// TIA Portal V19 export
FUNCTION "SUB_OUTPUT" : Void   // FC5, LAD
{ S7_Optimized_Access := 'TRUE' }
// stored: SetENOAutomatically false
   VAR_TEMP   // added for the SCL form of the ladder/FBD networks
      _w1 : Bool;
   END_VAR
BEGIN

REGION Network 2: "CENTRIFUGAL_PUMP-1"
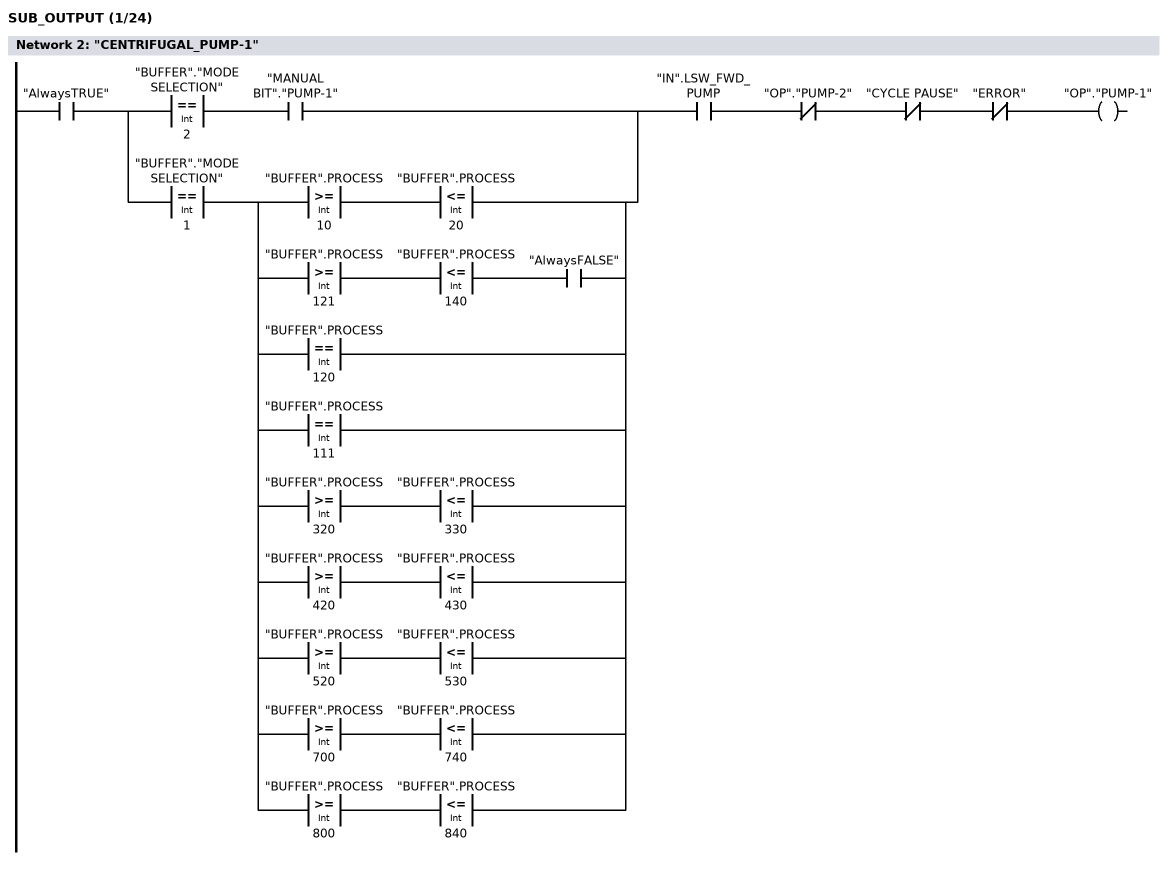
   RUNG wire#powerrail
      Contact( "AlwaysTRUE" )
      wire#w1
      { S7_Templates := "SrcType := Int" } EQ_Contact(in1 := "BUFFER"."MODE SELECTION", in2 := 2)
      Contact( "MANUAL BIT"."PUMP-1" )
      wire#w2
      Contact( "IN".LSW_FWD_PUMP )
      I_Contact( "OP"."PUMP-2" )
      I_Contact( "CYCLE PAUSE" )
      I_Contact( "ERROR" )
      Coil( "OP"."PUMP-1" )
   END_RUNG
   RUNG wire#w1
      { S7_Templates := "SrcType := Int" } EQ_Contact(in1 := "BUFFER"."MODE SELECTION", in2 := 1)
      wire#w3
      { S7_Templates := "SrcType := Int" } GE_Contact(in1 := "BUFFER".PROCESS, in2 := 10)
      { S7_Templates := "SrcType := Int" } LE_Contact(in1 := "BUFFER".PROCESS, in2 := 20)
   END_RUNG wire#w2
   RUNG wire#w3
      { S7_Templates := "SrcType := Int" } GE_Contact(in1 := "BUFFER".PROCESS, in2 := 121)
      { S7_Templates := "SrcType := Int" } LE_Contact(in1 := "BUFFER".PROCESS, in2 := 140)
      Contact( "AlwaysFALSE" )
   END_RUNG wire#w2
   RUNG wire#w3
      { S7_Templates := "SrcType := Int" } EQ_Contact(in1 := "BUFFER".PROCESS, in2 := 120)
   END_RUNG wire#w2
   RUNG wire#w3
      { S7_Templates := "SrcType := Int" } EQ_Contact(in1 := "BUFFER".PROCESS, in2 := 111)
   END_RUNG wire#w2
   RUNG wire#w3
      { S7_Templates := "SrcType := Int" } GE_Contact(in1 := "BUFFER".PROCESS, in2 := 320)
      { S7_Templates := "SrcType := Int" } LE_Contact(in1 := "BUFFER".PROCESS, in2 := 330)
   END_RUNG wire#w2
   RUNG wire#w3
      { S7_Templates := "SrcType := Int" } GE_Contact(in1 := "BUFFER".PROCESS, in2 := 420)
      { S7_Templates := "SrcType := Int" } LE_Contact(in1 := "BUFFER".PROCESS, in2 := 430)
   END_RUNG wire#w2
   RUNG wire#w3
      { S7_Templates := "SrcType := Int" } GE_Contact(in1 := "BUFFER".PROCESS, in2 := 520)
      { S7_Templates := "SrcType := Int" } LE_Contact(in1 := "BUFFER".PROCESS, in2 := 530)
   END_RUNG wire#w2
   RUNG wire#w3
      { S7_Templates := "SrcType := Int" } GE_Contact(in1 := "BUFFER".PROCESS, in2 := 700)
      { S7_Templates := "SrcType := Int" } LE_Contact(in1 := "BUFFER".PROCESS, in2 := 740)
   END_RUNG wire#w2
   RUNG wire#w3
      { S7_Templates := "SrcType := Int" } GE_Contact(in1 := "BUFFER".PROCESS, in2 := 800)
      { S7_Templates := "SrcType := Int" } LE_Contact(in1 := "BUFFER".PROCESS, in2 := 840)
   END_RUNG wire#w2
   // the same network as SCL:
   "OP"."PUMP-1" := "AlwaysTRUE" AND ((("BUFFER"."MODE SELECTION" = 2) AND "MANUAL BIT"."PUMP-1") OR (("BUFFER"."MODE SELECTION" = 1) AND ((("BUFFER".PROCESS >= 10) AND ("BUFFER".PROCESS <= 20)) OR (("BUFFER".PROCESS >= 121) AND ("BUFFER".PROCESS <= 140) AND "AlwaysFALSE") OR ("BUFFER".PROCESS = 120) OR ("BUFFER".PROCESS = 111) OR (("BUFFER".PROCESS >= 320) AND ("BUFFER".PROCESS <= 330)) OR (("BUFFER".PROCESS >= 420) AND ("BUFFER".PROCESS <= 430)) OR (("BUFFER".PROCESS >= 520) AND ("BUFFER".PROCESS <= 530)) OR (("BUFFER".PROCESS >= 700) AND ("BUFFER".PROCESS <= 740)) OR (("BUFFER".PROCESS >= 800) AND ("BUFFER".PROCESS <= 840))))) AND "IN".LSW_FWD_PUMP AND NOT "OP"."PUMP-2" AND NOT "CYCLE PAUSE" AND NOT "ERROR";
END_REGION

REGION Network 3: "CENTRIFUGAL_PUMP-2"
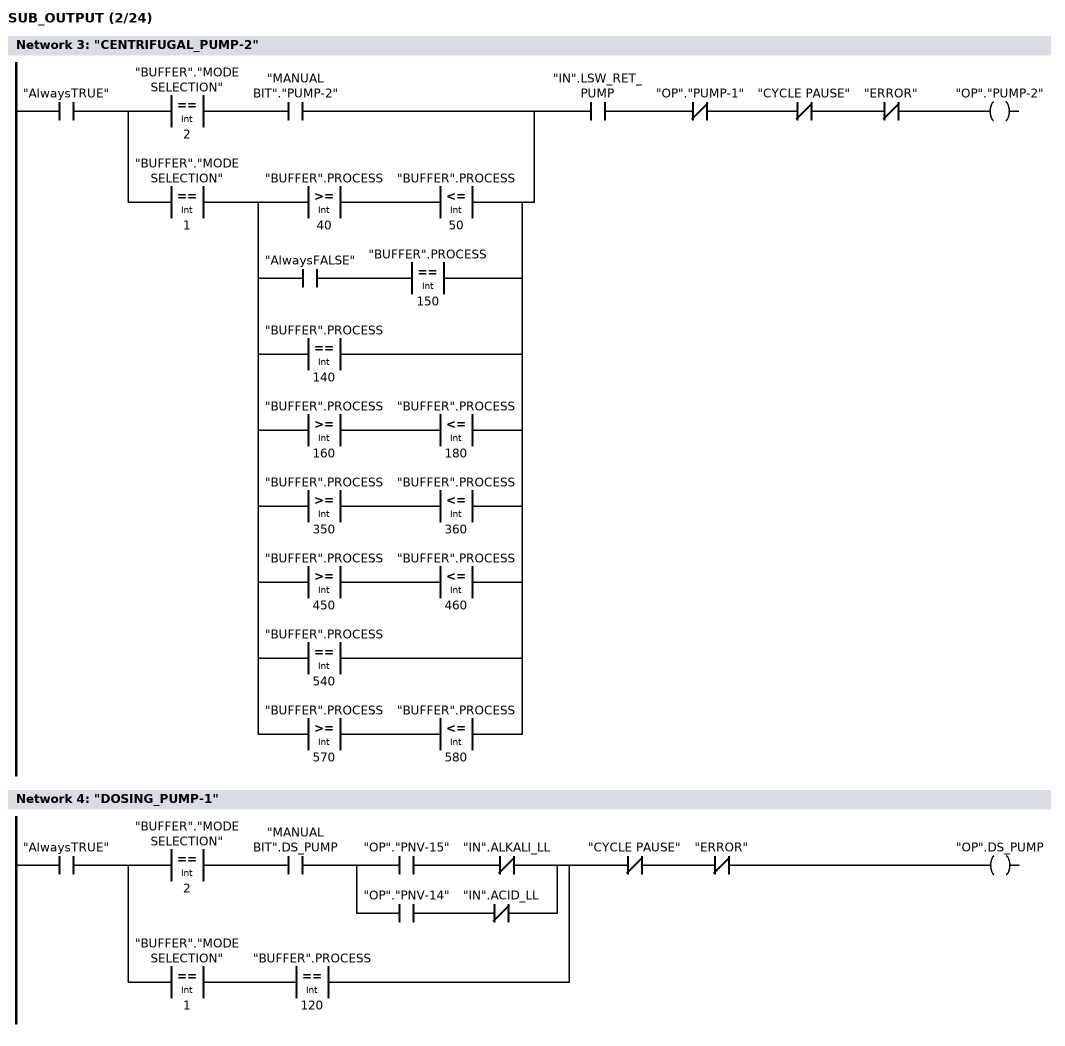
   RUNG wire#powerrail
      Contact( "AlwaysTRUE" )
      wire#w1
      { S7_Templates := "SrcType := Int" } EQ_Contact(in1 := "BUFFER"."MODE SELECTION", in2 := 2)
      Contact( "MANUAL BIT"."PUMP-2" )
      wire#w2
      Contact( "IN".LSW_RET_PUMP )
      I_Contact( "OP"."PUMP-1" )
      I_Contact( "CYCLE PAUSE" )
      I_Contact( "ERROR" )
      Coil( "OP"."PUMP-2" )
   END_RUNG
   RUNG wire#w1
      { S7_Templates := "SrcType := Int" } EQ_Contact(in1 := "BUFFER"."MODE SELECTION", in2 := 1)
      wire#w3
      { S7_Templates := "SrcType := Int" } GE_Contact(in1 := "BUFFER".PROCESS, in2 := 40)
      { S7_Templates := "SrcType := Int" } LE_Contact(in1 := "BUFFER".PROCESS, in2 := 50)
   END_RUNG wire#w2
   RUNG wire#w3
      Contact( "AlwaysFALSE" )
      { S7_Templates := "SrcType := Int" } EQ_Contact(in1 := "BUFFER".PROCESS, in2 := 150)
   END_RUNG wire#w2
   RUNG wire#w3
      { S7_Templates := "SrcType := Int" } EQ_Contact(in1 := "BUFFER".PROCESS, in2 := 140)
   END_RUNG wire#w2
   RUNG wire#w3
      { S7_Templates := "SrcType := Int" } GE_Contact(in1 := "BUFFER".PROCESS, in2 := 160)
      { S7_Templates := "SrcType := Int" } LE_Contact(in1 := "BUFFER".PROCESS, in2 := 180)
   END_RUNG wire#w2
   RUNG wire#w3
      { S7_Templates := "SrcType := Int" } GE_Contact(in1 := "BUFFER".PROCESS, in2 := 350)
      { S7_Templates := "SrcType := Int" } LE_Contact(in1 := "BUFFER".PROCESS, in2 := 360)
   END_RUNG wire#w2
   RUNG wire#w3
      { S7_Templates := "SrcType := Int" } GE_Contact(in1 := "BUFFER".PROCESS, in2 := 450)
      { S7_Templates := "SrcType := Int" } LE_Contact(in1 := "BUFFER".PROCESS, in2 := 460)
   END_RUNG wire#w2
   RUNG wire#w3
      { S7_Templates := "SrcType := Int" } EQ_Contact(in1 := "BUFFER".PROCESS, in2 := 540)
   END_RUNG wire#w2
   RUNG wire#w3
      { S7_Templates := "SrcType := Int" } GE_Contact(in1 := "BUFFER".PROCESS, in2 := 570)
      { S7_Templates := "SrcType := Int" } LE_Contact(in1 := "BUFFER".PROCESS, in2 := 580)
   END_RUNG wire#w2
   // the same network as SCL:
   "OP"."PUMP-2" := "AlwaysTRUE" AND ((("BUFFER"."MODE SELECTION" = 2) AND "MANUAL BIT"."PUMP-2") OR (("BUFFER"."MODE SELECTION" = 1) AND ((("BUFFER".PROCESS >= 40) AND ("BUFFER".PROCESS <= 50)) OR ("AlwaysFALSE" AND ("BUFFER".PROCESS = 150)) OR ("BUFFER".PROCESS = 140) OR (("BUFFER".PROCESS >= 160) AND ("BUFFER".PROCESS <= 180)) OR (("BUFFER".PROCESS >= 350) AND ("BUFFER".PROCESS <= 360)) OR (("BUFFER".PROCESS >= 450) AND ("BUFFER".PROCESS <= 460)) OR ("BUFFER".PROCESS = 540) OR (("BUFFER".PROCESS >= 570) AND ("BUFFER".PROCESS <= 580))))) AND "IN".LSW_RET_PUMP AND NOT "OP"."PUMP-1" AND NOT "CYCLE PAUSE" AND NOT "ERROR";
END_REGION

REGION Network 4: "DOSING_PUMP-1"
   RUNG wire#powerrail
      Contact( "AlwaysTRUE" )
      wire#w1
      { S7_Templates := "SrcType := Int" } EQ_Contact(in1 := "BUFFER"."MODE SELECTION", in2 := 2)
      Contact( "MANUAL BIT".DS_PUMP )
      wire#w2
      Contact( "OP"."PNV-15" )
      I_Contact( "IN".ALKALI_LL )
      wire#w3
      I_Contact( "CYCLE PAUSE" )
      I_Contact( "ERROR" )
      Coil( "OP".DS_PUMP )
   END_RUNG
   RUNG wire#w2
      Contact( "OP"."PNV-14" )
      I_Contact( "IN".ACID_LL )
   END_RUNG wire#w3
   RUNG wire#w1
      { S7_Templates := "SrcType := Int" } EQ_Contact(in1 := "BUFFER"."MODE SELECTION", in2 := 1)
      { S7_Templates := "SrcType := Int" } EQ_Contact(in1 := "BUFFER".PROCESS, in2 := 120)
   END_RUNG wire#w3
   // the same network as SCL:
   "OP".DS_PUMP := "AlwaysTRUE" AND ((("BUFFER"."MODE SELECTION" = 2) AND "MANUAL BIT".DS_PUMP AND (("OP"."PNV-15" AND NOT "IN".ALKALI_LL) OR ("OP"."PNV-14" AND NOT "IN".ACID_LL))) OR (("BUFFER"."MODE SELECTION" = 1) AND ("BUFFER".PROCESS = 120))) AND NOT "CYCLE PAUSE" AND NOT "ERROR";
END_REGION

REGION Network 5: "PBV-125 PURIFIED WATER VESSEL OUTLET VALVE"
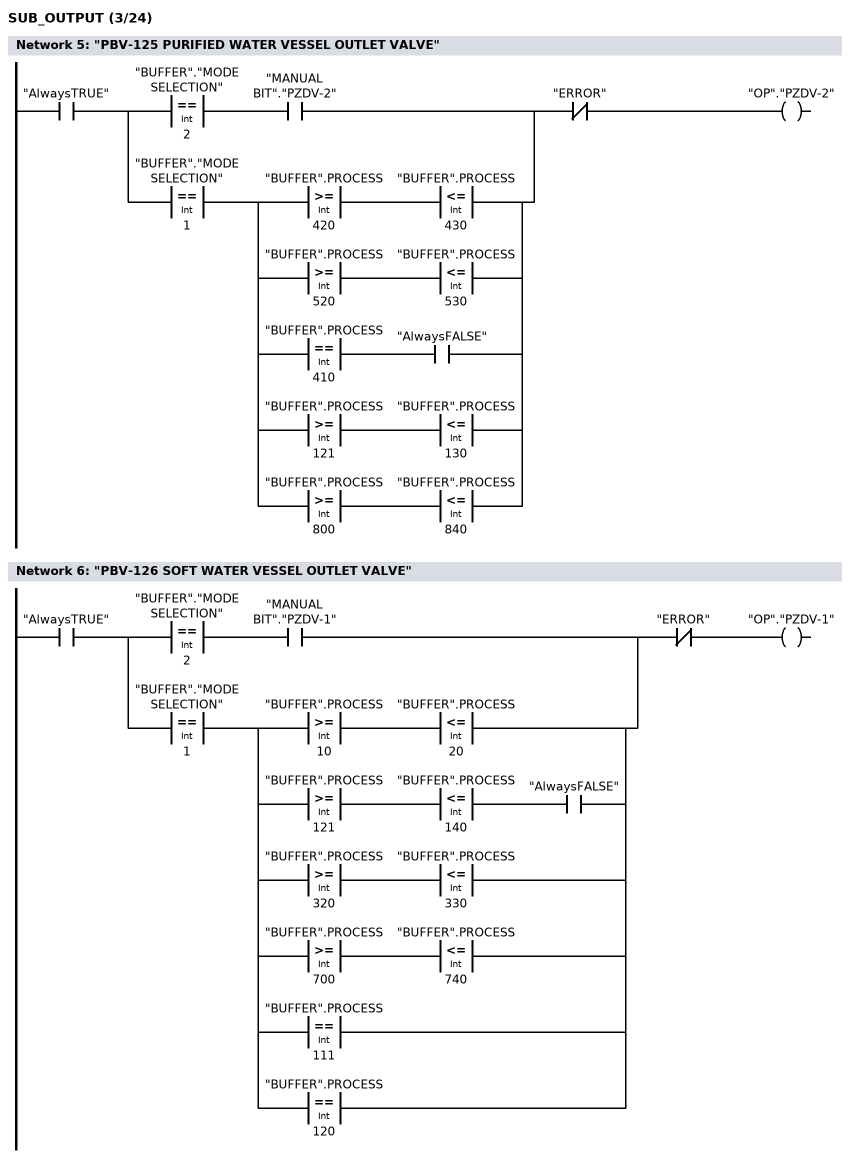
   RUNG wire#powerrail
      Contact( "AlwaysTRUE" )
      wire#w1
      { S7_Templates := "SrcType := Int" } EQ_Contact(in1 := "BUFFER"."MODE SELECTION", in2 := 2)
      Contact( "MANUAL BIT"."PZDV-2" )
      wire#w2
      I_Contact( "ERROR" )
      Coil( "OP"."PZDV-2" )
   END_RUNG
   RUNG wire#w1
      { S7_Templates := "SrcType := Int" } EQ_Contact(in1 := "BUFFER"."MODE SELECTION", in2 := 1)
      wire#w3
      { S7_Templates := "SrcType := Int" } GE_Contact(in1 := "BUFFER".PROCESS, in2 := 420)
      { S7_Templates := "SrcType := Int" } LE_Contact(in1 := "BUFFER".PROCESS, in2 := 430)
   END_RUNG wire#w2
   RUNG wire#w3
      { S7_Templates := "SrcType := Int" } GE_Contact(in1 := "BUFFER".PROCESS, in2 := 520)
      { S7_Templates := "SrcType := Int" } LE_Contact(in1 := "BUFFER".PROCESS, in2 := 530)
   END_RUNG wire#w2
   RUNG wire#w3
      { S7_Templates := "SrcType := Int" } EQ_Contact(in1 := "BUFFER".PROCESS, in2 := 410)
      Contact( "AlwaysFALSE" )
   END_RUNG wire#w2
   RUNG wire#w3
      { S7_Templates := "SrcType := Int" } GE_Contact(in1 := "BUFFER".PROCESS, in2 := 121)
      { S7_Templates := "SrcType := Int" } LE_Contact(in1 := "BUFFER".PROCESS, in2 := 130)
   END_RUNG wire#w2
   RUNG wire#w3
      { S7_Templates := "SrcType := Int" } GE_Contact(in1 := "BUFFER".PROCESS, in2 := 800)
      { S7_Templates := "SrcType := Int" } LE_Contact(in1 := "BUFFER".PROCESS, in2 := 840)
   END_RUNG wire#w2
   // the same network as SCL:
   "OP"."PZDV-2" := "AlwaysTRUE" AND ((("BUFFER"."MODE SELECTION" = 2) AND "MANUAL BIT"."PZDV-2") OR (("BUFFER"."MODE SELECTION" = 1) AND ((("BUFFER".PROCESS >= 420) AND ("BUFFER".PROCESS <= 430)) OR (("BUFFER".PROCESS >= 520) AND ("BUFFER".PROCESS <= 530)) OR (("BUFFER".PROCESS = 410) AND "AlwaysFALSE") OR (("BUFFER".PROCESS >= 121) AND ("BUFFER".PROCESS <= 130)) OR (("BUFFER".PROCESS >= 800) AND ("BUFFER".PROCESS <= 840))))) AND NOT "ERROR";
END_REGION

REGION Network 6: "PBV-126 SOFT WATER VESSEL OUTLET VALVE"
   RUNG wire#powerrail
      Contact( "AlwaysTRUE" )
      wire#w1
      { S7_Templates := "SrcType := Int" } EQ_Contact(in1 := "BUFFER"."MODE SELECTION", in2 := 2)
      Contact( "MANUAL BIT"."PZDV-1" )
      wire#w2
      I_Contact( "ERROR" )
      Coil( "OP"."PZDV-1" )
   END_RUNG
   RUNG wire#w1
      { S7_Templates := "SrcType := Int" } EQ_Contact(in1 := "BUFFER"."MODE SELECTION", in2 := 1)
      wire#w3
      { S7_Templates := "SrcType := Int" } GE_Contact(in1 := "BUFFER".PROCESS, in2 := 10)
      { S7_Templates := "SrcType := Int" } LE_Contact(in1 := "BUFFER".PROCESS, in2 := 20)
   END_RUNG wire#w2
   RUNG wire#w3
      { S7_Templates := "SrcType := Int" } GE_Contact(in1 := "BUFFER".PROCESS, in2 := 121)
      { S7_Templates := "SrcType := Int" } LE_Contact(in1 := "BUFFER".PROCESS, in2 := 140)
      Contact( "AlwaysFALSE" )
   END_RUNG wire#w2
   RUNG wire#w3
      { S7_Templates := "SrcType := Int" } GE_Contact(in1 := "BUFFER".PROCESS, in2 := 320)
      { S7_Templates := "SrcType := Int" } LE_Contact(in1 := "BUFFER".PROCESS, in2 := 330)
   END_RUNG wire#w2
   RUNG wire#w3
      { S7_Templates := "SrcType := Int" } GE_Contact(in1 := "BUFFER".PROCESS, in2 := 700)
      { S7_Templates := "SrcType := Int" } LE_Contact(in1 := "BUFFER".PROCESS, in2 := 740)
   END_RUNG wire#w2
   RUNG wire#w3
      { S7_Templates := "SrcType := Int" } EQ_Contact(in1 := "BUFFER".PROCESS, in2 := 111)
   END_RUNG wire#w2
   RUNG wire#w3
      { S7_Templates := "SrcType := Int" } EQ_Contact(in1 := "BUFFER".PROCESS, in2 := 120)
   END_RUNG wire#w2
   // the same network as SCL:
   "OP"."PZDV-1" := "AlwaysTRUE" AND ((("BUFFER"."MODE SELECTION" = 2) AND "MANUAL BIT"."PZDV-1") OR (("BUFFER"."MODE SELECTION" = 1) AND ((("BUFFER".PROCESS >= 10) AND ("BUFFER".PROCESS <= 20)) OR (("BUFFER".PROCESS >= 121) AND ("BUFFER".PROCESS <= 140) AND "AlwaysFALSE") OR (("BUFFER".PROCESS >= 320) AND ("BUFFER".PROCESS <= 330)) OR (("BUFFER".PROCESS >= 700) AND ("BUFFER".PROCESS <= 740)) OR ("BUFFER".PROCESS = 111) OR ("BUFFER".PROCESS = 120)))) AND NOT "ERROR";
END_REGION

REGION Network 7: "PBV-127 PW INLET LINE"
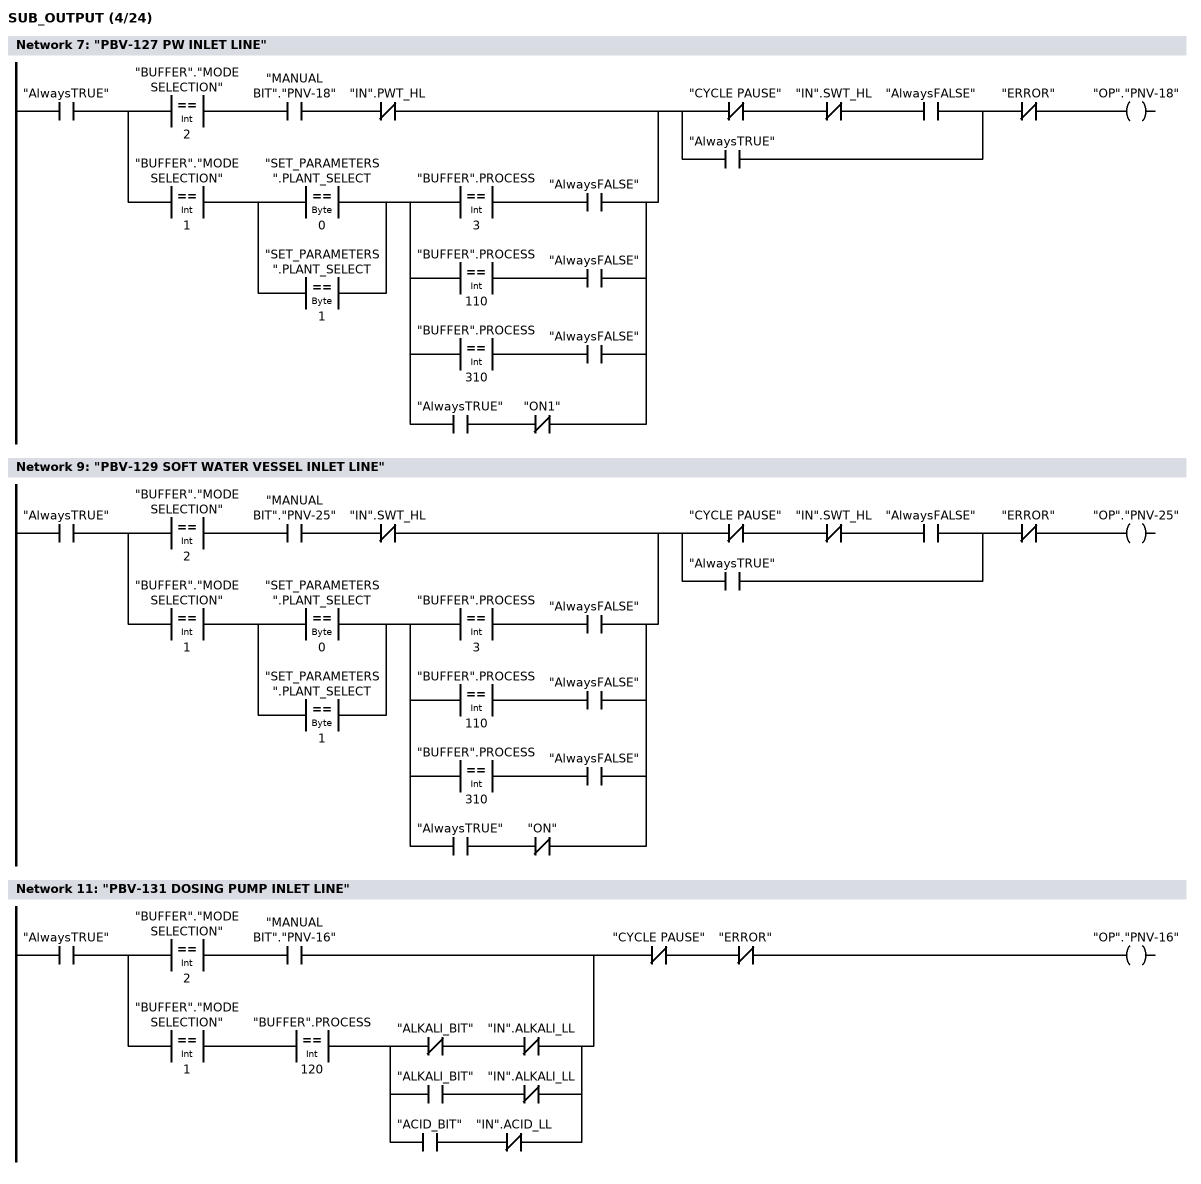
   RUNG wire#powerrail
      Contact( "AlwaysTRUE" )
      wire#w1
      { S7_Templates := "SrcType := Int" } EQ_Contact(in1 := "BUFFER"."MODE SELECTION", in2 := 2)
      Contact( "MANUAL BIT"."PNV-18" )
      I_Contact( "IN".PWT_HL )
      wire#w2
      I_Contact( "CYCLE PAUSE" )
      I_Contact( "IN".SWT_HL )
      Contact( "AlwaysFALSE" )
      wire#w5
      I_Contact( "ERROR" )
      Coil( "OP"."PNV-18" )
   END_RUNG
   RUNG wire#w1
      { S7_Templates := "SrcType := Int" } EQ_Contact(in1 := "BUFFER"."MODE SELECTION", in2 := 1)
      wire#w3
      { S7_Templates := "SrcType := Byte" } EQ_Contact(in1 := "SET_PARAMETERS".PLANT_SELECT, in2 := 0)
      wire#w4
      { S7_Templates := "SrcType := Int" } EQ_Contact(in1 := "BUFFER".PROCESS, in2 := 3)
      Contact( "AlwaysFALSE" )
   END_RUNG wire#w2
   RUNG wire#w3
      { S7_Templates := "SrcType := Byte" } EQ_Contact(in1 := "SET_PARAMETERS".PLANT_SELECT, in2 := 1)
   END_RUNG wire#w4
   RUNG wire#w4
      { S7_Templates := "SrcType := Int" } EQ_Contact(in1 := "BUFFER".PROCESS, in2 := 110)
      Contact( "AlwaysFALSE" )
   END_RUNG wire#w2
   RUNG wire#w4
      { S7_Templates := "SrcType := Int" } EQ_Contact(in1 := "BUFFER".PROCESS, in2 := 310)
      Contact( "AlwaysFALSE" )
   END_RUNG wire#w2
   RUNG wire#w4
      Contact( "AlwaysTRUE" )
      I_Contact( "ON1" )
   END_RUNG wire#w2
   RUNG wire#w2
      Contact( "AlwaysTRUE" )
   END_RUNG wire#w5
   // the same network as SCL:
   "OP"."PNV-18" := "AlwaysTRUE" AND ((("BUFFER"."MODE SELECTION" = 2) AND "MANUAL BIT"."PNV-18" AND NOT "IN".PWT_HL) OR (("BUFFER"."MODE SELECTION" = 1) AND (("SET_PARAMETERS".PLANT_SELECT = 0) OR ("SET_PARAMETERS".PLANT_SELECT = 1)) AND ((("BUFFER".PROCESS = 3) AND "AlwaysFALSE") OR (("BUFFER".PROCESS = 110) AND "AlwaysFALSE") OR (("BUFFER".PROCESS = 310) AND "AlwaysFALSE") OR ("AlwaysTRUE" AND NOT "ON1")))) AND ((NOT "CYCLE PAUSE" AND NOT "IN".SWT_HL AND "AlwaysFALSE") OR "AlwaysTRUE") AND NOT "ERROR";
END_REGION

REGION Network 8: "PBV-128 PURIFIED WATER VESSEL–SPRAY BALL INLET LINE"//////////////////NA
END_REGION

REGION Network 9: "PBV-129 SOFT WATER VESSEL INLET LINE"
   RUNG wire#powerrail
      Contact( "AlwaysTRUE" )
      wire#w1
      { S7_Templates := "SrcType := Int" } EQ_Contact(in1 := "BUFFER"."MODE SELECTION", in2 := 2)
      Contact( "MANUAL BIT"."PNV-25" )
      I_Contact( "IN".SWT_HL )
      wire#w2
      I_Contact( "CYCLE PAUSE" )
      I_Contact( "IN".SWT_HL )
      Contact( "AlwaysFALSE" )
      wire#w5
      I_Contact( "ERROR" )
      Coil( "OP"."PNV-25" )
   END_RUNG
   RUNG wire#w1
      { S7_Templates := "SrcType := Int" } EQ_Contact(in1 := "BUFFER"."MODE SELECTION", in2 := 1)
      wire#w3
      { S7_Templates := "SrcType := Byte" } EQ_Contact(in1 := "SET_PARAMETERS".PLANT_SELECT, in2 := 0)
      wire#w4
      { S7_Templates := "SrcType := Int" } EQ_Contact(in1 := "BUFFER".PROCESS, in2 := 3)
      Contact( "AlwaysFALSE" )
   END_RUNG wire#w2
   RUNG wire#w3
      { S7_Templates := "SrcType := Byte" } EQ_Contact(in1 := "SET_PARAMETERS".PLANT_SELECT, in2 := 1)
   END_RUNG wire#w4
   RUNG wire#w4
      { S7_Templates := "SrcType := Int" } EQ_Contact(in1 := "BUFFER".PROCESS, in2 := 110)
      Contact( "AlwaysFALSE" )
   END_RUNG wire#w2
   RUNG wire#w4
      { S7_Templates := "SrcType := Int" } EQ_Contact(in1 := "BUFFER".PROCESS, in2 := 310)
      Contact( "AlwaysFALSE" )
   END_RUNG wire#w2
   RUNG wire#w4
      Contact( "AlwaysTRUE" )
      I_Contact( "ON" )
   END_RUNG wire#w2
   RUNG wire#w2
      Contact( "AlwaysTRUE" )
   END_RUNG wire#w5
   // the same network as SCL:
   "OP"."PNV-25" := "AlwaysTRUE" AND ((("BUFFER"."MODE SELECTION" = 2) AND "MANUAL BIT"."PNV-25" AND NOT "IN".SWT_HL) OR (("BUFFER"."MODE SELECTION" = 1) AND (("SET_PARAMETERS".PLANT_SELECT = 0) OR ("SET_PARAMETERS".PLANT_SELECT = 1)) AND ((("BUFFER".PROCESS = 3) AND "AlwaysFALSE") OR (("BUFFER".PROCESS = 110) AND "AlwaysFALSE") OR (("BUFFER".PROCESS = 310) AND "AlwaysFALSE") OR ("AlwaysTRUE" AND NOT "ON")))) AND ((NOT "CYCLE PAUSE" AND NOT "IN".SWT_HL AND "AlwaysFALSE") OR "AlwaysTRUE") AND NOT "ERROR";
END_REGION

REGION Network 10: "PBV-130 SOFT WATER VESSEL–SPRAY BALL INLET LINE" /////////////////NA
END_REGION

REGION Network 11: "PBV-131 DOSING PUMP INLET LINE"
   RUNG wire#powerrail
      Contact( "AlwaysTRUE" )
      wire#w1
      { S7_Templates := "SrcType := Int" } EQ_Contact(in1 := "BUFFER"."MODE SELECTION", in2 := 2)
      Contact( "MANUAL BIT"."PNV-16" )
      wire#w2
      I_Contact( "CYCLE PAUSE" )
      I_Contact( "ERROR" )
      Coil( "OP"."PNV-16" )
   END_RUNG
   RUNG wire#w1
      { S7_Templates := "SrcType := Int" } EQ_Contact(in1 := "BUFFER"."MODE SELECTION", in2 := 1)
      { S7_Templates := "SrcType := Int" } EQ_Contact(in1 := "BUFFER".PROCESS, in2 := 120)
      wire#w3
      I_Contact( "ALKALI_BIT" )
      I_Contact( "IN".ALKALI_LL )
   END_RUNG wire#w2
   RUNG wire#w3
      Contact( "ALKALI_BIT" )
      I_Contact( "IN".ALKALI_LL )
   END_RUNG wire#w2
   RUNG wire#w3
      Contact( "ACID_BIT" )
      I_Contact( "IN".ACID_LL )
   END_RUNG wire#w2
   // the same network as SCL:
   "OP"."PNV-16" := "AlwaysTRUE" AND ((("BUFFER"."MODE SELECTION" = 2) AND "MANUAL BIT"."PNV-16") OR (("BUFFER"."MODE SELECTION" = 1) AND ("BUFFER".PROCESS = 120) AND ((NOT "ALKALI_BIT" AND NOT "IN".ALKALI_LL) OR ("ALKALI_BIT" AND NOT "IN".ALKALI_LL) OR ("ACID_BIT" AND NOT "IN".ACID_LL)))) AND NOT "CYCLE PAUSE" AND NOT "ERROR";
END_REGION

REGION Network 12: "PBV-132 PURIFIED WATER VESSEL OUTLET LINE" /////////////////NA
END_REGION

REGION Network 13: "PBV-133 SOFT WATER VESSEL OUTLET LINE" /////////////////NA
END_REGION

REGION Network 14: "PBV-134 FORWARD PUMP INLET LINE" /////////////////NA
END_REGION

REGION Network 15: "PBV-135 REVERSE PUMP CASING DRAIN"
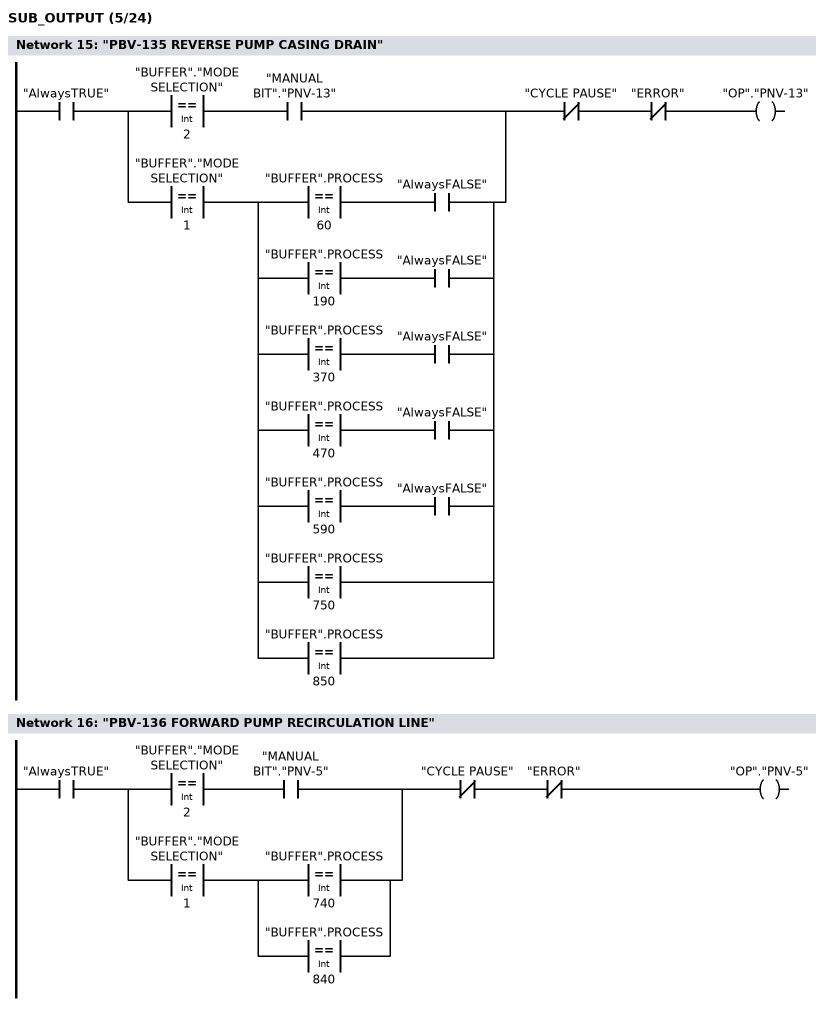
   RUNG wire#powerrail
      Contact( "AlwaysTRUE" )
      wire#w1
      { S7_Templates := "SrcType := Int" } EQ_Contact(in1 := "BUFFER"."MODE SELECTION", in2 := 2)
      Contact( "MANUAL BIT"."PNV-13" )
      wire#w2
      I_Contact( "CYCLE PAUSE" )
      I_Contact( "ERROR" )
      Coil( "OP"."PNV-13" )
   END_RUNG
   RUNG wire#w1
      { S7_Templates := "SrcType := Int" } EQ_Contact(in1 := "BUFFER"."MODE SELECTION", in2 := 1)
      wire#w3
      { S7_Templates := "SrcType := Int" } EQ_Contact(in1 := "BUFFER".PROCESS, in2 := 60)
      Contact( "AlwaysFALSE" )
   END_RUNG wire#w2
   RUNG wire#w3
      { S7_Templates := "SrcType := Int" } EQ_Contact(in1 := "BUFFER".PROCESS, in2 := 190)
      Contact( "AlwaysFALSE" )
   END_RUNG wire#w2
   RUNG wire#w3
      { S7_Templates := "SrcType := Int" } EQ_Contact(in1 := "BUFFER".PROCESS, in2 := 370)
      Contact( "AlwaysFALSE" )
   END_RUNG wire#w2
   RUNG wire#w3
      { S7_Templates := "SrcType := Int" } EQ_Contact(in1 := "BUFFER".PROCESS, in2 := 470)
      Contact( "AlwaysFALSE" )
   END_RUNG wire#w2
   RUNG wire#w3
      { S7_Templates := "SrcType := Int" } EQ_Contact(in1 := "BUFFER".PROCESS, in2 := 590)
      Contact( "AlwaysFALSE" )
   END_RUNG wire#w2
   RUNG wire#w3
      { S7_Templates := "SrcType := Int" } EQ_Contact(in1 := "BUFFER".PROCESS, in2 := 750)
   END_RUNG wire#w2
   RUNG wire#w3
      { S7_Templates := "SrcType := Int" } EQ_Contact(in1 := "BUFFER".PROCESS, in2 := 850)
   END_RUNG wire#w2
   // the same network as SCL:
   "OP"."PNV-13" := "AlwaysTRUE" AND ((("BUFFER"."MODE SELECTION" = 2) AND "MANUAL BIT"."PNV-13") OR (("BUFFER"."MODE SELECTION" = 1) AND ((("BUFFER".PROCESS = 60) AND "AlwaysFALSE") OR (("BUFFER".PROCESS = 190) AND "AlwaysFALSE") OR (("BUFFER".PROCESS = 370) AND "AlwaysFALSE") OR (("BUFFER".PROCESS = 470) AND "AlwaysFALSE") OR (("BUFFER".PROCESS = 590) AND "AlwaysFALSE") OR ("BUFFER".PROCESS = 750) OR ("BUFFER".PROCESS = 850)))) AND NOT "CYCLE PAUSE" AND NOT "ERROR";
END_REGION

REGION Network 16: "PBV-136 FORWARD PUMP RECIRCULATION LINE"
   RUNG wire#powerrail
      Contact( "AlwaysTRUE" )
      wire#w1
      { S7_Templates := "SrcType := Int" } EQ_Contact(in1 := "BUFFER"."MODE SELECTION", in2 := 2)
      Contact( "MANUAL BIT"."PNV-5" )
      wire#w2
      I_Contact( "CYCLE PAUSE" )
      I_Contact( "ERROR" )
      Coil( "OP"."PNV-5" )
   END_RUNG
   RUNG wire#w1
      { S7_Templates := "SrcType := Int" } EQ_Contact(in1 := "BUFFER"."MODE SELECTION", in2 := 1)
      wire#w3
      { S7_Templates := "SrcType := Int" } EQ_Contact(in1 := "BUFFER".PROCESS, in2 := 740)
   END_RUNG wire#w2
   RUNG wire#w3
      { S7_Templates := "SrcType := Int" } EQ_Contact(in1 := "BUFFER".PROCESS, in2 := 840)
   END_RUNG wire#w2
   // the same network as SCL:
   "OP"."PNV-5" := "AlwaysTRUE" AND ((("BUFFER"."MODE SELECTION" = 2) AND "MANUAL BIT"."PNV-5") OR (("BUFFER"."MODE SELECTION" = 1) AND (("BUFFER".PROCESS = 740) OR ("BUFFER".PROCESS = 840)))) AND NOT "CYCLE PAUSE" AND NOT "ERROR";
END_REGION

REGION Network 17: "PBV-137 FORWARD PUMP TO HEAT EXCHANGER LINE"
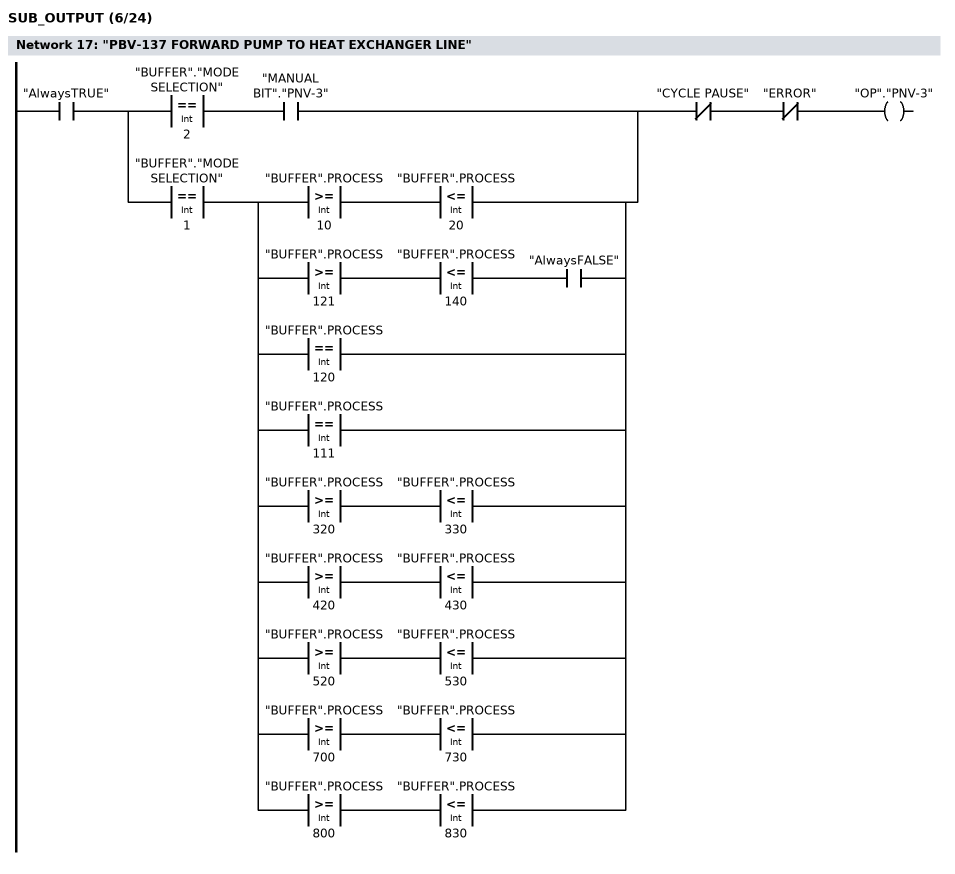
   RUNG wire#powerrail
      Contact( "AlwaysTRUE" )
      wire#w1
      { S7_Templates := "SrcType := Int" } EQ_Contact(in1 := "BUFFER"."MODE SELECTION", in2 := 2)
      Contact( "MANUAL BIT"."PNV-3" )
      wire#w2
      I_Contact( "CYCLE PAUSE" )
      I_Contact( "ERROR" )
      Coil( "OP"."PNV-3" )
   END_RUNG
   RUNG wire#w1
      { S7_Templates := "SrcType := Int" } EQ_Contact(in1 := "BUFFER"."MODE SELECTION", in2 := 1)
      wire#w3
      { S7_Templates := "SrcType := Int" } GE_Contact(in1 := "BUFFER".PROCESS, in2 := 10)
      { S7_Templates := "SrcType := Int" } LE_Contact(in1 := "BUFFER".PROCESS, in2 := 20)
   END_RUNG wire#w2
   RUNG wire#w3
      { S7_Templates := "SrcType := Int" } GE_Contact(in1 := "BUFFER".PROCESS, in2 := 121)
      { S7_Templates := "SrcType := Int" } LE_Contact(in1 := "BUFFER".PROCESS, in2 := 140)
      Contact( "AlwaysFALSE" )
   END_RUNG wire#w2
   RUNG wire#w3
      { S7_Templates := "SrcType := Int" } EQ_Contact(in1 := "BUFFER".PROCESS, in2 := 120)
   END_RUNG wire#w2
   RUNG wire#w3
      { S7_Templates := "SrcType := Int" } EQ_Contact(in1 := "BUFFER".PROCESS, in2 := 111)
   END_RUNG wire#w2
   RUNG wire#w3
      { S7_Templates := "SrcType := Int" } GE_Contact(in1 := "BUFFER".PROCESS, in2 := 320)
      { S7_Templates := "SrcType := Int" } LE_Contact(in1 := "BUFFER".PROCESS, in2 := 330)
   END_RUNG wire#w2
   RUNG wire#w3
      { S7_Templates := "SrcType := Int" } GE_Contact(in1 := "BUFFER".PROCESS, in2 := 420)
      { S7_Templates := "SrcType := Int" } LE_Contact(in1 := "BUFFER".PROCESS, in2 := 430)
   END_RUNG wire#w2
   RUNG wire#w3
      { S7_Templates := "SrcType := Int" } GE_Contact(in1 := "BUFFER".PROCESS, in2 := 520)
      { S7_Templates := "SrcType := Int" } LE_Contact(in1 := "BUFFER".PROCESS, in2 := 530)
   END_RUNG wire#w2
   RUNG wire#w3
      { S7_Templates := "SrcType := Int" } GE_Contact(in1 := "BUFFER".PROCESS, in2 := 700)
      { S7_Templates := "SrcType := Int" } LE_Contact(in1 := "BUFFER".PROCESS, in2 := 730)
   END_RUNG wire#w2
   RUNG wire#w3
      { S7_Templates := "SrcType := Int" } GE_Contact(in1 := "BUFFER".PROCESS, in2 := 800)
      { S7_Templates := "SrcType := Int" } LE_Contact(in1 := "BUFFER".PROCESS, in2 := 830)
   END_RUNG wire#w2
   // the same network as SCL:
   "OP"."PNV-3" := "AlwaysTRUE" AND ((("BUFFER"."MODE SELECTION" = 2) AND "MANUAL BIT"."PNV-3") OR (("BUFFER"."MODE SELECTION" = 1) AND ((("BUFFER".PROCESS >= 10) AND ("BUFFER".PROCESS <= 20)) OR (("BUFFER".PROCESS >= 121) AND ("BUFFER".PROCESS <= 140) AND "AlwaysFALSE") OR ("BUFFER".PROCESS = 120) OR ("BUFFER".PROCESS = 111) OR (("BUFFER".PROCESS >= 320) AND ("BUFFER".PROCESS <= 330)) OR (("BUFFER".PROCESS >= 420) AND ("BUFFER".PROCESS <= 430)) OR (("BUFFER".PROCESS >= 520) AND ("BUFFER".PROCESS <= 530)) OR (("BUFFER".PROCESS >= 700) AND ("BUFFER".PROCESS <= 730)) OR (("BUFFER".PROCESS >= 800) AND ("BUFFER".PROCESS <= 830))))) AND NOT "CYCLE PAUSE" AND NOT "ERROR";
END_REGION

REGION Network 18: "PBV-138 PURIFIED WATER DRAIN LINE" /////////////////NA
END_REGION

REGION Network 19: "PAV-139 HEAT EXCHANGER BYPASS DRAIN"
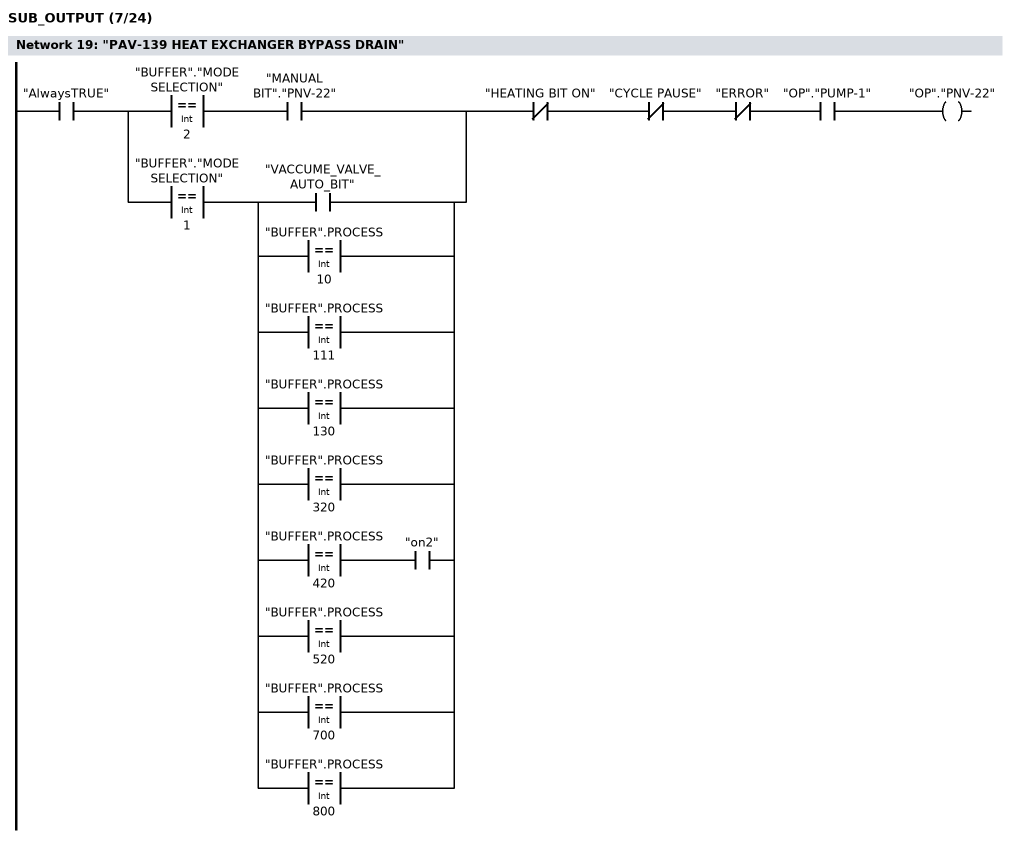
   RUNG wire#powerrail
      Contact( "AlwaysTRUE" )
      wire#w1
      { S7_Templates := "SrcType := Int" } EQ_Contact(in1 := "BUFFER"."MODE SELECTION", in2 := 2)
      Contact( "MANUAL BIT"."PNV-22" )
      wire#w2
      I_Contact( "HEATING BIT ON" )
      I_Contact( "CYCLE PAUSE" )
      I_Contact( "ERROR" )
      Contact( "OP"."PUMP-1" )
      Coil( "OP"."PNV-22" )
   END_RUNG
   RUNG wire#w1
      { S7_Templates := "SrcType := Int" } EQ_Contact(in1 := "BUFFER"."MODE SELECTION", in2 := 1)
      wire#w3
      Contact( "VACCUME_VALVE_AUTO_BIT" )
   END_RUNG wire#w2
   RUNG wire#w3
      { S7_Templates := "SrcType := Int" } EQ_Contact(in1 := "BUFFER".PROCESS, in2 := 10)
   END_RUNG wire#w2
   RUNG wire#w3
      { S7_Templates := "SrcType := Int" } EQ_Contact(in1 := "BUFFER".PROCESS, in2 := 111)
   END_RUNG wire#w2
   RUNG wire#w3
      { S7_Templates := "SrcType := Int" } EQ_Contact(in1 := "BUFFER".PROCESS, in2 := 130)
   END_RUNG wire#w2
   RUNG wire#w3
      { S7_Templates := "SrcType := Int" } EQ_Contact(in1 := "BUFFER".PROCESS, in2 := 320)
   END_RUNG wire#w2
   RUNG wire#w3
      { S7_Templates := "SrcType := Int" } EQ_Contact(in1 := "BUFFER".PROCESS, in2 := 420)
      Contact( "on2" )
   END_RUNG wire#w2
   RUNG wire#w3
      { S7_Templates := "SrcType := Int" } EQ_Contact(in1 := "BUFFER".PROCESS, in2 := 520)
   END_RUNG wire#w2
   RUNG wire#w3
      { S7_Templates := "SrcType := Int" } EQ_Contact(in1 := "BUFFER".PROCESS, in2 := 700)
   END_RUNG wire#w2
   RUNG wire#w3
      { S7_Templates := "SrcType := Int" } EQ_Contact(in1 := "BUFFER".PROCESS, in2 := 800)
   END_RUNG wire#w2
   // the same network as SCL:
   "OP"."PNV-22" := "AlwaysTRUE" AND ((("BUFFER"."MODE SELECTION" = 2) AND "MANUAL BIT"."PNV-22") OR (("BUFFER"."MODE SELECTION" = 1) AND ("VACCUME_VALVE_AUTO_BIT" OR ("BUFFER".PROCESS = 10) OR ("BUFFER".PROCESS = 111) OR ("BUFFER".PROCESS = 130) OR ("BUFFER".PROCESS = 320) OR (("BUFFER".PROCESS = 420) AND "on2") OR ("BUFFER".PROCESS = 520) OR ("BUFFER".PROCESS = 700) OR ("BUFFER".PROCESS = 800)))) AND NOT "HEATING BIT ON" AND NOT "CYCLE PAUSE" AND NOT "ERROR" AND "OP"."PUMP-1";
END_REGION

REGION Network 20: "PBV-140 HEAT EXCHANGER INLET LINE"
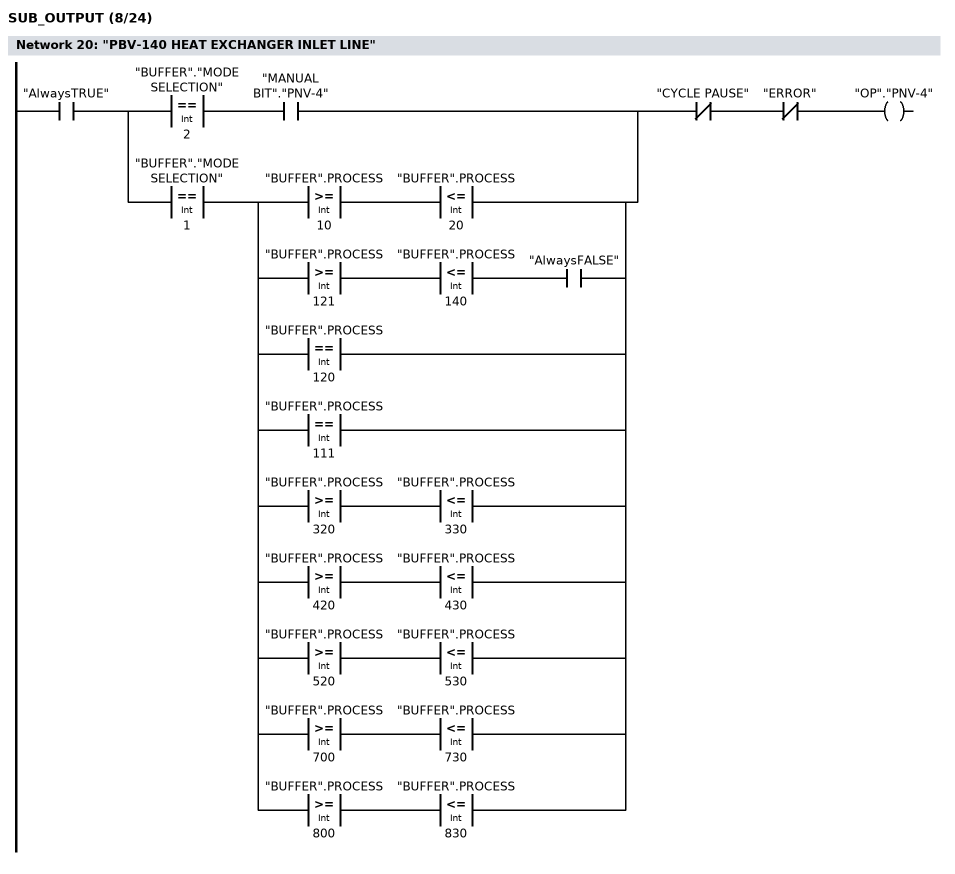
   RUNG wire#powerrail
      Contact( "AlwaysTRUE" )
      wire#w1
      { S7_Templates := "SrcType := Int" } EQ_Contact(in1 := "BUFFER"."MODE SELECTION", in2 := 2)
      Contact( "MANUAL BIT"."PNV-4" )
      wire#w2
      I_Contact( "CYCLE PAUSE" )
      I_Contact( "ERROR" )
      Coil( "OP"."PNV-4" )
   END_RUNG
   RUNG wire#w1
      { S7_Templates := "SrcType := Int" } EQ_Contact(in1 := "BUFFER"."MODE SELECTION", in2 := 1)
      wire#w3
      { S7_Templates := "SrcType := Int" } GE_Contact(in1 := "BUFFER".PROCESS, in2 := 10)
      { S7_Templates := "SrcType := Int" } LE_Contact(in1 := "BUFFER".PROCESS, in2 := 20)
   END_RUNG wire#w2
   RUNG wire#w3
      { S7_Templates := "SrcType := Int" } GE_Contact(in1 := "BUFFER".PROCESS, in2 := 121)
      { S7_Templates := "SrcType := Int" } LE_Contact(in1 := "BUFFER".PROCESS, in2 := 140)
      Contact( "AlwaysFALSE" )
   END_RUNG wire#w2
   RUNG wire#w3
      { S7_Templates := "SrcType := Int" } EQ_Contact(in1 := "BUFFER".PROCESS, in2 := 120)
   END_RUNG wire#w2
   RUNG wire#w3
      { S7_Templates := "SrcType := Int" } EQ_Contact(in1 := "BUFFER".PROCESS, in2 := 111)
   END_RUNG wire#w2
   RUNG wire#w3
      { S7_Templates := "SrcType := Int" } GE_Contact(in1 := "BUFFER".PROCESS, in2 := 320)
      { S7_Templates := "SrcType := Int" } LE_Contact(in1 := "BUFFER".PROCESS, in2 := 330)
   END_RUNG wire#w2
   RUNG wire#w3
      { S7_Templates := "SrcType := Int" } GE_Contact(in1 := "BUFFER".PROCESS, in2 := 420)
      { S7_Templates := "SrcType := Int" } LE_Contact(in1 := "BUFFER".PROCESS, in2 := 430)
   END_RUNG wire#w2
   RUNG wire#w3
      { S7_Templates := "SrcType := Int" } GE_Contact(in1 := "BUFFER".PROCESS, in2 := 520)
      { S7_Templates := "SrcType := Int" } LE_Contact(in1 := "BUFFER".PROCESS, in2 := 530)
   END_RUNG wire#w2
   RUNG wire#w3
      { S7_Templates := "SrcType := Int" } GE_Contact(in1 := "BUFFER".PROCESS, in2 := 700)
      { S7_Templates := "SrcType := Int" } LE_Contact(in1 := "BUFFER".PROCESS, in2 := 730)
   END_RUNG wire#w2
   RUNG wire#w3
      { S7_Templates := "SrcType := Int" } GE_Contact(in1 := "BUFFER".PROCESS, in2 := 800)
      { S7_Templates := "SrcType := Int" } LE_Contact(in1 := "BUFFER".PROCESS, in2 := 830)
   END_RUNG wire#w2
   // the same network as SCL:
   "OP"."PNV-4" := "AlwaysTRUE" AND ((("BUFFER"."MODE SELECTION" = 2) AND "MANUAL BIT"."PNV-4") OR (("BUFFER"."MODE SELECTION" = 1) AND ((("BUFFER".PROCESS >= 10) AND ("BUFFER".PROCESS <= 20)) OR (("BUFFER".PROCESS >= 121) AND ("BUFFER".PROCESS <= 140) AND "AlwaysFALSE") OR ("BUFFER".PROCESS = 120) OR ("BUFFER".PROCESS = 111) OR (("BUFFER".PROCESS >= 320) AND ("BUFFER".PROCESS <= 330)) OR (("BUFFER".PROCESS >= 420) AND ("BUFFER".PROCESS <= 430)) OR (("BUFFER".PROCESS >= 520) AND ("BUFFER".PROCESS <= 530)) OR (("BUFFER".PROCESS >= 700) AND ("BUFFER".PROCESS <= 730)) OR (("BUFFER".PROCESS >= 800) AND ("BUFFER".PROCESS <= 830))))) AND NOT "CYCLE PAUSE" AND NOT "ERROR";
END_REGION

REGION Network 21: "PNEUMATIC_VALVE-1" (PBFV-1) MFG1- SUGAR
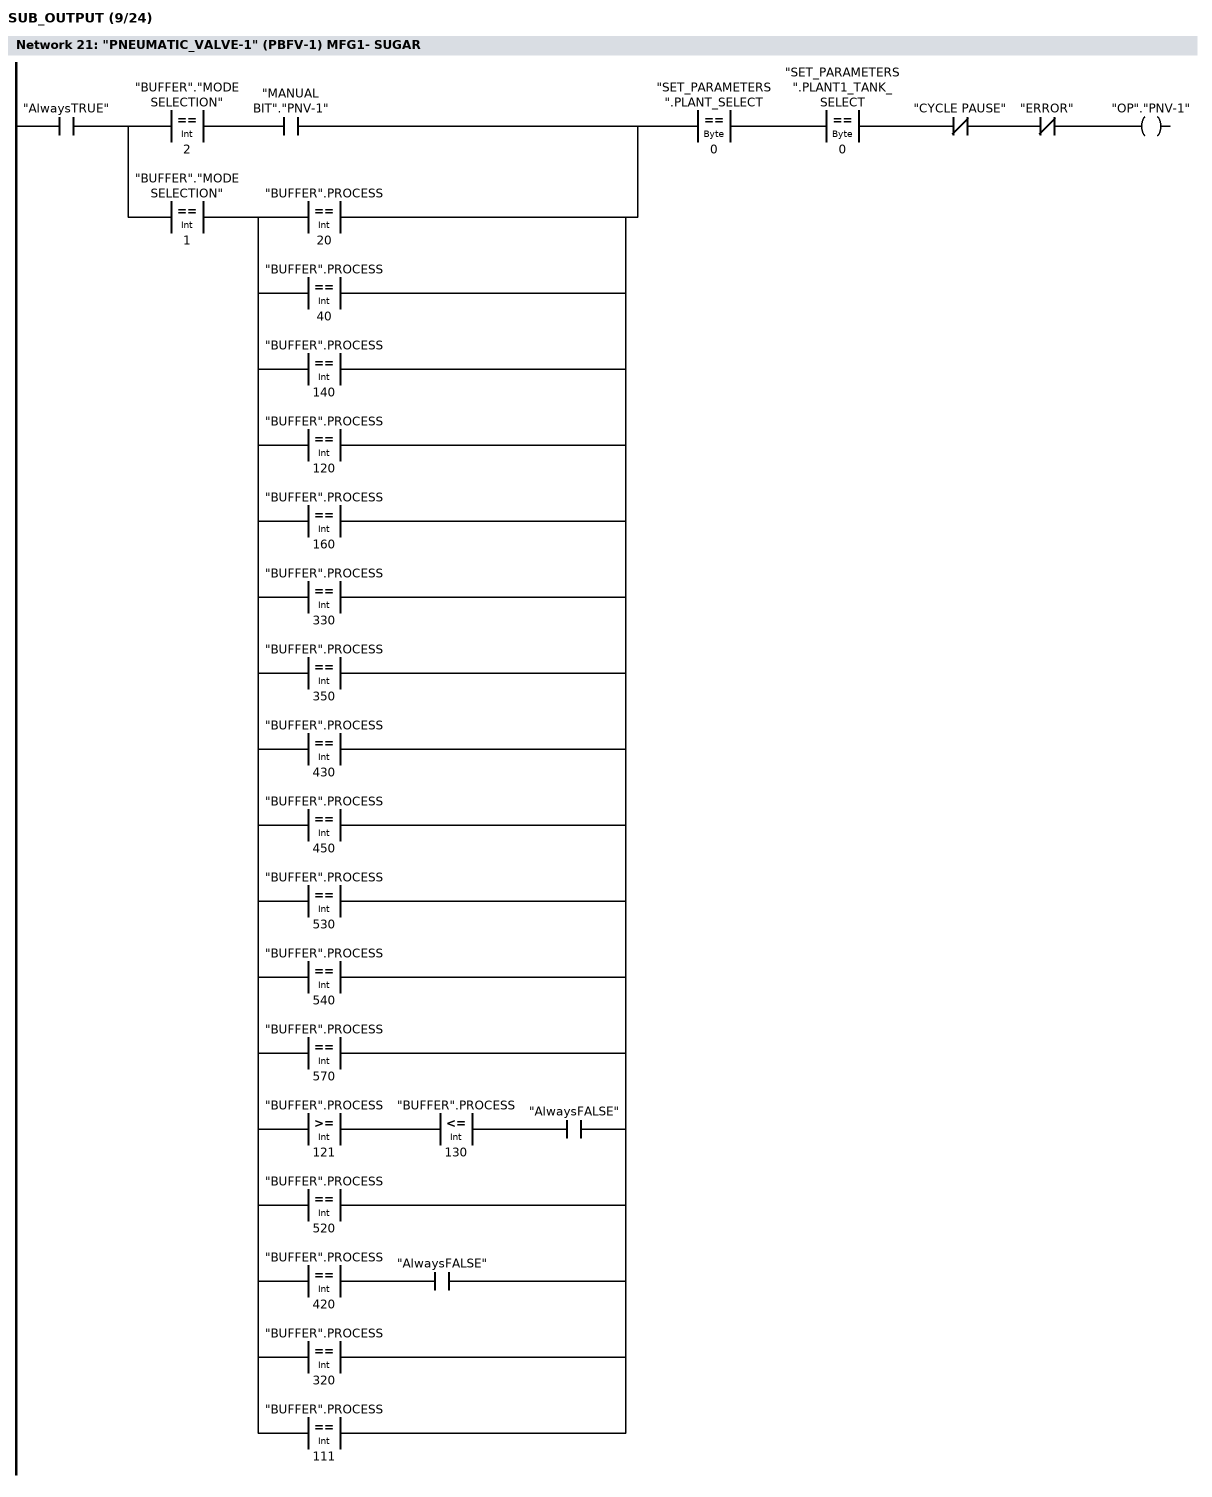
   RUNG wire#powerrail
      Contact( "AlwaysTRUE" )
      wire#w1
      { S7_Templates := "SrcType := Int" } EQ_Contact(in1 := "BUFFER"."MODE SELECTION", in2 := 2)
      Contact( "MANUAL BIT"."PNV-1" )
      wire#w2
      { S7_Templates := "SrcType := Byte" } EQ_Contact(in1 := "SET_PARAMETERS".PLANT_SELECT, in2 := 0)
      { S7_Templates := "SrcType := Byte" } EQ_Contact(in1 := "SET_PARAMETERS".PLANT1_TANK_SELECT, in2 := 0)
      I_Contact( "CYCLE PAUSE" )
      I_Contact( "ERROR" )
      Coil( "OP"."PNV-1" )
   END_RUNG
   RUNG wire#w1
      { S7_Templates := "SrcType := Int" } EQ_Contact(in1 := "BUFFER"."MODE SELECTION", in2 := 1)
      wire#w3
      { S7_Templates := "SrcType := Int" } EQ_Contact(in1 := "BUFFER".PROCESS, in2 := 20)
   END_RUNG wire#w2
   RUNG wire#w3
      { S7_Templates := "SrcType := Int" } EQ_Contact(in1 := "BUFFER".PROCESS, in2 := 40)
   END_RUNG wire#w2
   RUNG wire#w3
      { S7_Templates := "SrcType := Int" } EQ_Contact(in1 := "BUFFER".PROCESS, in2 := 140)
   END_RUNG wire#w2
   RUNG wire#w3
      { S7_Templates := "SrcType := Int" } EQ_Contact(in1 := "BUFFER".PROCESS, in2 := 120)
   END_RUNG wire#w2
   RUNG wire#w3
      { S7_Templates := "SrcType := Int" } EQ_Contact(in1 := "BUFFER".PROCESS, in2 := 160)
   END_RUNG wire#w2
   RUNG wire#w3
      { S7_Templates := "SrcType := Int" } EQ_Contact(in1 := "BUFFER".PROCESS, in2 := 330)
   END_RUNG wire#w2
   RUNG wire#w3
      { S7_Templates := "SrcType := Int" } EQ_Contact(in1 := "BUFFER".PROCESS, in2 := 350)
   END_RUNG wire#w2
   RUNG wire#w3
      { S7_Templates := "SrcType := Int" } EQ_Contact(in1 := "BUFFER".PROCESS, in2 := 430)
   END_RUNG wire#w2
   RUNG wire#w3
      { S7_Templates := "SrcType := Int" } EQ_Contact(in1 := "BUFFER".PROCESS, in2 := 450)
   END_RUNG wire#w2
   RUNG wire#w3
      { S7_Templates := "SrcType := Int" } EQ_Contact(in1 := "BUFFER".PROCESS, in2 := 530)
   END_RUNG wire#w2
   RUNG wire#w3
      { S7_Templates := "SrcType := Int" } EQ_Contact(in1 := "BUFFER".PROCESS, in2 := 540)
   END_RUNG wire#w2
   RUNG wire#w3
      { S7_Templates := "SrcType := Int" } EQ_Contact(in1 := "BUFFER".PROCESS, in2 := 570)
   END_RUNG wire#w2
   RUNG wire#w3
      { S7_Templates := "SrcType := Int" } GE_Contact(in1 := "BUFFER".PROCESS, in2 := 121)
      { S7_Templates := "SrcType := Int" } LE_Contact(in1 := "BUFFER".PROCESS, in2 := 130)
      Contact( "AlwaysFALSE" )
   END_RUNG wire#w2
   RUNG wire#w3
      { S7_Templates := "SrcType := Int" } EQ_Contact(in1 := "BUFFER".PROCESS, in2 := 520)
   END_RUNG wire#w2
   RUNG wire#w3
      { S7_Templates := "SrcType := Int" } EQ_Contact(in1 := "BUFFER".PROCESS, in2 := 420)
      Contact( "AlwaysFALSE" )
   END_RUNG wire#w2
   RUNG wire#w3
      { S7_Templates := "SrcType := Int" } EQ_Contact(in1 := "BUFFER".PROCESS, in2 := 320)
   END_RUNG wire#w2
   RUNG wire#w3
      { S7_Templates := "SrcType := Int" } EQ_Contact(in1 := "BUFFER".PROCESS, in2 := 111)
   END_RUNG wire#w2
   // the same network as SCL:
   "OP"."PNV-1" := "AlwaysTRUE" AND ((("BUFFER"."MODE SELECTION" = 2) AND "MANUAL BIT"."PNV-1") OR (("BUFFER"."MODE SELECTION" = 1) AND (("BUFFER".PROCESS = 20) OR ("BUFFER".PROCESS = 40) OR ("BUFFER".PROCESS = 140) OR ("BUFFER".PROCESS = 120) OR ("BUFFER".PROCESS = 160) OR ("BUFFER".PROCESS = 330) OR ("BUFFER".PROCESS = 350) OR ("BUFFER".PROCESS = 430) OR ("BUFFER".PROCESS = 450) OR ("BUFFER".PROCESS = 530) OR ("BUFFER".PROCESS = 540) OR ("BUFFER".PROCESS = 570) OR (("BUFFER".PROCESS >= 121) AND ("BUFFER".PROCESS <= 130) AND "AlwaysFALSE") OR ("BUFFER".PROCESS = 520) OR (("BUFFER".PROCESS = 420) AND "AlwaysFALSE") OR ("BUFFER".PROCESS = 320) OR ("BUFFER".PROCESS = 111)))) AND ("SET_PARAMETERS".PLANT_SELECT = 0) AND ("SET_PARAMETERS".PLANT1_TANK_SELECT = 0) AND NOT "CYCLE PAUSE" AND NOT "ERROR";
END_REGION

REGION Network 22: "PNEUMATIC_VALVE-2" (PBFV-2) MFG1- MFG
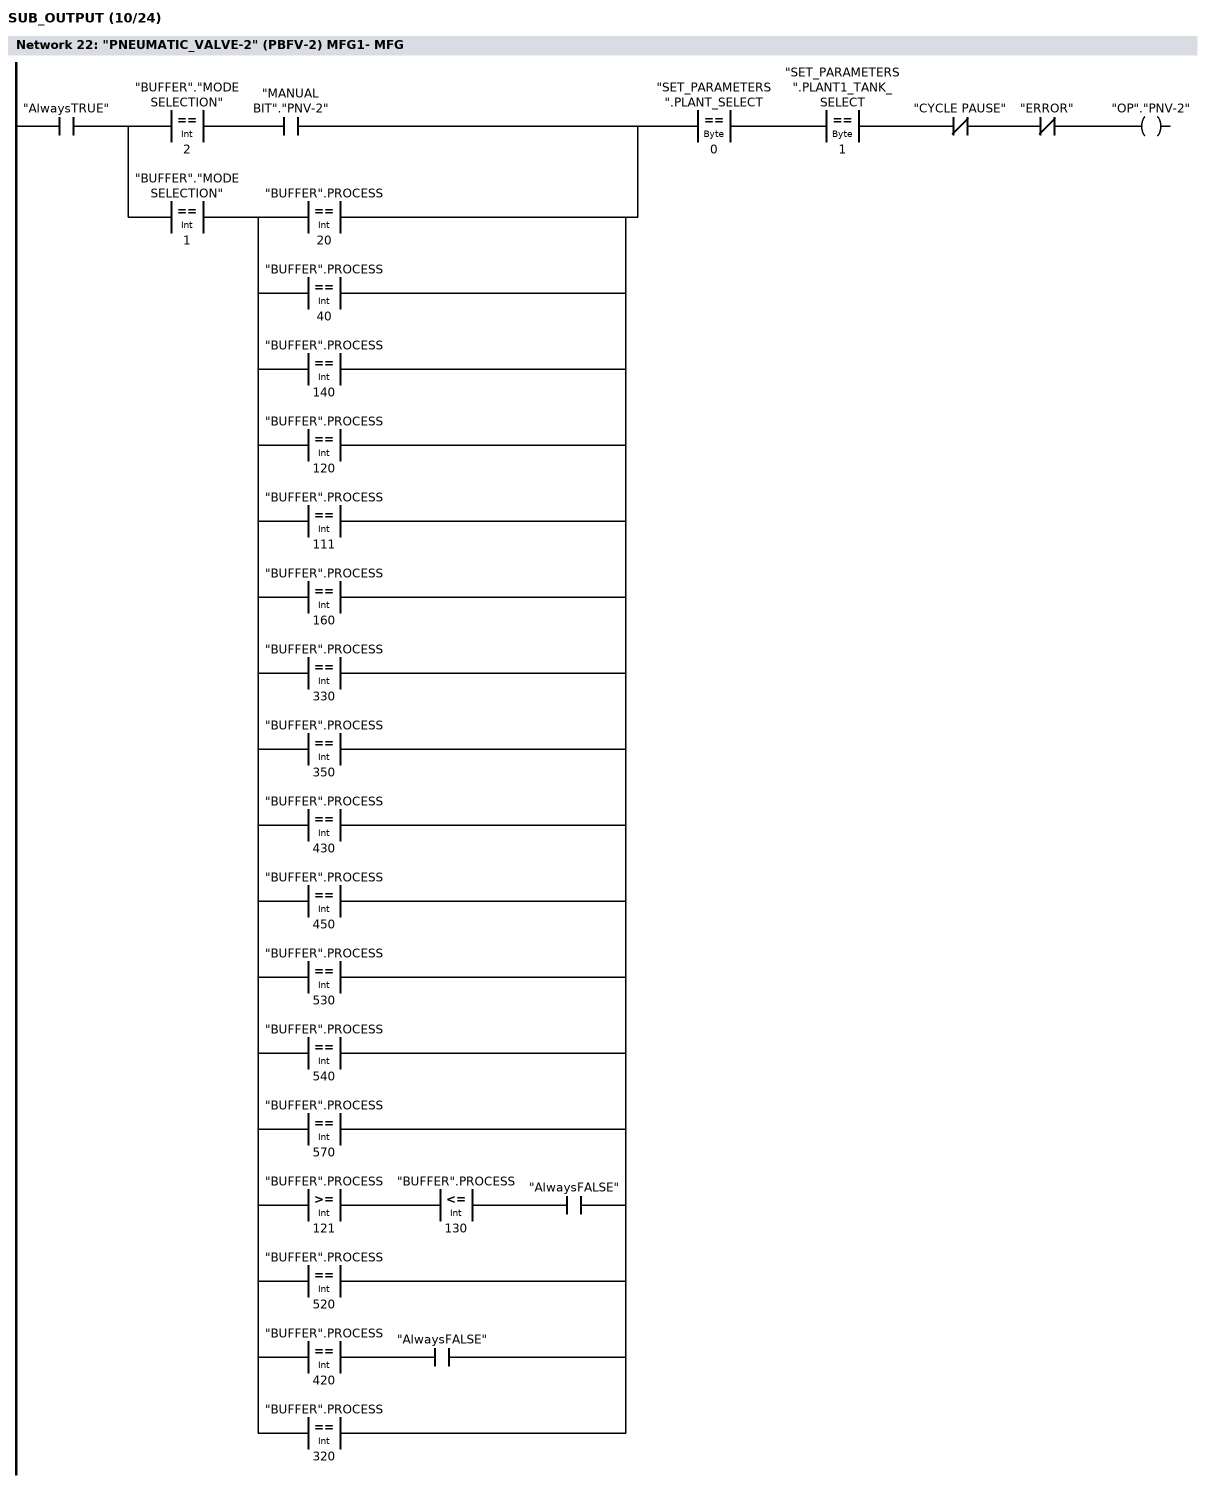
   RUNG wire#powerrail
      Contact( "AlwaysTRUE" )
      wire#w1
      { S7_Templates := "SrcType := Int" } EQ_Contact(in1 := "BUFFER"."MODE SELECTION", in2 := 2)
      Contact( "MANUAL BIT"."PNV-2" )
      wire#w2
      { S7_Templates := "SrcType := Byte" } EQ_Contact(in1 := "SET_PARAMETERS".PLANT_SELECT, in2 := 0)
      { S7_Templates := "SrcType := Byte" } EQ_Contact(in1 := "SET_PARAMETERS".PLANT1_TANK_SELECT, in2 := 1)
      I_Contact( "CYCLE PAUSE" )
      I_Contact( "ERROR" )
      Coil( "OP"."PNV-2" )
   END_RUNG
   RUNG wire#w1
      { S7_Templates := "SrcType := Int" } EQ_Contact(in1 := "BUFFER"."MODE SELECTION", in2 := 1)
      wire#w3
      { S7_Templates := "SrcType := Int" } EQ_Contact(in1 := "BUFFER".PROCESS, in2 := 20)
   END_RUNG wire#w2
   RUNG wire#w3
      { S7_Templates := "SrcType := Int" } EQ_Contact(in1 := "BUFFER".PROCESS, in2 := 40)
   END_RUNG wire#w2
   RUNG wire#w3
      { S7_Templates := "SrcType := Int" } EQ_Contact(in1 := "BUFFER".PROCESS, in2 := 140)
   END_RUNG wire#w2
   RUNG wire#w3
      { S7_Templates := "SrcType := Int" } EQ_Contact(in1 := "BUFFER".PROCESS, in2 := 120)
   END_RUNG wire#w2
   RUNG wire#w3
      { S7_Templates := "SrcType := Int" } EQ_Contact(in1 := "BUFFER".PROCESS, in2 := 111)
   END_RUNG wire#w2
   RUNG wire#w3
      { S7_Templates := "SrcType := Int" } EQ_Contact(in1 := "BUFFER".PROCESS, in2 := 160)
   END_RUNG wire#w2
   RUNG wire#w3
      { S7_Templates := "SrcType := Int" } EQ_Contact(in1 := "BUFFER".PROCESS, in2 := 330)
   END_RUNG wire#w2
   RUNG wire#w3
      { S7_Templates := "SrcType := Int" } EQ_Contact(in1 := "BUFFER".PROCESS, in2 := 350)
   END_RUNG wire#w2
   RUNG wire#w3
      { S7_Templates := "SrcType := Int" } EQ_Contact(in1 := "BUFFER".PROCESS, in2 := 430)
   END_RUNG wire#w2
   RUNG wire#w3
      { S7_Templates := "SrcType := Int" } EQ_Contact(in1 := "BUFFER".PROCESS, in2 := 450)
   END_RUNG wire#w2
   RUNG wire#w3
      { S7_Templates := "SrcType := Int" } EQ_Contact(in1 := "BUFFER".PROCESS, in2 := 530)
   END_RUNG wire#w2
   RUNG wire#w3
      { S7_Templates := "SrcType := Int" } EQ_Contact(in1 := "BUFFER".PROCESS, in2 := 540)
   END_RUNG wire#w2
   RUNG wire#w3
      { S7_Templates := "SrcType := Int" } EQ_Contact(in1 := "BUFFER".PROCESS, in2 := 570)
   END_RUNG wire#w2
   RUNG wire#w3
      { S7_Templates := "SrcType := Int" } GE_Contact(in1 := "BUFFER".PROCESS, in2 := 121)
      { S7_Templates := "SrcType := Int" } LE_Contact(in1 := "BUFFER".PROCESS, in2 := 130)
      Contact( "AlwaysFALSE" )
   END_RUNG wire#w2
   RUNG wire#w3
      { S7_Templates := "SrcType := Int" } EQ_Contact(in1 := "BUFFER".PROCESS, in2 := 520)
   END_RUNG wire#w2
   RUNG wire#w3
      { S7_Templates := "SrcType := Int" } EQ_Contact(in1 := "BUFFER".PROCESS, in2 := 420)
      Contact( "AlwaysFALSE" )
   END_RUNG wire#w2
   RUNG wire#w3
      { S7_Templates := "SrcType := Int" } EQ_Contact(in1 := "BUFFER".PROCESS, in2 := 320)
   END_RUNG wire#w2
   // the same network as SCL:
   "OP"."PNV-2" := "AlwaysTRUE" AND ((("BUFFER"."MODE SELECTION" = 2) AND "MANUAL BIT"."PNV-2") OR (("BUFFER"."MODE SELECTION" = 1) AND (("BUFFER".PROCESS = 20) OR ("BUFFER".PROCESS = 40) OR ("BUFFER".PROCESS = 140) OR ("BUFFER".PROCESS = 120) OR ("BUFFER".PROCESS = 111) OR ("BUFFER".PROCESS = 160) OR ("BUFFER".PROCESS = 330) OR ("BUFFER".PROCESS = 350) OR ("BUFFER".PROCESS = 430) OR ("BUFFER".PROCESS = 450) OR ("BUFFER".PROCESS = 530) OR ("BUFFER".PROCESS = 540) OR ("BUFFER".PROCESS = 570) OR (("BUFFER".PROCESS >= 121) AND ("BUFFER".PROCESS <= 130) AND "AlwaysFALSE") OR ("BUFFER".PROCESS = 520) OR (("BUFFER".PROCESS = 420) AND "AlwaysFALSE") OR ("BUFFER".PROCESS = 320)))) AND ("SET_PARAMETERS".PLANT_SELECT = 0) AND ("SET_PARAMETERS".PLANT1_TANK_SELECT = 1) AND NOT "CYCLE PAUSE" AND NOT "ERROR";
END_REGION

REGION Network 23: "PNEUMATIC_VALVE-6" (PBFV-6)
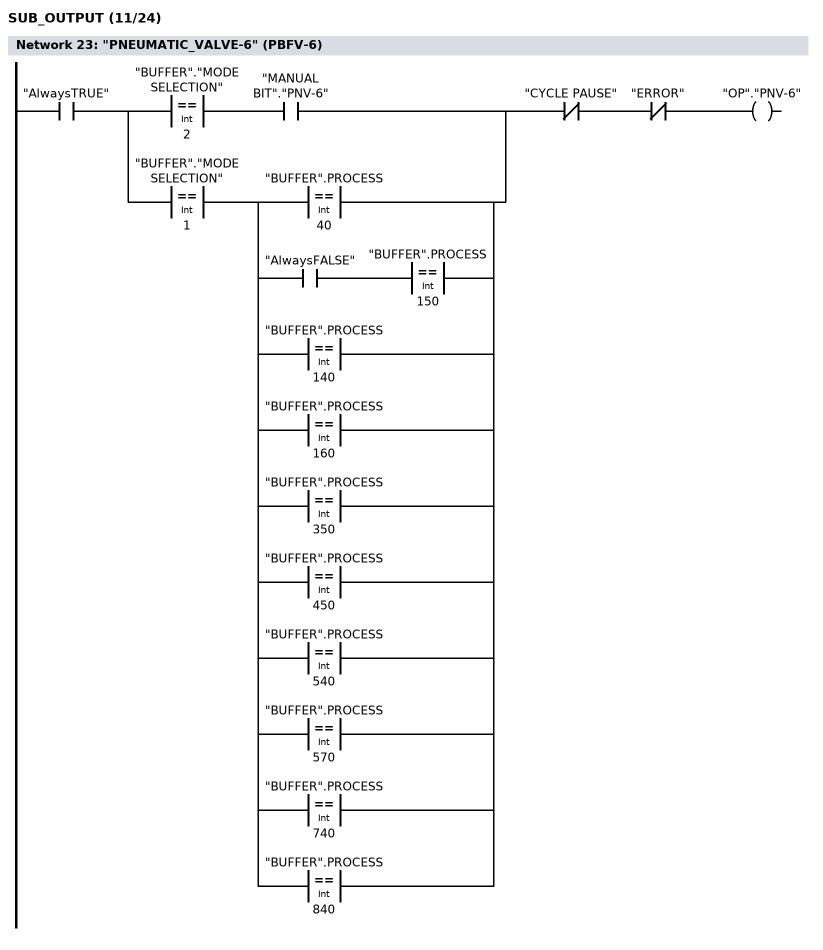
   RUNG wire#powerrail
      Contact( "AlwaysTRUE" )
      wire#w1
      { S7_Templates := "SrcType := Int" } EQ_Contact(in1 := "BUFFER"."MODE SELECTION", in2 := 2)
      Contact( "MANUAL BIT"."PNV-6" )
      wire#w2
      I_Contact( "CYCLE PAUSE" )
      I_Contact( "ERROR" )
      Coil( "OP"."PNV-6" )
   END_RUNG
   RUNG wire#w1
      { S7_Templates := "SrcType := Int" } EQ_Contact(in1 := "BUFFER"."MODE SELECTION", in2 := 1)
      wire#w3
      { S7_Templates := "SrcType := Int" } EQ_Contact(in1 := "BUFFER".PROCESS, in2 := 40)
   END_RUNG wire#w2
   RUNG wire#w3
      Contact( "AlwaysFALSE" )
      { S7_Templates := "SrcType := Int" } EQ_Contact(in1 := "BUFFER".PROCESS, in2 := 150)
   END_RUNG wire#w2
   RUNG wire#w3
      { S7_Templates := "SrcType := Int" } EQ_Contact(in1 := "BUFFER".PROCESS, in2 := 140)
   END_RUNG wire#w2
   RUNG wire#w3
      { S7_Templates := "SrcType := Int" } EQ_Contact(in1 := "BUFFER".PROCESS, in2 := 160)
   END_RUNG wire#w2
   RUNG wire#w3
      { S7_Templates := "SrcType := Int" } EQ_Contact(in1 := "BUFFER".PROCESS, in2 := 350)
   END_RUNG wire#w2
   RUNG wire#w3
      { S7_Templates := "SrcType := Int" } EQ_Contact(in1 := "BUFFER".PROCESS, in2 := 450)
   END_RUNG wire#w2
   RUNG wire#w3
      { S7_Templates := "SrcType := Int" } EQ_Contact(in1 := "BUFFER".PROCESS, in2 := 540)
   END_RUNG wire#w2
   RUNG wire#w3
      { S7_Templates := "SrcType := Int" } EQ_Contact(in1 := "BUFFER".PROCESS, in2 := 570)
   END_RUNG wire#w2
   RUNG wire#w3
      { S7_Templates := "SrcType := Int" } EQ_Contact(in1 := "BUFFER".PROCESS, in2 := 740)
   END_RUNG wire#w2
   RUNG wire#w3
      { S7_Templates := "SrcType := Int" } EQ_Contact(in1 := "BUFFER".PROCESS, in2 := 840)
   END_RUNG wire#w2
   // the same network as SCL:
   "OP"."PNV-6" := "AlwaysTRUE" AND ((("BUFFER"."MODE SELECTION" = 2) AND "MANUAL BIT"."PNV-6") OR (("BUFFER"."MODE SELECTION" = 1) AND (("BUFFER".PROCESS = 40) OR ("AlwaysFALSE" AND ("BUFFER".PROCESS = 150)) OR ("BUFFER".PROCESS = 140) OR ("BUFFER".PROCESS = 160) OR ("BUFFER".PROCESS = 350) OR ("BUFFER".PROCESS = 450) OR ("BUFFER".PROCESS = 540) OR ("BUFFER".PROCESS = 570) OR ("BUFFER".PROCESS = 740) OR ("BUFFER".PROCESS = 840)))) AND NOT "CYCLE PAUSE" AND NOT "ERROR";
END_REGION

REGION Network 24: "PNEUMATIC_VALVE-7" (PBFV-7) SWT RECIRCULATION
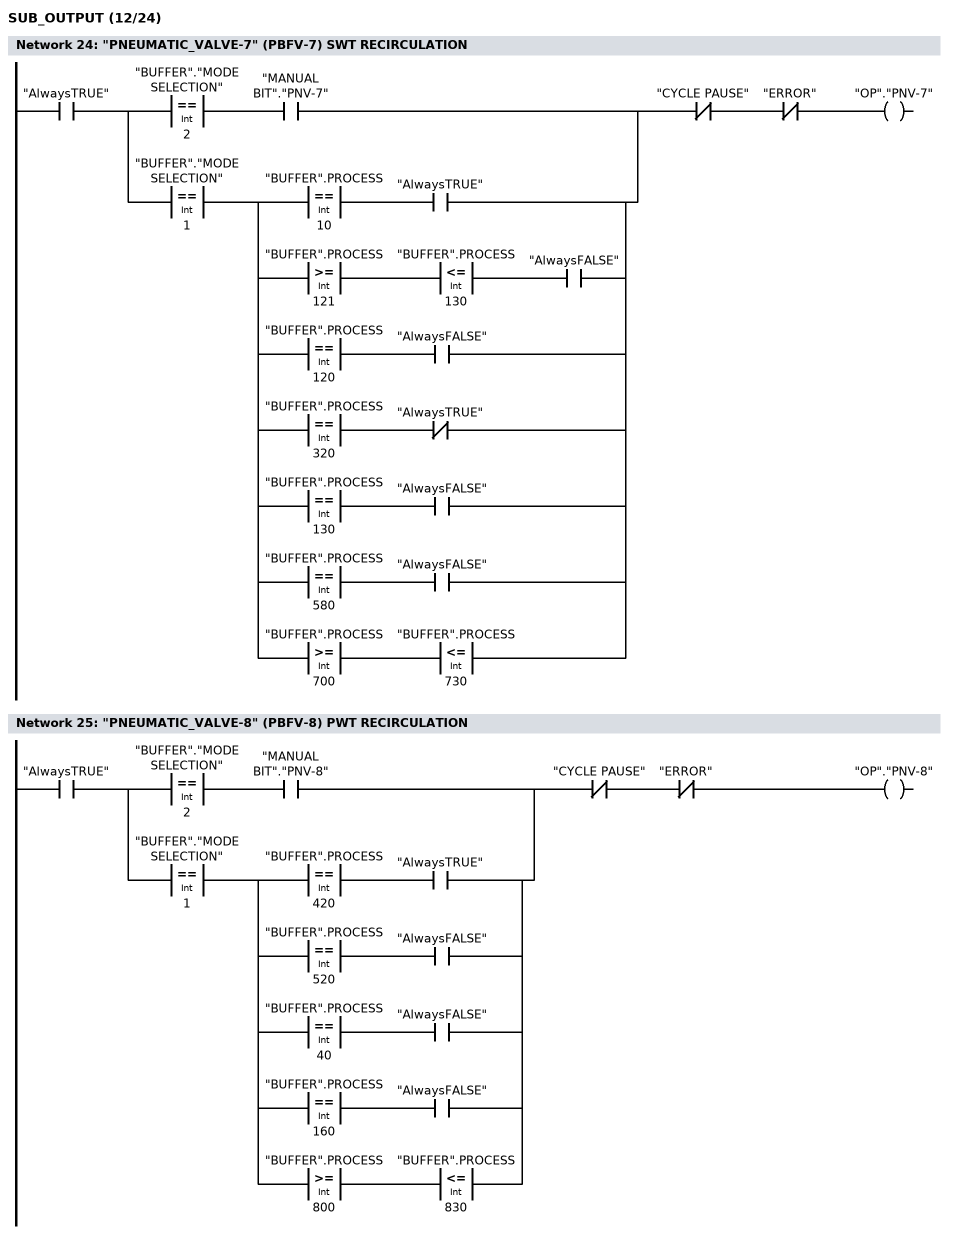
   RUNG wire#powerrail
      Contact( "AlwaysTRUE" )
      wire#w1
      { S7_Templates := "SrcType := Int" } EQ_Contact(in1 := "BUFFER"."MODE SELECTION", in2 := 2)
      Contact( "MANUAL BIT"."PNV-7" )
      wire#w2
      I_Contact( "CYCLE PAUSE" )
      I_Contact( "ERROR" )
      Coil( "OP"."PNV-7" )
   END_RUNG
   RUNG wire#w1
      { S7_Templates := "SrcType := Int" } EQ_Contact(in1 := "BUFFER"."MODE SELECTION", in2 := 1)
      wire#w3
      { S7_Templates := "SrcType := Int" } EQ_Contact(in1 := "BUFFER".PROCESS, in2 := 10)
      Contact( "AlwaysTRUE" )
   END_RUNG wire#w2
   RUNG wire#w3
      { S7_Templates := "SrcType := Int" } GE_Contact(in1 := "BUFFER".PROCESS, in2 := 121)
      { S7_Templates := "SrcType := Int" } LE_Contact(in1 := "BUFFER".PROCESS, in2 := 130)
      Contact( "AlwaysFALSE" )
   END_RUNG wire#w2
   RUNG wire#w3
      { S7_Templates := "SrcType := Int" } EQ_Contact(in1 := "BUFFER".PROCESS, in2 := 120)
      Contact( "AlwaysFALSE" )
   END_RUNG wire#w2
   RUNG wire#w3
      { S7_Templates := "SrcType := Int" } EQ_Contact(in1 := "BUFFER".PROCESS, in2 := 320)
      I_Contact( "AlwaysTRUE" )
   END_RUNG wire#w2
   RUNG wire#w3
      { S7_Templates := "SrcType := Int" } EQ_Contact(in1 := "BUFFER".PROCESS, in2 := 130)
      Contact( "AlwaysFALSE" )
   END_RUNG wire#w2
   RUNG wire#w3
      { S7_Templates := "SrcType := Int" } EQ_Contact(in1 := "BUFFER".PROCESS, in2 := 580)
      Contact( "AlwaysFALSE" )
   END_RUNG wire#w2
   RUNG wire#w3
      { S7_Templates := "SrcType := Int" } GE_Contact(in1 := "BUFFER".PROCESS, in2 := 700)
      { S7_Templates := "SrcType := Int" } LE_Contact(in1 := "BUFFER".PROCESS, in2 := 730)
   END_RUNG wire#w2
   // the same network as SCL:
   "OP"."PNV-7" := "AlwaysTRUE" AND ((("BUFFER"."MODE SELECTION" = 2) AND "MANUAL BIT"."PNV-7") OR (("BUFFER"."MODE SELECTION" = 1) AND ((("BUFFER".PROCESS = 10) AND "AlwaysTRUE") OR (("BUFFER".PROCESS >= 121) AND ("BUFFER".PROCESS <= 130) AND "AlwaysFALSE") OR (("BUFFER".PROCESS = 120) AND "AlwaysFALSE") OR (("BUFFER".PROCESS = 320) AND NOT "AlwaysTRUE") OR (("BUFFER".PROCESS = 130) AND "AlwaysFALSE") OR (("BUFFER".PROCESS = 580) AND "AlwaysFALSE") OR (("BUFFER".PROCESS >= 700) AND ("BUFFER".PROCESS <= 730))))) AND NOT "CYCLE PAUSE" AND NOT "ERROR";
END_REGION

REGION Network 25: "PNEUMATIC_VALVE-8" (PBFV-8) PWT RECIRCULATION
   RUNG wire#powerrail
      Contact( "AlwaysTRUE" )
      wire#w1
      { S7_Templates := "SrcType := Int" } EQ_Contact(in1 := "BUFFER"."MODE SELECTION", in2 := 2)
      Contact( "MANUAL BIT"."PNV-8" )
      wire#w2
      I_Contact( "CYCLE PAUSE" )
      I_Contact( "ERROR" )
      Coil( "OP"."PNV-8" )
   END_RUNG
   RUNG wire#w1
      { S7_Templates := "SrcType := Int" } EQ_Contact(in1 := "BUFFER"."MODE SELECTION", in2 := 1)
      wire#w3
      { S7_Templates := "SrcType := Int" } EQ_Contact(in1 := "BUFFER".PROCESS, in2 := 420)
      Contact( "AlwaysTRUE" )
   END_RUNG wire#w2
   RUNG wire#w3
      { S7_Templates := "SrcType := Int" } EQ_Contact(in1 := "BUFFER".PROCESS, in2 := 520)
      Contact( "AlwaysFALSE" )
   END_RUNG wire#w2
   RUNG wire#w3
      { S7_Templates := "SrcType := Int" } EQ_Contact(in1 := "BUFFER".PROCESS, in2 := 40)
      Contact( "AlwaysFALSE" )
   END_RUNG wire#w2
   RUNG wire#w3
      { S7_Templates := "SrcType := Int" } EQ_Contact(in1 := "BUFFER".PROCESS, in2 := 160)
      Contact( "AlwaysFALSE" )
   END_RUNG wire#w2
   RUNG wire#w3
      { S7_Templates := "SrcType := Int" } GE_Contact(in1 := "BUFFER".PROCESS, in2 := 800)
      { S7_Templates := "SrcType := Int" } LE_Contact(in1 := "BUFFER".PROCESS, in2 := 830)
   END_RUNG wire#w2
   // the same network as SCL:
   "OP"."PNV-8" := "AlwaysTRUE" AND ((("BUFFER"."MODE SELECTION" = 2) AND "MANUAL BIT"."PNV-8") OR (("BUFFER"."MODE SELECTION" = 1) AND ((("BUFFER".PROCESS = 420) AND "AlwaysTRUE") OR (("BUFFER".PROCESS = 520) AND "AlwaysFALSE") OR (("BUFFER".PROCESS = 40) AND "AlwaysFALSE") OR (("BUFFER".PROCESS = 160) AND "AlwaysFALSE") OR (("BUFFER".PROCESS >= 800) AND ("BUFFER".PROCESS <= 830))))) AND NOT "CYCLE PAUSE" AND NOT "ERROR";
END_REGION

REGION Network 26: "PNEUMATIC_VALVE-9" (PBFV-9) MFG-1 - STORAGE1
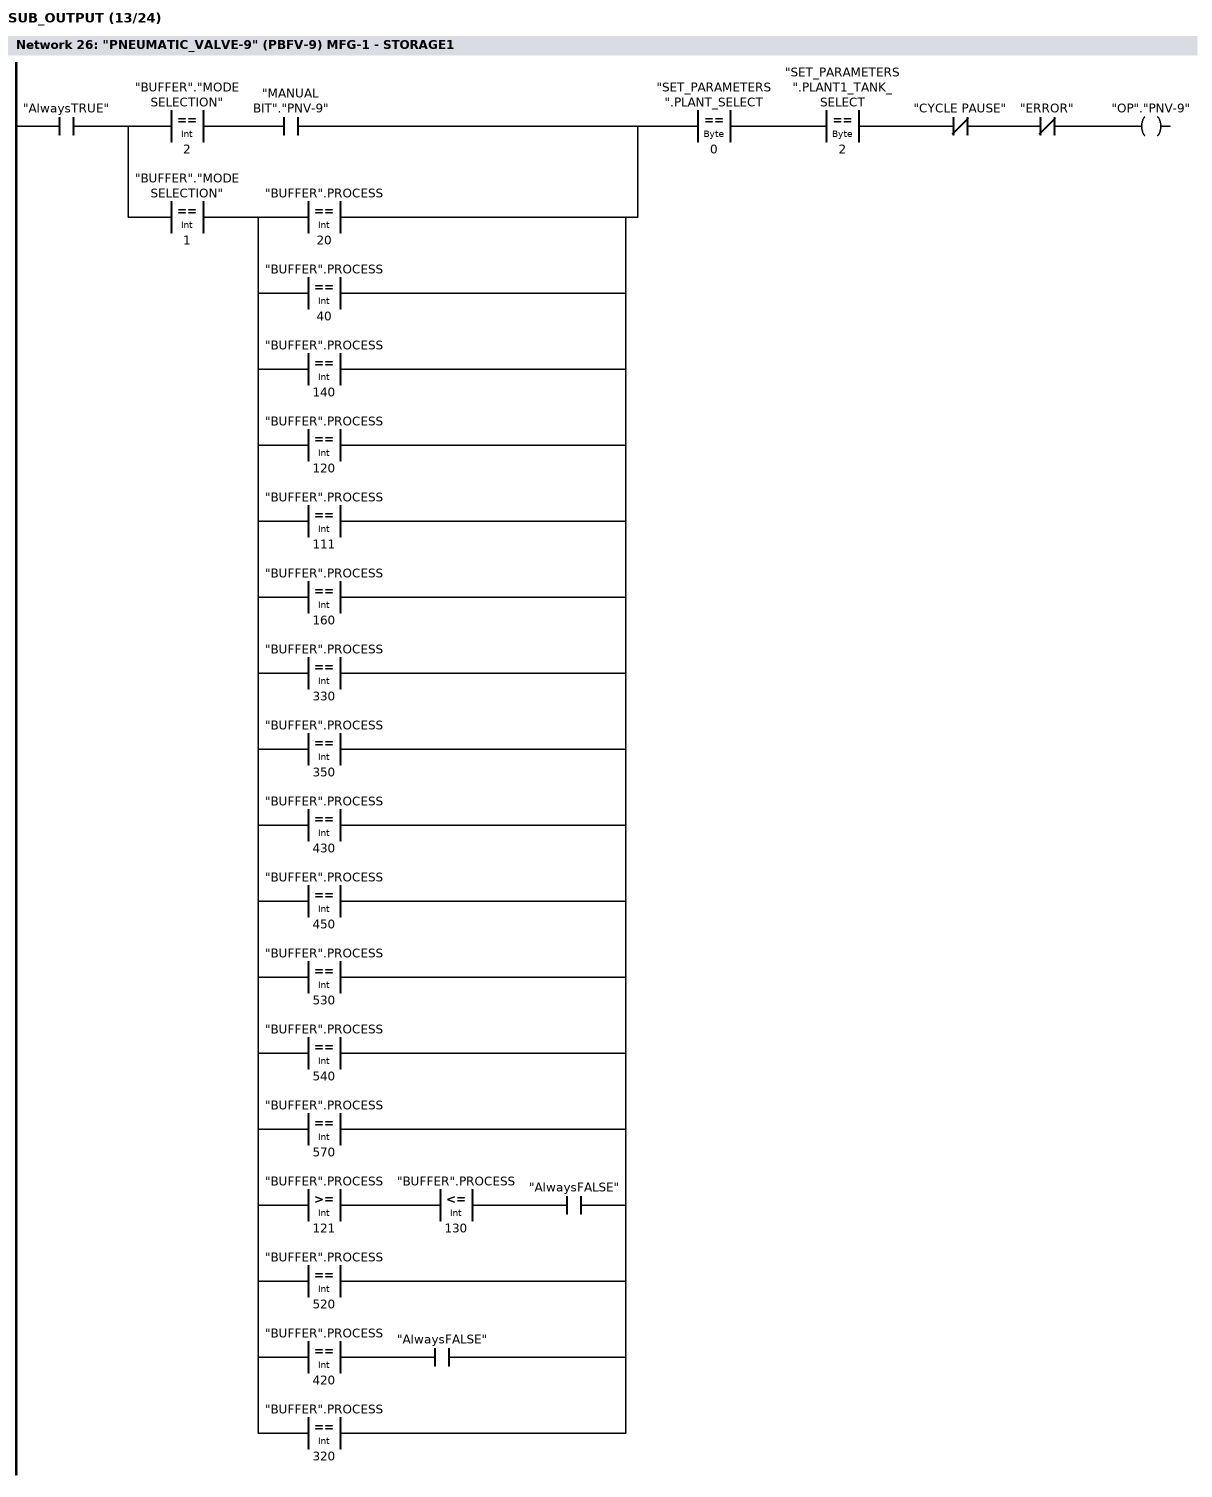
   RUNG wire#powerrail
      Contact( "AlwaysTRUE" )
      wire#w1
      { S7_Templates := "SrcType := Int" } EQ_Contact(in1 := "BUFFER"."MODE SELECTION", in2 := 2)
      Contact( "MANUAL BIT"."PNV-9" )
      wire#w2
      { S7_Templates := "SrcType := Byte" } EQ_Contact(in1 := "SET_PARAMETERS".PLANT_SELECT, in2 := 0)
      { S7_Templates := "SrcType := Byte" } EQ_Contact(in1 := "SET_PARAMETERS".PLANT1_TANK_SELECT, in2 := 2)
      I_Contact( "CYCLE PAUSE" )
      I_Contact( "ERROR" )
      Coil( "OP"."PNV-9" )
   END_RUNG
   RUNG wire#w1
      { S7_Templates := "SrcType := Int" } EQ_Contact(in1 := "BUFFER"."MODE SELECTION", in2 := 1)
      wire#w3
      { S7_Templates := "SrcType := Int" } EQ_Contact(in1 := "BUFFER".PROCESS, in2 := 20)
   END_RUNG wire#w2
   RUNG wire#w3
      { S7_Templates := "SrcType := Int" } EQ_Contact(in1 := "BUFFER".PROCESS, in2 := 40)
   END_RUNG wire#w2
   RUNG wire#w3
      { S7_Templates := "SrcType := Int" } EQ_Contact(in1 := "BUFFER".PROCESS, in2 := 140)
   END_RUNG wire#w2
   RUNG wire#w3
      { S7_Templates := "SrcType := Int" } EQ_Contact(in1 := "BUFFER".PROCESS, in2 := 120)
   END_RUNG wire#w2
   RUNG wire#w3
      { S7_Templates := "SrcType := Int" } EQ_Contact(in1 := "BUFFER".PROCESS, in2 := 111)
   END_RUNG wire#w2
   RUNG wire#w3
      { S7_Templates := "SrcType := Int" } EQ_Contact(in1 := "BUFFER".PROCESS, in2 := 160)
   END_RUNG wire#w2
   RUNG wire#w3
      { S7_Templates := "SrcType := Int" } EQ_Contact(in1 := "BUFFER".PROCESS, in2 := 330)
   END_RUNG wire#w2
   RUNG wire#w3
      { S7_Templates := "SrcType := Int" } EQ_Contact(in1 := "BUFFER".PROCESS, in2 := 350)
   END_RUNG wire#w2
   RUNG wire#w3
      { S7_Templates := "SrcType := Int" } EQ_Contact(in1 := "BUFFER".PROCESS, in2 := 430)
   END_RUNG wire#w2
   RUNG wire#w3
      { S7_Templates := "SrcType := Int" } EQ_Contact(in1 := "BUFFER".PROCESS, in2 := 450)
   END_RUNG wire#w2
   RUNG wire#w3
      { S7_Templates := "SrcType := Int" } EQ_Contact(in1 := "BUFFER".PROCESS, in2 := 530)
   END_RUNG wire#w2
   RUNG wire#w3
      { S7_Templates := "SrcType := Int" } EQ_Contact(in1 := "BUFFER".PROCESS, in2 := 540)
   END_RUNG wire#w2
   RUNG wire#w3
      { S7_Templates := "SrcType := Int" } EQ_Contact(in1 := "BUFFER".PROCESS, in2 := 570)
   END_RUNG wire#w2
   RUNG wire#w3
      { S7_Templates := "SrcType := Int" } GE_Contact(in1 := "BUFFER".PROCESS, in2 := 121)
      { S7_Templates := "SrcType := Int" } LE_Contact(in1 := "BUFFER".PROCESS, in2 := 130)
      Contact( "AlwaysFALSE" )
   END_RUNG wire#w2
   RUNG wire#w3
      { S7_Templates := "SrcType := Int" } EQ_Contact(in1 := "BUFFER".PROCESS, in2 := 520)
   END_RUNG wire#w2
   RUNG wire#w3
      { S7_Templates := "SrcType := Int" } EQ_Contact(in1 := "BUFFER".PROCESS, in2 := 420)
      Contact( "AlwaysFALSE" )
   END_RUNG wire#w2
   RUNG wire#w3
      { S7_Templates := "SrcType := Int" } EQ_Contact(in1 := "BUFFER".PROCESS, in2 := 320)
   END_RUNG wire#w2
   // the same network as SCL:
   "OP"."PNV-9" := "AlwaysTRUE" AND ((("BUFFER"."MODE SELECTION" = 2) AND "MANUAL BIT"."PNV-9") OR (("BUFFER"."MODE SELECTION" = 1) AND (("BUFFER".PROCESS = 20) OR ("BUFFER".PROCESS = 40) OR ("BUFFER".PROCESS = 140) OR ("BUFFER".PROCESS = 120) OR ("BUFFER".PROCESS = 111) OR ("BUFFER".PROCESS = 160) OR ("BUFFER".PROCESS = 330) OR ("BUFFER".PROCESS = 350) OR ("BUFFER".PROCESS = 430) OR ("BUFFER".PROCESS = 450) OR ("BUFFER".PROCESS = 530) OR ("BUFFER".PROCESS = 540) OR ("BUFFER".PROCESS = 570) OR (("BUFFER".PROCESS >= 121) AND ("BUFFER".PROCESS <= 130) AND "AlwaysFALSE") OR ("BUFFER".PROCESS = 520) OR (("BUFFER".PROCESS = 420) AND "AlwaysFALSE") OR ("BUFFER".PROCESS = 320)))) AND ("SET_PARAMETERS".PLANT_SELECT = 0) AND ("SET_PARAMETERS".PLANT1_TANK_SELECT = 2) AND NOT "CYCLE PAUSE" AND NOT "ERROR";
END_REGION

REGION Network 27: "PNEUMATIC_VALVE-10" (PBFV-10) MFG1- STORAGE2
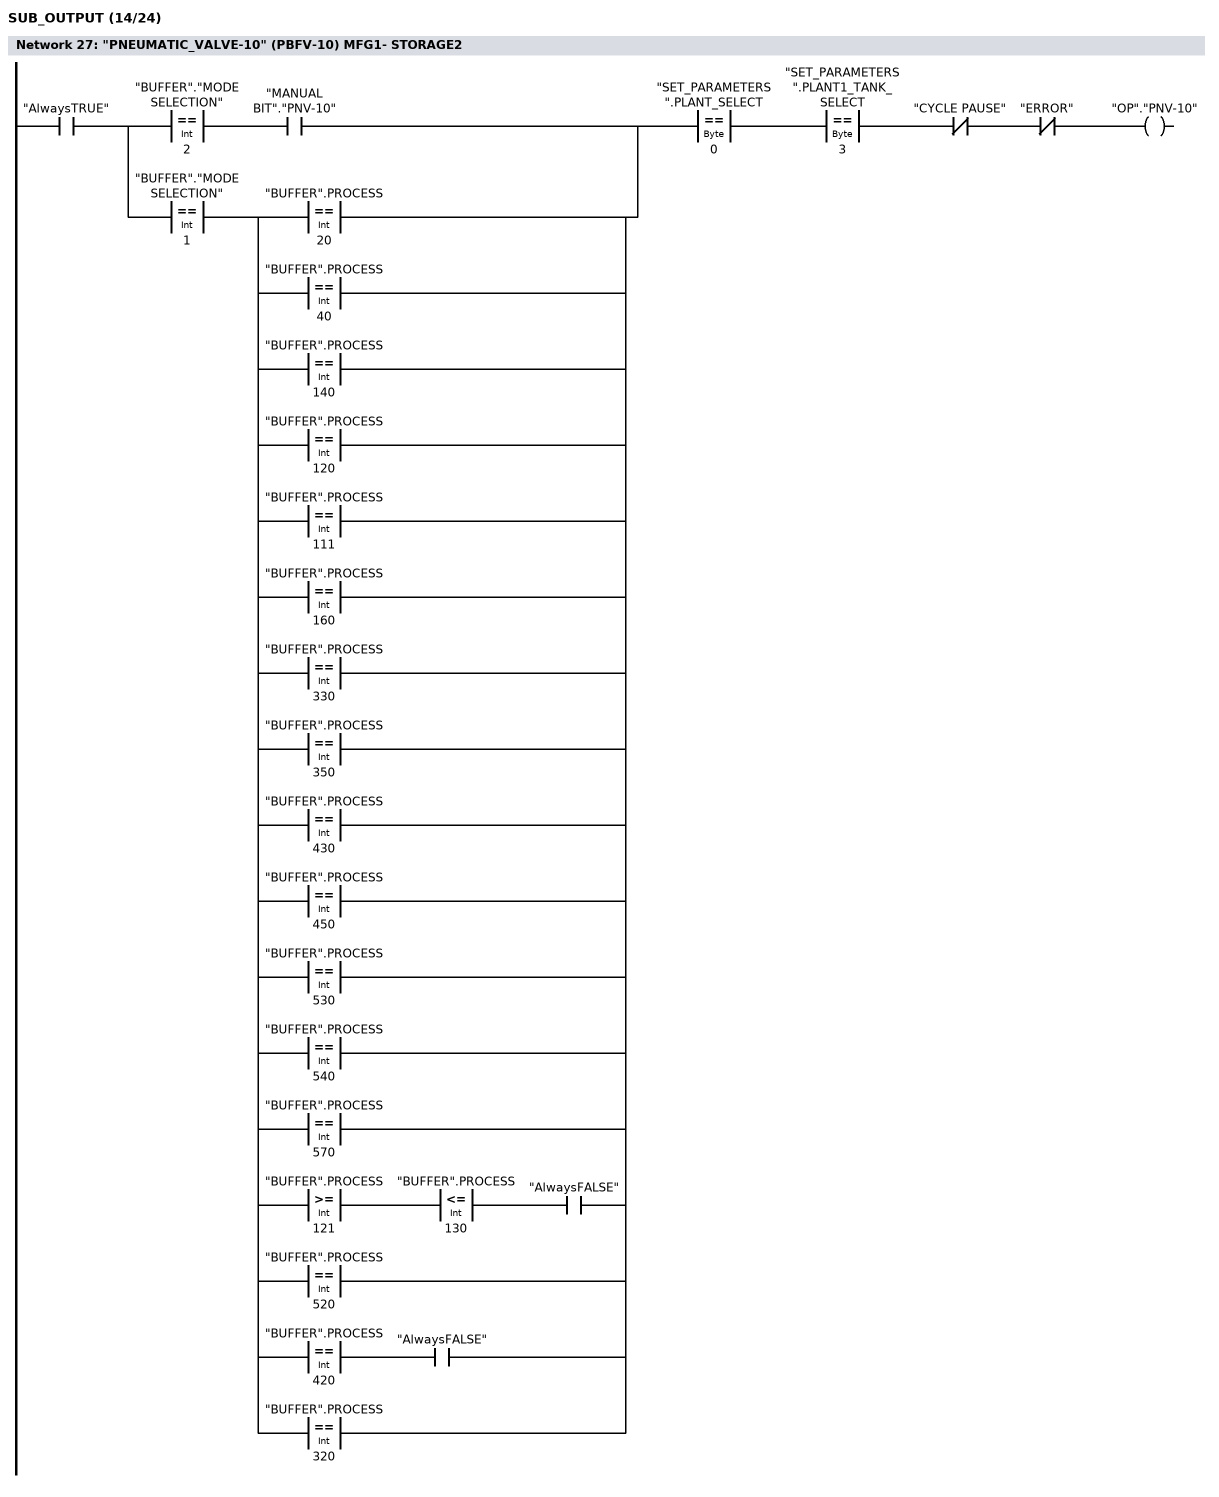
   RUNG wire#powerrail
      Contact( "AlwaysTRUE" )
      wire#w1
      { S7_Templates := "SrcType := Int" } EQ_Contact(in1 := "BUFFER"."MODE SELECTION", in2 := 2)
      Contact( "MANUAL BIT"."PNV-10" )
      wire#w2
      { S7_Templates := "SrcType := Byte" } EQ_Contact(in1 := "SET_PARAMETERS".PLANT_SELECT, in2 := 0)
      { S7_Templates := "SrcType := Byte" } EQ_Contact(in1 := "SET_PARAMETERS".PLANT1_TANK_SELECT, in2 := 3)
      I_Contact( "CYCLE PAUSE" )
      I_Contact( "ERROR" )
      Coil( "OP"."PNV-10" )
   END_RUNG
   RUNG wire#w1
      { S7_Templates := "SrcType := Int" } EQ_Contact(in1 := "BUFFER"."MODE SELECTION", in2 := 1)
      wire#w3
      { S7_Templates := "SrcType := Int" } EQ_Contact(in1 := "BUFFER".PROCESS, in2 := 20)
   END_RUNG wire#w2
   RUNG wire#w3
      { S7_Templates := "SrcType := Int" } EQ_Contact(in1 := "BUFFER".PROCESS, in2 := 40)
   END_RUNG wire#w2
   RUNG wire#w3
      { S7_Templates := "SrcType := Int" } EQ_Contact(in1 := "BUFFER".PROCESS, in2 := 140)
   END_RUNG wire#w2
   RUNG wire#w3
      { S7_Templates := "SrcType := Int" } EQ_Contact(in1 := "BUFFER".PROCESS, in2 := 120)
   END_RUNG wire#w2
   RUNG wire#w3
      { S7_Templates := "SrcType := Int" } EQ_Contact(in1 := "BUFFER".PROCESS, in2 := 111)
   END_RUNG wire#w2
   RUNG wire#w3
      { S7_Templates := "SrcType := Int" } EQ_Contact(in1 := "BUFFER".PROCESS, in2 := 160)
   END_RUNG wire#w2
   RUNG wire#w3
      { S7_Templates := "SrcType := Int" } EQ_Contact(in1 := "BUFFER".PROCESS, in2 := 330)
   END_RUNG wire#w2
   RUNG wire#w3
      { S7_Templates := "SrcType := Int" } EQ_Contact(in1 := "BUFFER".PROCESS, in2 := 350)
   END_RUNG wire#w2
   RUNG wire#w3
      { S7_Templates := "SrcType := Int" } EQ_Contact(in1 := "BUFFER".PROCESS, in2 := 430)
   END_RUNG wire#w2
   RUNG wire#w3
      { S7_Templates := "SrcType := Int" } EQ_Contact(in1 := "BUFFER".PROCESS, in2 := 450)
   END_RUNG wire#w2
   RUNG wire#w3
      { S7_Templates := "SrcType := Int" } EQ_Contact(in1 := "BUFFER".PROCESS, in2 := 530)
   END_RUNG wire#w2
   RUNG wire#w3
      { S7_Templates := "SrcType := Int" } EQ_Contact(in1 := "BUFFER".PROCESS, in2 := 540)
   END_RUNG wire#w2
   RUNG wire#w3
      { S7_Templates := "SrcType := Int" } EQ_Contact(in1 := "BUFFER".PROCESS, in2 := 570)
   END_RUNG wire#w2
   RUNG wire#w3
      { S7_Templates := "SrcType := Int" } GE_Contact(in1 := "BUFFER".PROCESS, in2 := 121)
      { S7_Templates := "SrcType := Int" } LE_Contact(in1 := "BUFFER".PROCESS, in2 := 130)
      Contact( "AlwaysFALSE" )
   END_RUNG wire#w2
   RUNG wire#w3
      { S7_Templates := "SrcType := Int" } EQ_Contact(in1 := "BUFFER".PROCESS, in2 := 520)
   END_RUNG wire#w2
   RUNG wire#w3
      { S7_Templates := "SrcType := Int" } EQ_Contact(in1 := "BUFFER".PROCESS, in2 := 420)
      Contact( "AlwaysFALSE" )
   END_RUNG wire#w2
   RUNG wire#w3
      { S7_Templates := "SrcType := Int" } EQ_Contact(in1 := "BUFFER".PROCESS, in2 := 320)
   END_RUNG wire#w2
   // the same network as SCL:
   "OP"."PNV-10" := "AlwaysTRUE" AND ((("BUFFER"."MODE SELECTION" = 2) AND "MANUAL BIT"."PNV-10") OR (("BUFFER"."MODE SELECTION" = 1) AND (("BUFFER".PROCESS = 20) OR ("BUFFER".PROCESS = 40) OR ("BUFFER".PROCESS = 140) OR ("BUFFER".PROCESS = 120) OR ("BUFFER".PROCESS = 111) OR ("BUFFER".PROCESS = 160) OR ("BUFFER".PROCESS = 330) OR ("BUFFER".PROCESS = 350) OR ("BUFFER".PROCESS = 430) OR ("BUFFER".PROCESS = 450) OR ("BUFFER".PROCESS = 530) OR ("BUFFER".PROCESS = 540) OR ("BUFFER".PROCESS = 570) OR (("BUFFER".PROCESS >= 121) AND ("BUFFER".PROCESS <= 130) AND "AlwaysFALSE") OR ("BUFFER".PROCESS = 520) OR (("BUFFER".PROCESS = 420) AND "AlwaysFALSE") OR ("BUFFER".PROCESS = 320)))) AND ("SET_PARAMETERS".PLANT_SELECT = 0) AND ("SET_PARAMETERS".PLANT1_TANK_SELECT = 3) AND NOT "CYCLE PAUSE" AND NOT "ERROR";
END_REGION

REGION Network 28: "PNEUMATIC_VALVE-11" (PBFV-11)
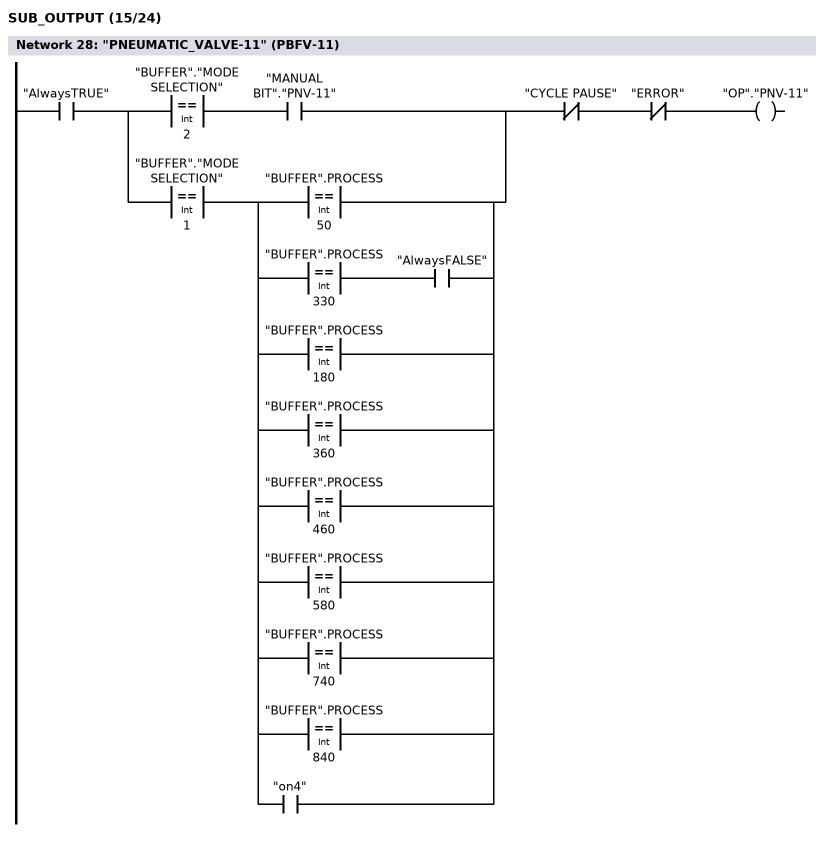
   RUNG wire#powerrail
      Contact( "AlwaysTRUE" )
      wire#w1
      { S7_Templates := "SrcType := Int" } EQ_Contact(in1 := "BUFFER"."MODE SELECTION", in2 := 2)
      Contact( "MANUAL BIT"."PNV-11" )
      wire#w2
      I_Contact( "CYCLE PAUSE" )
      I_Contact( "ERROR" )
      Coil( "OP"."PNV-11" )
   END_RUNG
   RUNG wire#w1
      { S7_Templates := "SrcType := Int" } EQ_Contact(in1 := "BUFFER"."MODE SELECTION", in2 := 1)
      wire#w3
      { S7_Templates := "SrcType := Int" } EQ_Contact(in1 := "BUFFER".PROCESS, in2 := 50)
   END_RUNG wire#w2
   RUNG wire#w3
      { S7_Templates := "SrcType := Int" } EQ_Contact(in1 := "BUFFER".PROCESS, in2 := 330)
      Contact( "AlwaysFALSE" )
   END_RUNG wire#w2
   RUNG wire#w3
      { S7_Templates := "SrcType := Int" } EQ_Contact(in1 := "BUFFER".PROCESS, in2 := 180)
   END_RUNG wire#w2
   RUNG wire#w3
      { S7_Templates := "SrcType := Int" } EQ_Contact(in1 := "BUFFER".PROCESS, in2 := 360)
   END_RUNG wire#w2
   RUNG wire#w3
      { S7_Templates := "SrcType := Int" } EQ_Contact(in1 := "BUFFER".PROCESS, in2 := 460)
   END_RUNG wire#w2
   RUNG wire#w3
      { S7_Templates := "SrcType := Int" } EQ_Contact(in1 := "BUFFER".PROCESS, in2 := 580)
   END_RUNG wire#w2
   RUNG wire#w3
      { S7_Templates := "SrcType := Int" } EQ_Contact(in1 := "BUFFER".PROCESS, in2 := 740)
   END_RUNG wire#w2
   RUNG wire#w3
      { S7_Templates := "SrcType := Int" } EQ_Contact(in1 := "BUFFER".PROCESS, in2 := 840)
   END_RUNG wire#w2
   RUNG wire#w3
      Contact( "on4" )
   END_RUNG wire#w2
   // the same network as SCL:
   "OP"."PNV-11" := "AlwaysTRUE" AND ((("BUFFER"."MODE SELECTION" = 2) AND "MANUAL BIT"."PNV-11") OR (("BUFFER"."MODE SELECTION" = 1) AND (("BUFFER".PROCESS = 50) OR (("BUFFER".PROCESS = 330) AND "AlwaysFALSE") OR ("BUFFER".PROCESS = 180) OR ("BUFFER".PROCESS = 360) OR ("BUFFER".PROCESS = 460) OR ("BUFFER".PROCESS = 580) OR ("BUFFER".PROCESS = 740) OR ("BUFFER".PROCESS = 840) OR "on4"))) AND NOT "CYCLE PAUSE" AND NOT "ERROR";
END_REGION

REGION Network 29: (PBFV-12)
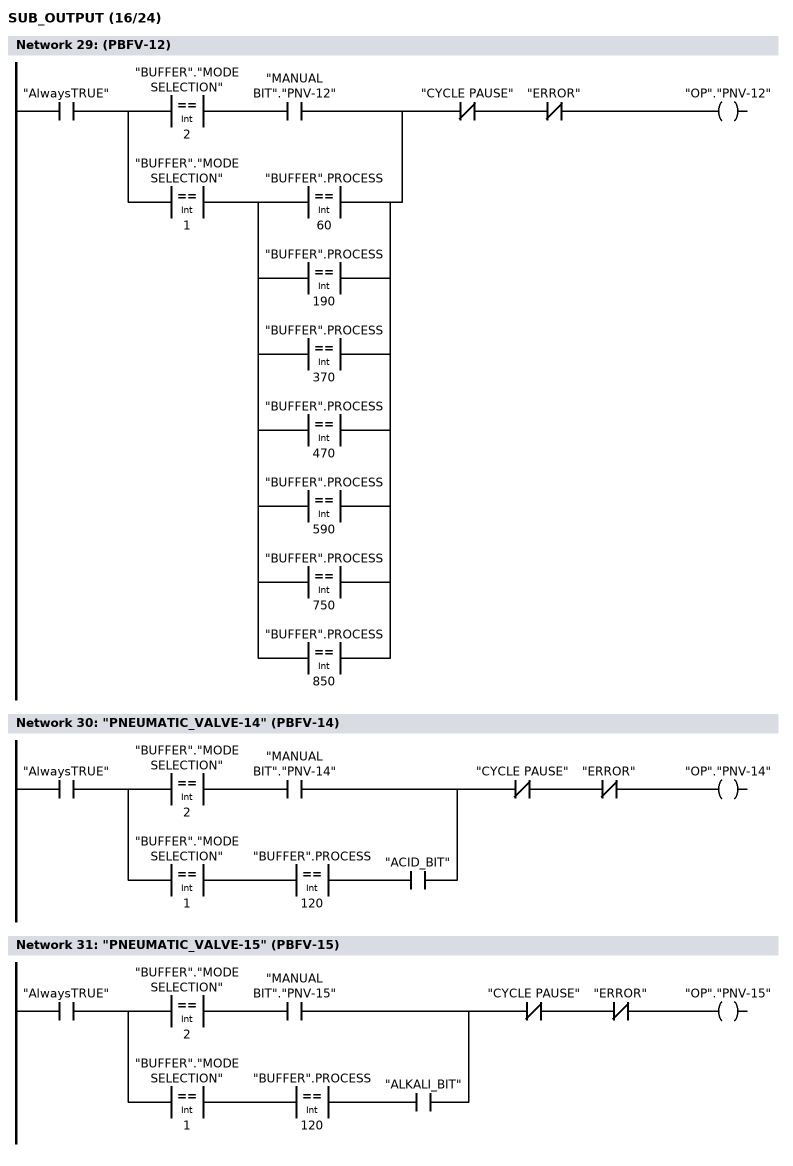
   RUNG wire#powerrail
      Contact( "AlwaysTRUE" )
      wire#w1
      { S7_Templates := "SrcType := Int" } EQ_Contact(in1 := "BUFFER"."MODE SELECTION", in2 := 2)
      Contact( "MANUAL BIT"."PNV-12" )
      wire#w2
      I_Contact( "CYCLE PAUSE" )
      I_Contact( "ERROR" )
      Coil( "OP"."PNV-12" )
   END_RUNG
   RUNG wire#w1
      { S7_Templates := "SrcType := Int" } EQ_Contact(in1 := "BUFFER"."MODE SELECTION", in2 := 1)
      wire#w3
      { S7_Templates := "SrcType := Int" } EQ_Contact(in1 := "BUFFER".PROCESS, in2 := 60)
   END_RUNG wire#w2
   RUNG wire#w3
      { S7_Templates := "SrcType := Int" } EQ_Contact(in1 := "BUFFER".PROCESS, in2 := 190)
   END_RUNG wire#w2
   RUNG wire#w3
      { S7_Templates := "SrcType := Int" } EQ_Contact(in1 := "BUFFER".PROCESS, in2 := 370)
   END_RUNG wire#w2
   RUNG wire#w3
      { S7_Templates := "SrcType := Int" } EQ_Contact(in1 := "BUFFER".PROCESS, in2 := 470)
   END_RUNG wire#w2
   RUNG wire#w3
      { S7_Templates := "SrcType := Int" } EQ_Contact(in1 := "BUFFER".PROCESS, in2 := 590)
   END_RUNG wire#w2
   RUNG wire#w3
      { S7_Templates := "SrcType := Int" } EQ_Contact(in1 := "BUFFER".PROCESS, in2 := 750)
   END_RUNG wire#w2
   RUNG wire#w3
      { S7_Templates := "SrcType := Int" } EQ_Contact(in1 := "BUFFER".PROCESS, in2 := 850)
   END_RUNG wire#w2
   // the same network as SCL:
   "OP"."PNV-12" := "AlwaysTRUE" AND ((("BUFFER"."MODE SELECTION" = 2) AND "MANUAL BIT"."PNV-12") OR (("BUFFER"."MODE SELECTION" = 1) AND (("BUFFER".PROCESS = 60) OR ("BUFFER".PROCESS = 190) OR ("BUFFER".PROCESS = 370) OR ("BUFFER".PROCESS = 470) OR ("BUFFER".PROCESS = 590) OR ("BUFFER".PROCESS = 750) OR ("BUFFER".PROCESS = 850)))) AND NOT "CYCLE PAUSE" AND NOT "ERROR";
END_REGION

REGION Network 30: "PNEUMATIC_VALVE-14" (PBFV-14)
   RUNG wire#powerrail
      Contact( "AlwaysTRUE" )
      wire#w1
      { S7_Templates := "SrcType := Int" } EQ_Contact(in1 := "BUFFER"."MODE SELECTION", in2 := 2)
      Contact( "MANUAL BIT"."PNV-14" )
      wire#w2
      I_Contact( "CYCLE PAUSE" )
      I_Contact( "ERROR" )
      Coil( "OP"."PNV-14" )
   END_RUNG
   RUNG wire#w1
      { S7_Templates := "SrcType := Int" } EQ_Contact(in1 := "BUFFER"."MODE SELECTION", in2 := 1)
      { S7_Templates := "SrcType := Int" } EQ_Contact(in1 := "BUFFER".PROCESS, in2 := 120)
      Contact( "ACID_BIT" )
   END_RUNG wire#w2
   // the same network as SCL:
   "OP"."PNV-14" := "AlwaysTRUE" AND ((("BUFFER"."MODE SELECTION" = 2) AND "MANUAL BIT"."PNV-14") OR (("BUFFER"."MODE SELECTION" = 1) AND ("BUFFER".PROCESS = 120) AND "ACID_BIT")) AND NOT "CYCLE PAUSE" AND NOT "ERROR";
END_REGION

REGION Network 31: "PNEUMATIC_VALVE-15" (PBFV-15)
   RUNG wire#powerrail
      Contact( "AlwaysTRUE" )
      wire#w1
      { S7_Templates := "SrcType := Int" } EQ_Contact(in1 := "BUFFER"."MODE SELECTION", in2 := 2)
      Contact( "MANUAL BIT"."PNV-15" )
      wire#w2
      I_Contact( "CYCLE PAUSE" )
      I_Contact( "ERROR" )
      Coil( "OP"."PNV-15" )
   END_RUNG
   RUNG wire#w1
      { S7_Templates := "SrcType := Int" } EQ_Contact(in1 := "BUFFER"."MODE SELECTION", in2 := 1)
      { S7_Templates := "SrcType := Int" } EQ_Contact(in1 := "BUFFER".PROCESS, in2 := 120)
      Contact( "ALKALI_BIT" )
   END_RUNG wire#w2
   // the same network as SCL:
   "OP"."PNV-15" := "AlwaysTRUE" AND ((("BUFFER"."MODE SELECTION" = 2) AND "MANUAL BIT"."PNV-15") OR (("BUFFER"."MODE SELECTION" = 1) AND ("BUFFER".PROCESS = 120) AND "ALKALI_BIT")) AND NOT "CYCLE PAUSE" AND NOT "ERROR";
END_REGION

REGION Network 32: "PNEUMATIC_VALVE-17" (PBFV-17) MFG1- MIXING
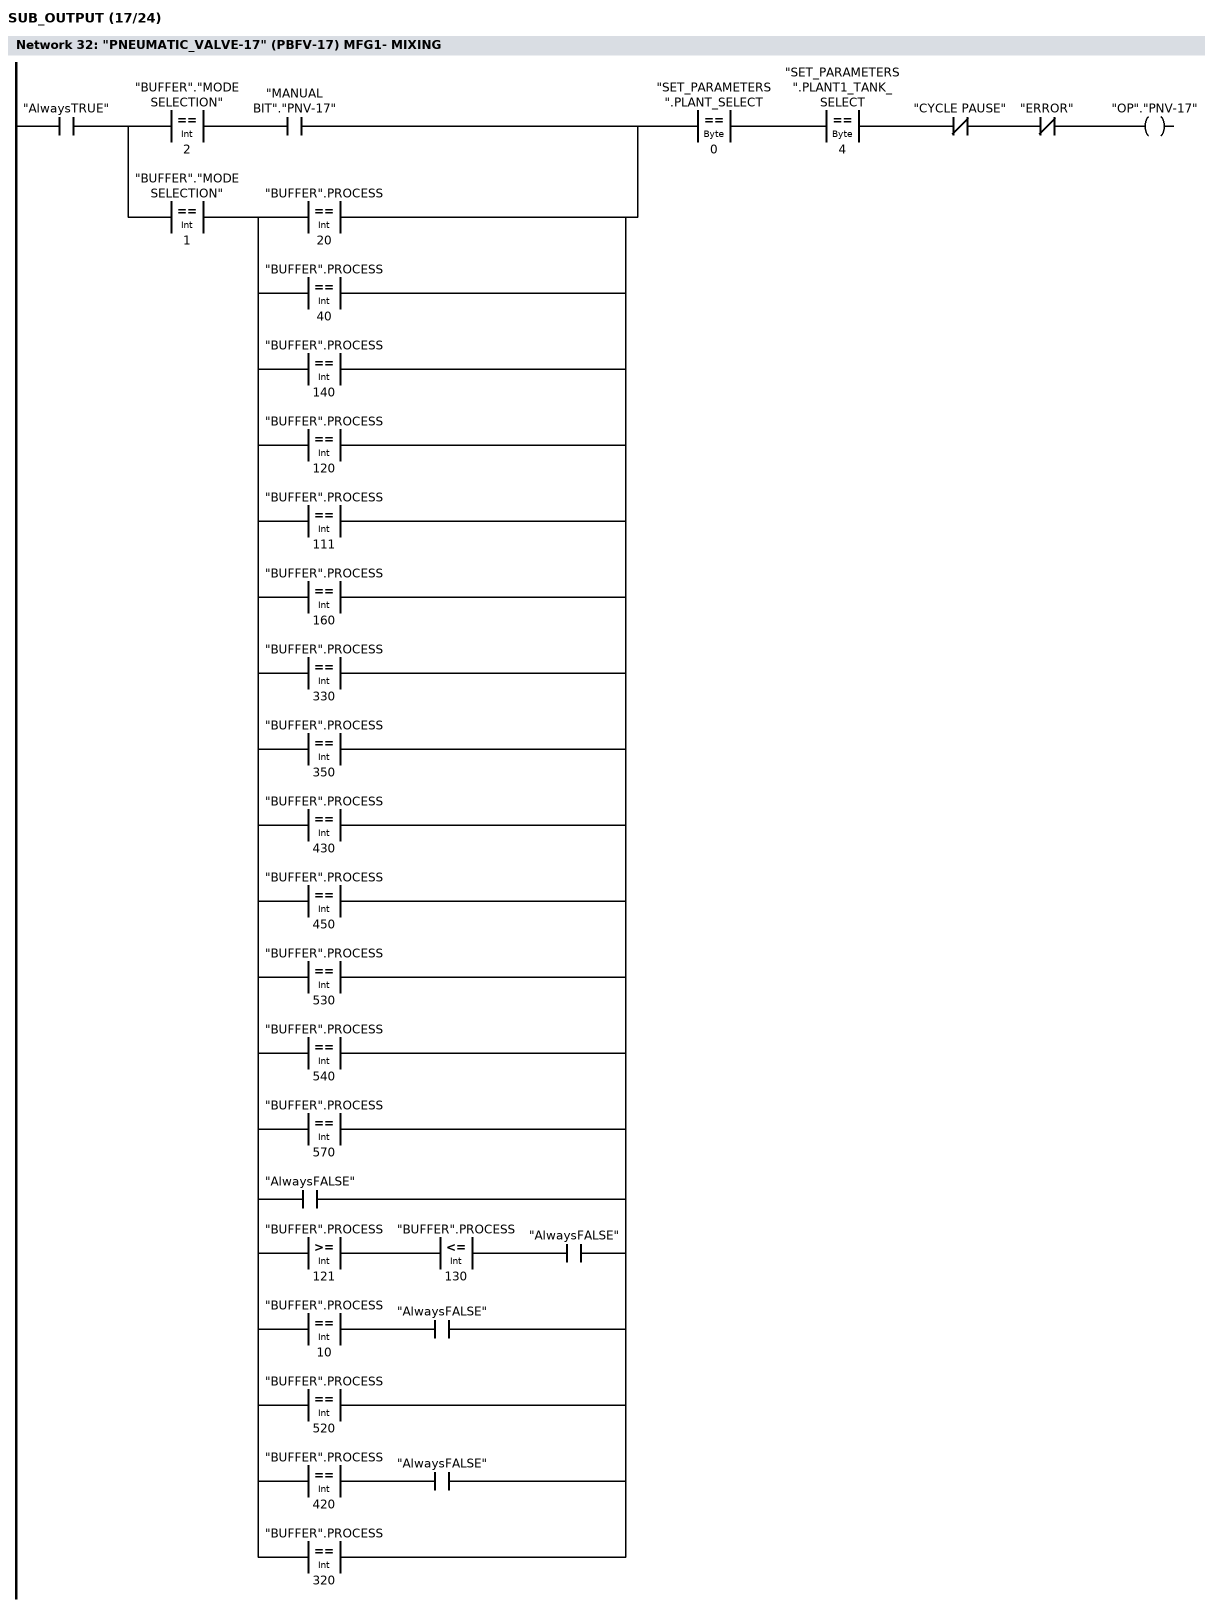
   RUNG wire#powerrail
      Contact( "AlwaysTRUE" )
      wire#w1
      { S7_Templates := "SrcType := Int" } EQ_Contact(in1 := "BUFFER"."MODE SELECTION", in2 := 2)
      Contact( "MANUAL BIT"."PNV-17" )
      wire#w2
      { S7_Templates := "SrcType := Byte" } EQ_Contact(in1 := "SET_PARAMETERS".PLANT_SELECT, in2 := 0)
      { S7_Templates := "SrcType := Byte" } EQ_Contact(in1 := "SET_PARAMETERS".PLANT1_TANK_SELECT, in2 := 4)
      I_Contact( "CYCLE PAUSE" )
      I_Contact( "ERROR" )
      Coil( "OP"."PNV-17" )
   END_RUNG
   RUNG wire#w1
      { S7_Templates := "SrcType := Int" } EQ_Contact(in1 := "BUFFER"."MODE SELECTION", in2 := 1)
      wire#w3
      { S7_Templates := "SrcType := Int" } EQ_Contact(in1 := "BUFFER".PROCESS, in2 := 20)
   END_RUNG wire#w2
   RUNG wire#w3
      { S7_Templates := "SrcType := Int" } EQ_Contact(in1 := "BUFFER".PROCESS, in2 := 40)
   END_RUNG wire#w2
   RUNG wire#w3
      { S7_Templates := "SrcType := Int" } EQ_Contact(in1 := "BUFFER".PROCESS, in2 := 140)
   END_RUNG wire#w2
   RUNG wire#w3
      { S7_Templates := "SrcType := Int" } EQ_Contact(in1 := "BUFFER".PROCESS, in2 := 120)
   END_RUNG wire#w2
   RUNG wire#w3
      { S7_Templates := "SrcType := Int" } EQ_Contact(in1 := "BUFFER".PROCESS, in2 := 111)
   END_RUNG wire#w2
   RUNG wire#w3
      { S7_Templates := "SrcType := Int" } EQ_Contact(in1 := "BUFFER".PROCESS, in2 := 160)
   END_RUNG wire#w2
   RUNG wire#w3
      { S7_Templates := "SrcType := Int" } EQ_Contact(in1 := "BUFFER".PROCESS, in2 := 330)
   END_RUNG wire#w2
   RUNG wire#w3
      { S7_Templates := "SrcType := Int" } EQ_Contact(in1 := "BUFFER".PROCESS, in2 := 350)
   END_RUNG wire#w2
   RUNG wire#w3
      { S7_Templates := "SrcType := Int" } EQ_Contact(in1 := "BUFFER".PROCESS, in2 := 430)
   END_RUNG wire#w2
   RUNG wire#w3
      { S7_Templates := "SrcType := Int" } EQ_Contact(in1 := "BUFFER".PROCESS, in2 := 450)
   END_RUNG wire#w2
   RUNG wire#w3
      { S7_Templates := "SrcType := Int" } EQ_Contact(in1 := "BUFFER".PROCESS, in2 := 530)
   END_RUNG wire#w2
   RUNG wire#w3
      { S7_Templates := "SrcType := Int" } EQ_Contact(in1 := "BUFFER".PROCESS, in2 := 540)
   END_RUNG wire#w2
   RUNG wire#w3
      { S7_Templates := "SrcType := Int" } EQ_Contact(in1 := "BUFFER".PROCESS, in2 := 570)
   END_RUNG wire#w2
   RUNG wire#w3
      Contact( "AlwaysFALSE" )
   END_RUNG wire#w2
   RUNG wire#w3
      { S7_Templates := "SrcType := Int" } GE_Contact(in1 := "BUFFER".PROCESS, in2 := 121)
      { S7_Templates := "SrcType := Int" } LE_Contact(in1 := "BUFFER".PROCESS, in2 := 130)
      Contact( "AlwaysFALSE" )
   END_RUNG wire#w2
   RUNG wire#w3
      { S7_Templates := "SrcType := Int" } EQ_Contact(in1 := "BUFFER".PROCESS, in2 := 10)
      Contact( "AlwaysFALSE" )
   END_RUNG wire#w2
   RUNG wire#w3
      { S7_Templates := "SrcType := Int" } EQ_Contact(in1 := "BUFFER".PROCESS, in2 := 520)
   END_RUNG wire#w2
   RUNG wire#w3
      { S7_Templates := "SrcType := Int" } EQ_Contact(in1 := "BUFFER".PROCESS, in2 := 420)
      Contact( "AlwaysFALSE" )
   END_RUNG wire#w2
   RUNG wire#w3
      { S7_Templates := "SrcType := Int" } EQ_Contact(in1 := "BUFFER".PROCESS, in2 := 320)
   END_RUNG wire#w2
   // the same network as SCL:
   "OP"."PNV-17" := "AlwaysTRUE" AND ((("BUFFER"."MODE SELECTION" = 2) AND "MANUAL BIT"."PNV-17") OR (("BUFFER"."MODE SELECTION" = 1) AND (("BUFFER".PROCESS = 20) OR ("BUFFER".PROCESS = 40) OR ("BUFFER".PROCESS = 140) OR ("BUFFER".PROCESS = 120) OR ("BUFFER".PROCESS = 111) OR ("BUFFER".PROCESS = 160) OR ("BUFFER".PROCESS = 330) OR ("BUFFER".PROCESS = 350) OR ("BUFFER".PROCESS = 430) OR ("BUFFER".PROCESS = 450) OR ("BUFFER".PROCESS = 530) OR ("BUFFER".PROCESS = 540) OR ("BUFFER".PROCESS = 570) OR "AlwaysFALSE" OR (("BUFFER".PROCESS >= 121) AND ("BUFFER".PROCESS <= 130) AND "AlwaysFALSE") OR (("BUFFER".PROCESS = 10) AND "AlwaysFALSE") OR ("BUFFER".PROCESS = 520) OR (("BUFFER".PROCESS = 420) AND "AlwaysFALSE") OR ("BUFFER".PROCESS = 320)))) AND ("SET_PARAMETERS".PLANT_SELECT = 0) AND ("SET_PARAMETERS".PLANT1_TANK_SELECT = 4) AND NOT "CYCLE PAUSE" AND NOT "ERROR";
END_REGION

REGION Network 33: "PNEUMATIC_VALVE-19" (PBFV-19) MFG2 - MFG
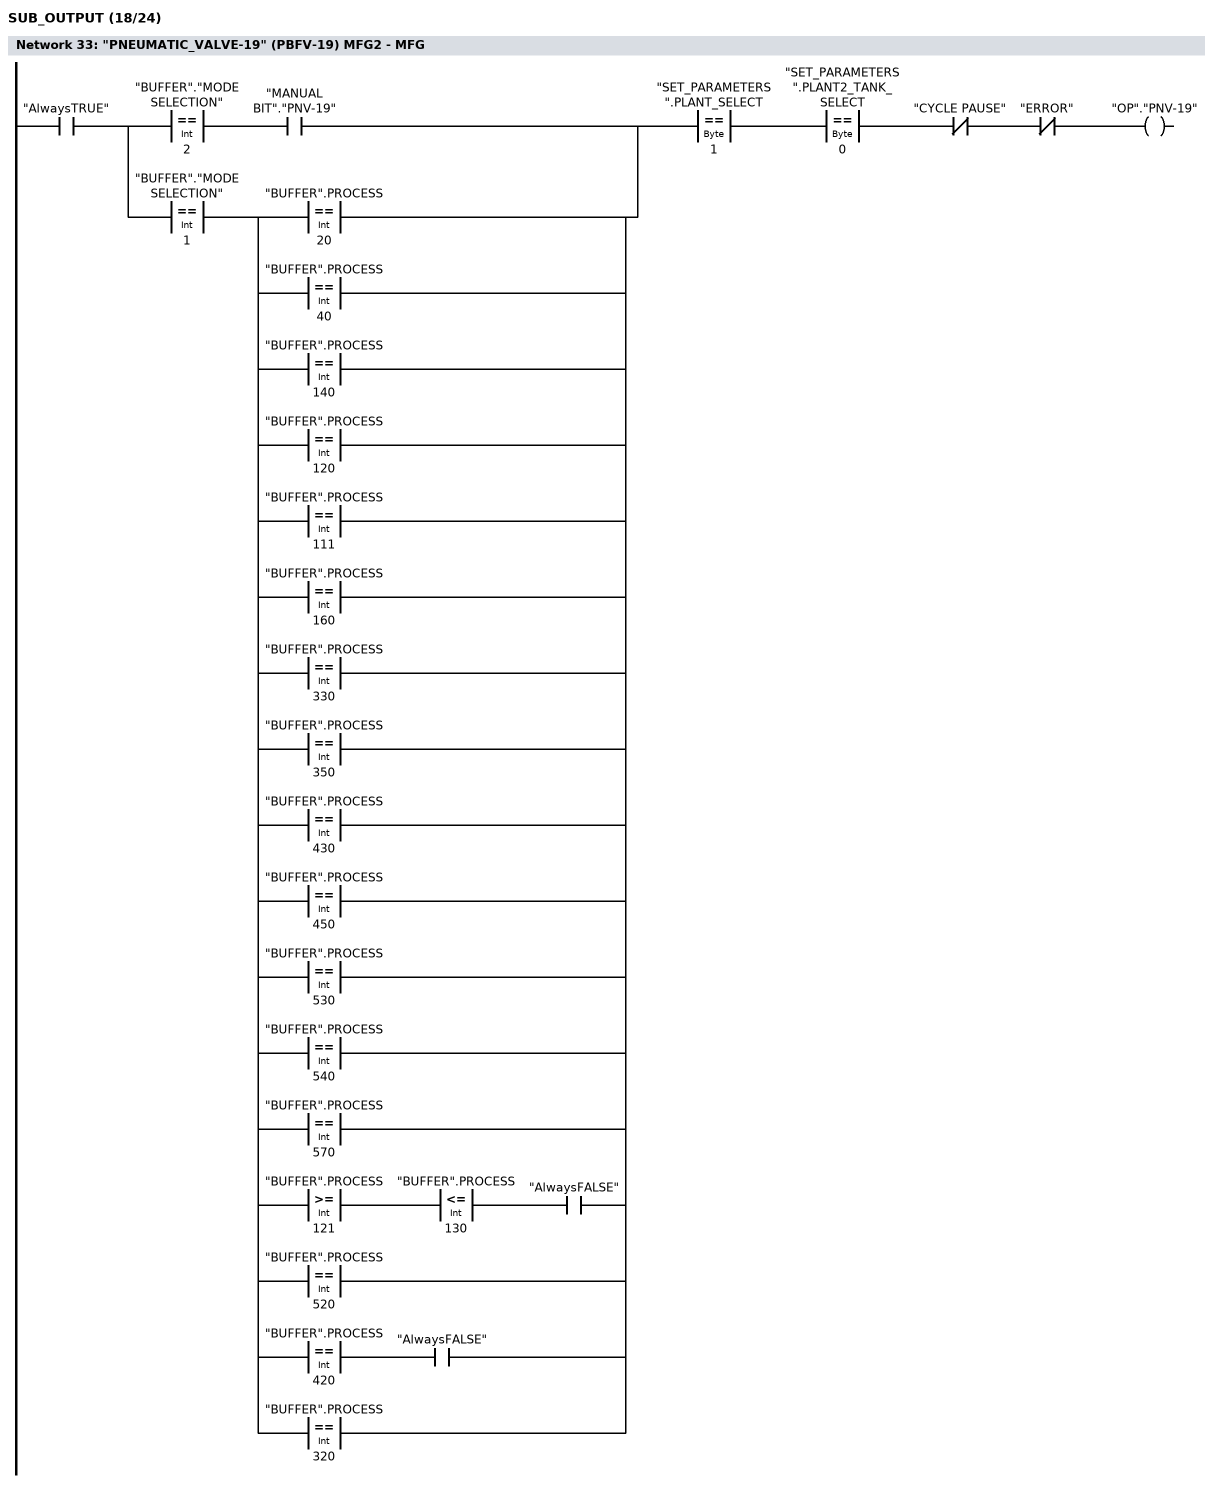
   RUNG wire#powerrail
      Contact( "AlwaysTRUE" )
      wire#w1
      { S7_Templates := "SrcType := Int" } EQ_Contact(in1 := "BUFFER"."MODE SELECTION", in2 := 2)
      Contact( "MANUAL BIT"."PNV-19" )
      wire#w2
      { S7_Templates := "SrcType := Byte" } EQ_Contact(in1 := "SET_PARAMETERS".PLANT_SELECT, in2 := 1)
      { S7_Templates := "SrcType := Byte" } EQ_Contact(in1 := "SET_PARAMETERS".PLANT2_TANK_SELECT, in2 := 0)
      I_Contact( "CYCLE PAUSE" )
      I_Contact( "ERROR" )
      Coil( "OP"."PNV-19" )
   END_RUNG
   RUNG wire#w1
      { S7_Templates := "SrcType := Int" } EQ_Contact(in1 := "BUFFER"."MODE SELECTION", in2 := 1)
      wire#w3
      { S7_Templates := "SrcType := Int" } EQ_Contact(in1 := "BUFFER".PROCESS, in2 := 20)
   END_RUNG wire#w2
   RUNG wire#w3
      { S7_Templates := "SrcType := Int" } EQ_Contact(in1 := "BUFFER".PROCESS, in2 := 40)
   END_RUNG wire#w2
   RUNG wire#w3
      { S7_Templates := "SrcType := Int" } EQ_Contact(in1 := "BUFFER".PROCESS, in2 := 140)
   END_RUNG wire#w2
   RUNG wire#w3
      { S7_Templates := "SrcType := Int" } EQ_Contact(in1 := "BUFFER".PROCESS, in2 := 120)
   END_RUNG wire#w2
   RUNG wire#w3
      { S7_Templates := "SrcType := Int" } EQ_Contact(in1 := "BUFFER".PROCESS, in2 := 111)
   END_RUNG wire#w2
   RUNG wire#w3
      { S7_Templates := "SrcType := Int" } EQ_Contact(in1 := "BUFFER".PROCESS, in2 := 160)
   END_RUNG wire#w2
   RUNG wire#w3
      { S7_Templates := "SrcType := Int" } EQ_Contact(in1 := "BUFFER".PROCESS, in2 := 330)
   END_RUNG wire#w2
   RUNG wire#w3
      { S7_Templates := "SrcType := Int" } EQ_Contact(in1 := "BUFFER".PROCESS, in2 := 350)
   END_RUNG wire#w2
   RUNG wire#w3
      { S7_Templates := "SrcType := Int" } EQ_Contact(in1 := "BUFFER".PROCESS, in2 := 430)
   END_RUNG wire#w2
   RUNG wire#w3
      { S7_Templates := "SrcType := Int" } EQ_Contact(in1 := "BUFFER".PROCESS, in2 := 450)
   END_RUNG wire#w2
   RUNG wire#w3
      { S7_Templates := "SrcType := Int" } EQ_Contact(in1 := "BUFFER".PROCESS, in2 := 530)
   END_RUNG wire#w2
   RUNG wire#w3
      { S7_Templates := "SrcType := Int" } EQ_Contact(in1 := "BUFFER".PROCESS, in2 := 540)
   END_RUNG wire#w2
   RUNG wire#w3
      { S7_Templates := "SrcType := Int" } EQ_Contact(in1 := "BUFFER".PROCESS, in2 := 570)
   END_RUNG wire#w2
   RUNG wire#w3
      { S7_Templates := "SrcType := Int" } GE_Contact(in1 := "BUFFER".PROCESS, in2 := 121)
      { S7_Templates := "SrcType := Int" } LE_Contact(in1 := "BUFFER".PROCESS, in2 := 130)
      Contact( "AlwaysFALSE" )
   END_RUNG wire#w2
   RUNG wire#w3
      { S7_Templates := "SrcType := Int" } EQ_Contact(in1 := "BUFFER".PROCESS, in2 := 520)
   END_RUNG wire#w2
   RUNG wire#w3
      { S7_Templates := "SrcType := Int" } EQ_Contact(in1 := "BUFFER".PROCESS, in2 := 420)
      Contact( "AlwaysFALSE" )
   END_RUNG wire#w2
   RUNG wire#w3
      { S7_Templates := "SrcType := Int" } EQ_Contact(in1 := "BUFFER".PROCESS, in2 := 320)
   END_RUNG wire#w2
   // the same network as SCL:
   "OP"."PNV-19" := "AlwaysTRUE" AND ((("BUFFER"."MODE SELECTION" = 2) AND "MANUAL BIT"."PNV-19") OR (("BUFFER"."MODE SELECTION" = 1) AND (("BUFFER".PROCESS = 20) OR ("BUFFER".PROCESS = 40) OR ("BUFFER".PROCESS = 140) OR ("BUFFER".PROCESS = 120) OR ("BUFFER".PROCESS = 111) OR ("BUFFER".PROCESS = 160) OR ("BUFFER".PROCESS = 330) OR ("BUFFER".PROCESS = 350) OR ("BUFFER".PROCESS = 430) OR ("BUFFER".PROCESS = 450) OR ("BUFFER".PROCESS = 530) OR ("BUFFER".PROCESS = 540) OR ("BUFFER".PROCESS = 570) OR (("BUFFER".PROCESS >= 121) AND ("BUFFER".PROCESS <= 130) AND "AlwaysFALSE") OR ("BUFFER".PROCESS = 520) OR (("BUFFER".PROCESS = 420) AND "AlwaysFALSE") OR ("BUFFER".PROCESS = 320)))) AND ("SET_PARAMETERS".PLANT_SELECT = 1) AND ("SET_PARAMETERS".PLANT2_TANK_SELECT = 0) AND NOT "CYCLE PAUSE" AND NOT "ERROR";
END_REGION

REGION Network 34: "PNEUMATIC_VALVE-20" (PBFV-20) MFG2- STORAGE1
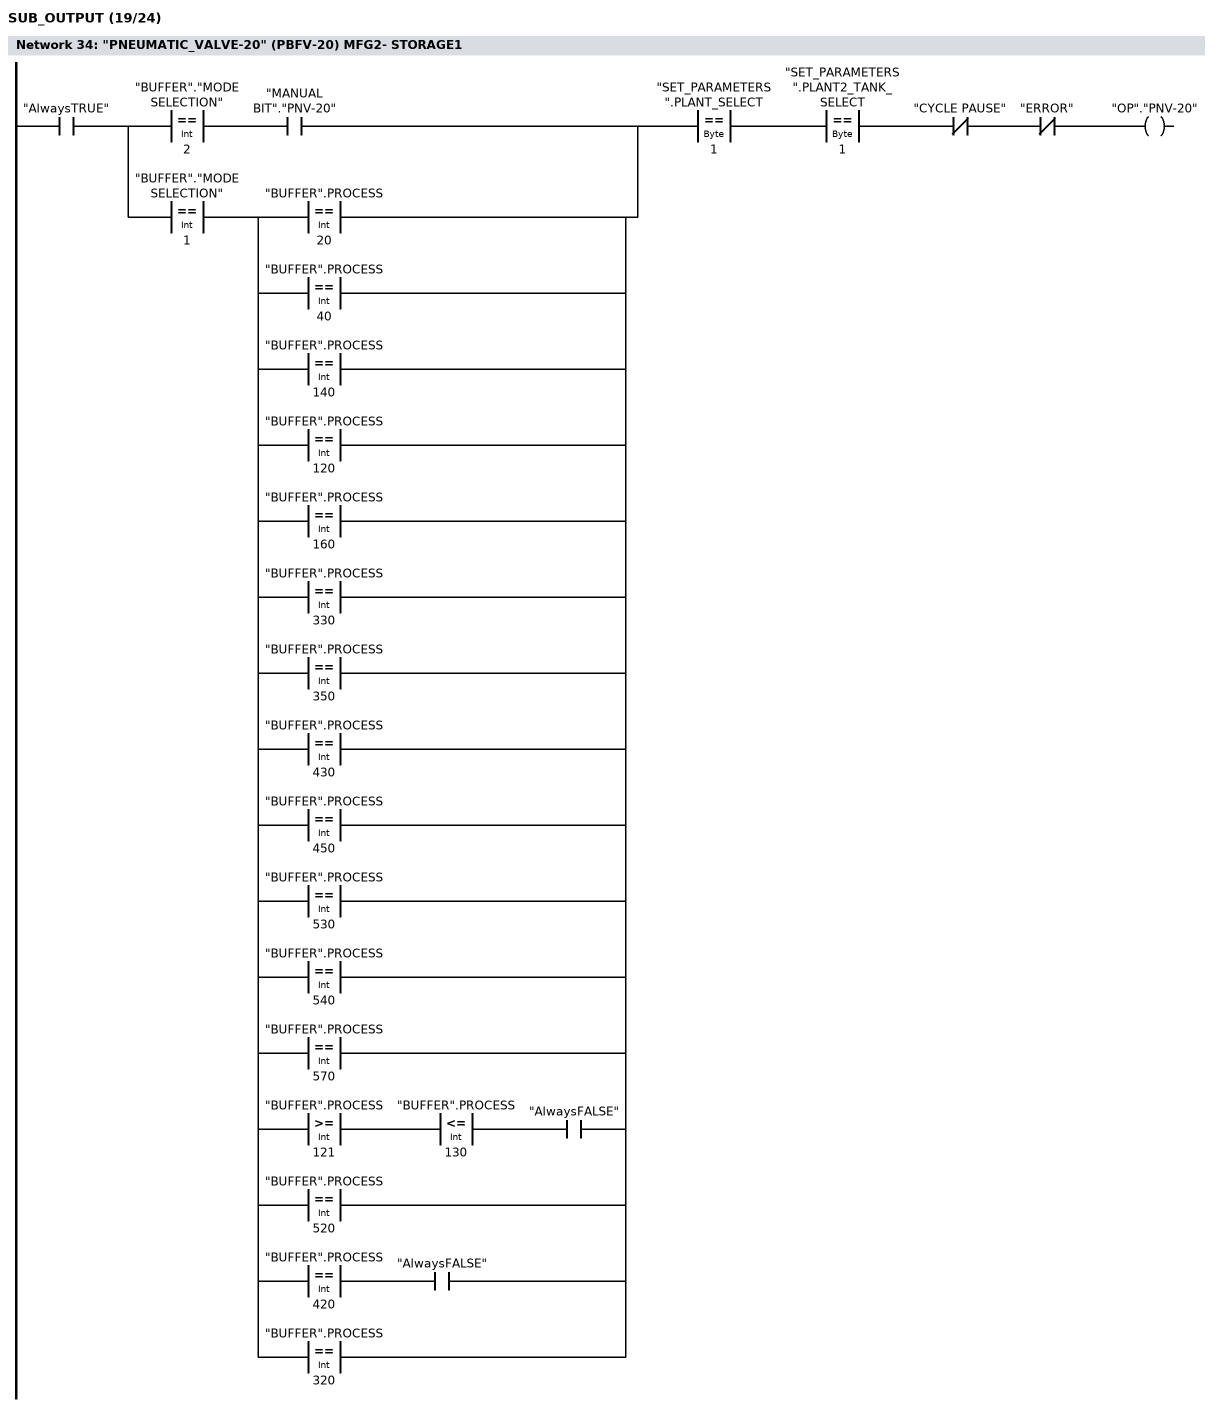
   RUNG wire#powerrail
      Contact( "AlwaysTRUE" )
      wire#w1
      { S7_Templates := "SrcType := Int" } EQ_Contact(in1 := "BUFFER"."MODE SELECTION", in2 := 2)
      Contact( "MANUAL BIT"."PNV-20" )
      wire#w2
      { S7_Templates := "SrcType := Byte" } EQ_Contact(in1 := "SET_PARAMETERS".PLANT_SELECT, in2 := 1)
      { S7_Templates := "SrcType := Byte" } EQ_Contact(in1 := "SET_PARAMETERS".PLANT2_TANK_SELECT, in2 := 1)
      I_Contact( "CYCLE PAUSE" )
      I_Contact( "ERROR" )
      Coil( "OP"."PNV-20" )
   END_RUNG
   RUNG wire#w1
      { S7_Templates := "SrcType := Int" } EQ_Contact(in1 := "BUFFER"."MODE SELECTION", in2 := 1)
      wire#w3
      { S7_Templates := "SrcType := Int" } EQ_Contact(in1 := "BUFFER".PROCESS, in2 := 20)
   END_RUNG wire#w2
   RUNG wire#w3
      { S7_Templates := "SrcType := Int" } EQ_Contact(in1 := "BUFFER".PROCESS, in2 := 40)
   END_RUNG wire#w2
   RUNG wire#w3
      { S7_Templates := "SrcType := Int" } EQ_Contact(in1 := "BUFFER".PROCESS, in2 := 140)
   END_RUNG wire#w2
   RUNG wire#w3
      { S7_Templates := "SrcType := Int" } EQ_Contact(in1 := "BUFFER".PROCESS, in2 := 120)
   END_RUNG wire#w2
   RUNG wire#w3
      { S7_Templates := "SrcType := Int" } EQ_Contact(in1 := "BUFFER".PROCESS, in2 := 160)
   END_RUNG wire#w2
   RUNG wire#w3
      { S7_Templates := "SrcType := Int" } EQ_Contact(in1 := "BUFFER".PROCESS, in2 := 330)
   END_RUNG wire#w2
   RUNG wire#w3
      { S7_Templates := "SrcType := Int" } EQ_Contact(in1 := "BUFFER".PROCESS, in2 := 350)
   END_RUNG wire#w2
   RUNG wire#w3
      { S7_Templates := "SrcType := Int" } EQ_Contact(in1 := "BUFFER".PROCESS, in2 := 430)
   END_RUNG wire#w2
   RUNG wire#w3
      { S7_Templates := "SrcType := Int" } EQ_Contact(in1 := "BUFFER".PROCESS, in2 := 450)
   END_RUNG wire#w2
   RUNG wire#w3
      { S7_Templates := "SrcType := Int" } EQ_Contact(in1 := "BUFFER".PROCESS, in2 := 530)
   END_RUNG wire#w2
   RUNG wire#w3
      { S7_Templates := "SrcType := Int" } EQ_Contact(in1 := "BUFFER".PROCESS, in2 := 540)
   END_RUNG wire#w2
   RUNG wire#w3
      { S7_Templates := "SrcType := Int" } EQ_Contact(in1 := "BUFFER".PROCESS, in2 := 570)
   END_RUNG wire#w2
   RUNG wire#w3
      { S7_Templates := "SrcType := Int" } GE_Contact(in1 := "BUFFER".PROCESS, in2 := 121)
      { S7_Templates := "SrcType := Int" } LE_Contact(in1 := "BUFFER".PROCESS, in2 := 130)
      Contact( "AlwaysFALSE" )
   END_RUNG wire#w2
   RUNG wire#w3
      { S7_Templates := "SrcType := Int" } EQ_Contact(in1 := "BUFFER".PROCESS, in2 := 520)
   END_RUNG wire#w2
   RUNG wire#w3
      { S7_Templates := "SrcType := Int" } EQ_Contact(in1 := "BUFFER".PROCESS, in2 := 420)
      Contact( "AlwaysFALSE" )
   END_RUNG wire#w2
   RUNG wire#w3
      { S7_Templates := "SrcType := Int" } EQ_Contact(in1 := "BUFFER".PROCESS, in2 := 320)
   END_RUNG wire#w2
   // the same network as SCL:
   "OP"."PNV-20" := "AlwaysTRUE" AND ((("BUFFER"."MODE SELECTION" = 2) AND "MANUAL BIT"."PNV-20") OR (("BUFFER"."MODE SELECTION" = 1) AND (("BUFFER".PROCESS = 20) OR ("BUFFER".PROCESS = 40) OR ("BUFFER".PROCESS = 140) OR ("BUFFER".PROCESS = 120) OR ("BUFFER".PROCESS = 160) OR ("BUFFER".PROCESS = 330) OR ("BUFFER".PROCESS = 350) OR ("BUFFER".PROCESS = 430) OR ("BUFFER".PROCESS = 450) OR ("BUFFER".PROCESS = 530) OR ("BUFFER".PROCESS = 540) OR ("BUFFER".PROCESS = 570) OR (("BUFFER".PROCESS >= 121) AND ("BUFFER".PROCESS <= 130) AND "AlwaysFALSE") OR ("BUFFER".PROCESS = 520) OR (("BUFFER".PROCESS = 420) AND "AlwaysFALSE") OR ("BUFFER".PROCESS = 320)))) AND ("SET_PARAMETERS".PLANT_SELECT = 1) AND ("SET_PARAMETERS".PLANT2_TANK_SELECT = 1) AND NOT "CYCLE PAUSE" AND NOT "ERROR";
END_REGION

REGION Network 35: "PNEUMATIC_VALVE-21" (PV-21)
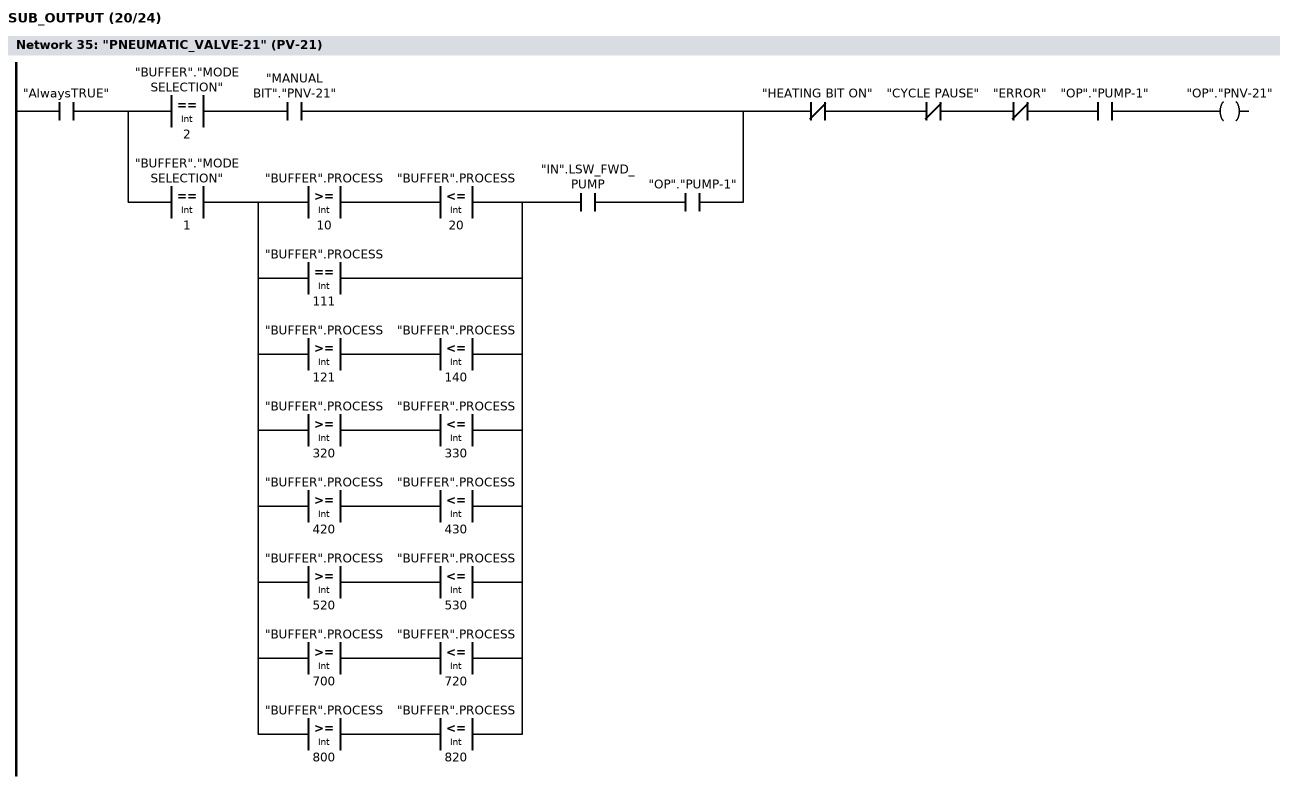
   RUNG wire#powerrail
      Contact( "AlwaysTRUE" )
      wire#w1
      { S7_Templates := "SrcType := Int" } EQ_Contact(in1 := "BUFFER"."MODE SELECTION", in2 := 2)
      Contact( "MANUAL BIT"."PNV-21" )
      wire#w2
      I_Contact( "HEATING BIT ON" )
      I_Contact( "CYCLE PAUSE" )
      I_Contact( "ERROR" )
      Contact( "OP"."PUMP-1" )
      Coil( "OP"."PNV-21" )
   END_RUNG
   RUNG wire#w1
      { S7_Templates := "SrcType := Int" } EQ_Contact(in1 := "BUFFER"."MODE SELECTION", in2 := 1)
      wire#w3
      { S7_Templates := "SrcType := Int" } GE_Contact(in1 := "BUFFER".PROCESS, in2 := 10)
      { S7_Templates := "SrcType := Int" } LE_Contact(in1 := "BUFFER".PROCESS, in2 := 20)
      wire#w4
      Contact( "IN".LSW_FWD_PUMP )
      Contact( "OP"."PUMP-1" )
   END_RUNG wire#w2
   RUNG wire#w3
      { S7_Templates := "SrcType := Int" } EQ_Contact(in1 := "BUFFER".PROCESS, in2 := 111)
   END_RUNG wire#w4
   RUNG wire#w3
      { S7_Templates := "SrcType := Int" } GE_Contact(in1 := "BUFFER".PROCESS, in2 := 121)
      { S7_Templates := "SrcType := Int" } LE_Contact(in1 := "BUFFER".PROCESS, in2 := 140)
   END_RUNG wire#w4
   RUNG wire#w3
      { S7_Templates := "SrcType := Int" } GE_Contact(in1 := "BUFFER".PROCESS, in2 := 320)
      { S7_Templates := "SrcType := Int" } LE_Contact(in1 := "BUFFER".PROCESS, in2 := 330)
   END_RUNG wire#w4
   RUNG wire#w3
      { S7_Templates := "SrcType := Int" } GE_Contact(in1 := "BUFFER".PROCESS, in2 := 420)
      { S7_Templates := "SrcType := Int" } LE_Contact(in1 := "BUFFER".PROCESS, in2 := 430)
   END_RUNG wire#w4
   RUNG wire#w3
      { S7_Templates := "SrcType := Int" } GE_Contact(in1 := "BUFFER".PROCESS, in2 := 520)
      { S7_Templates := "SrcType := Int" } LE_Contact(in1 := "BUFFER".PROCESS, in2 := 530)
   END_RUNG wire#w4
   RUNG wire#w3
      { S7_Templates := "SrcType := Int" } GE_Contact(in1 := "BUFFER".PROCESS, in2 := 700)
      { S7_Templates := "SrcType := Int" } LE_Contact(in1 := "BUFFER".PROCESS, in2 := 720)
   END_RUNG wire#w4
   RUNG wire#w3
      { S7_Templates := "SrcType := Int" } GE_Contact(in1 := "BUFFER".PROCESS, in2 := 800)
      { S7_Templates := "SrcType := Int" } LE_Contact(in1 := "BUFFER".PROCESS, in2 := 820)
   END_RUNG wire#w4
   // the same network as SCL:
   "OP"."PNV-21" := "AlwaysTRUE" AND ((("BUFFER"."MODE SELECTION" = 2) AND "MANUAL BIT"."PNV-21") OR (("BUFFER"."MODE SELECTION" = 1) AND ((("BUFFER".PROCESS >= 10) AND ("BUFFER".PROCESS <= 20)) OR ("BUFFER".PROCESS = 111) OR (("BUFFER".PROCESS >= 121) AND ("BUFFER".PROCESS <= 140)) OR (("BUFFER".PROCESS >= 320) AND ("BUFFER".PROCESS <= 330)) OR (("BUFFER".PROCESS >= 420) AND ("BUFFER".PROCESS <= 430)) OR (("BUFFER".PROCESS >= 520) AND ("BUFFER".PROCESS <= 530)) OR (("BUFFER".PROCESS >= 700) AND ("BUFFER".PROCESS <= 720)) OR (("BUFFER".PROCESS >= 800) AND ("BUFFER".PROCESS <= 820))) AND "IN".LSW_FWD_PUMP AND "OP"."PUMP-1")) AND NOT "HEATING BIT ON" AND NOT "CYCLE PAUSE" AND NOT "ERROR" AND "OP"."PUMP-1";
END_REGION

REGION Network 36: "PNEUMATIC_VALVE-25" (CIP_IN) MFG2- STORAGE2 PBFV-23
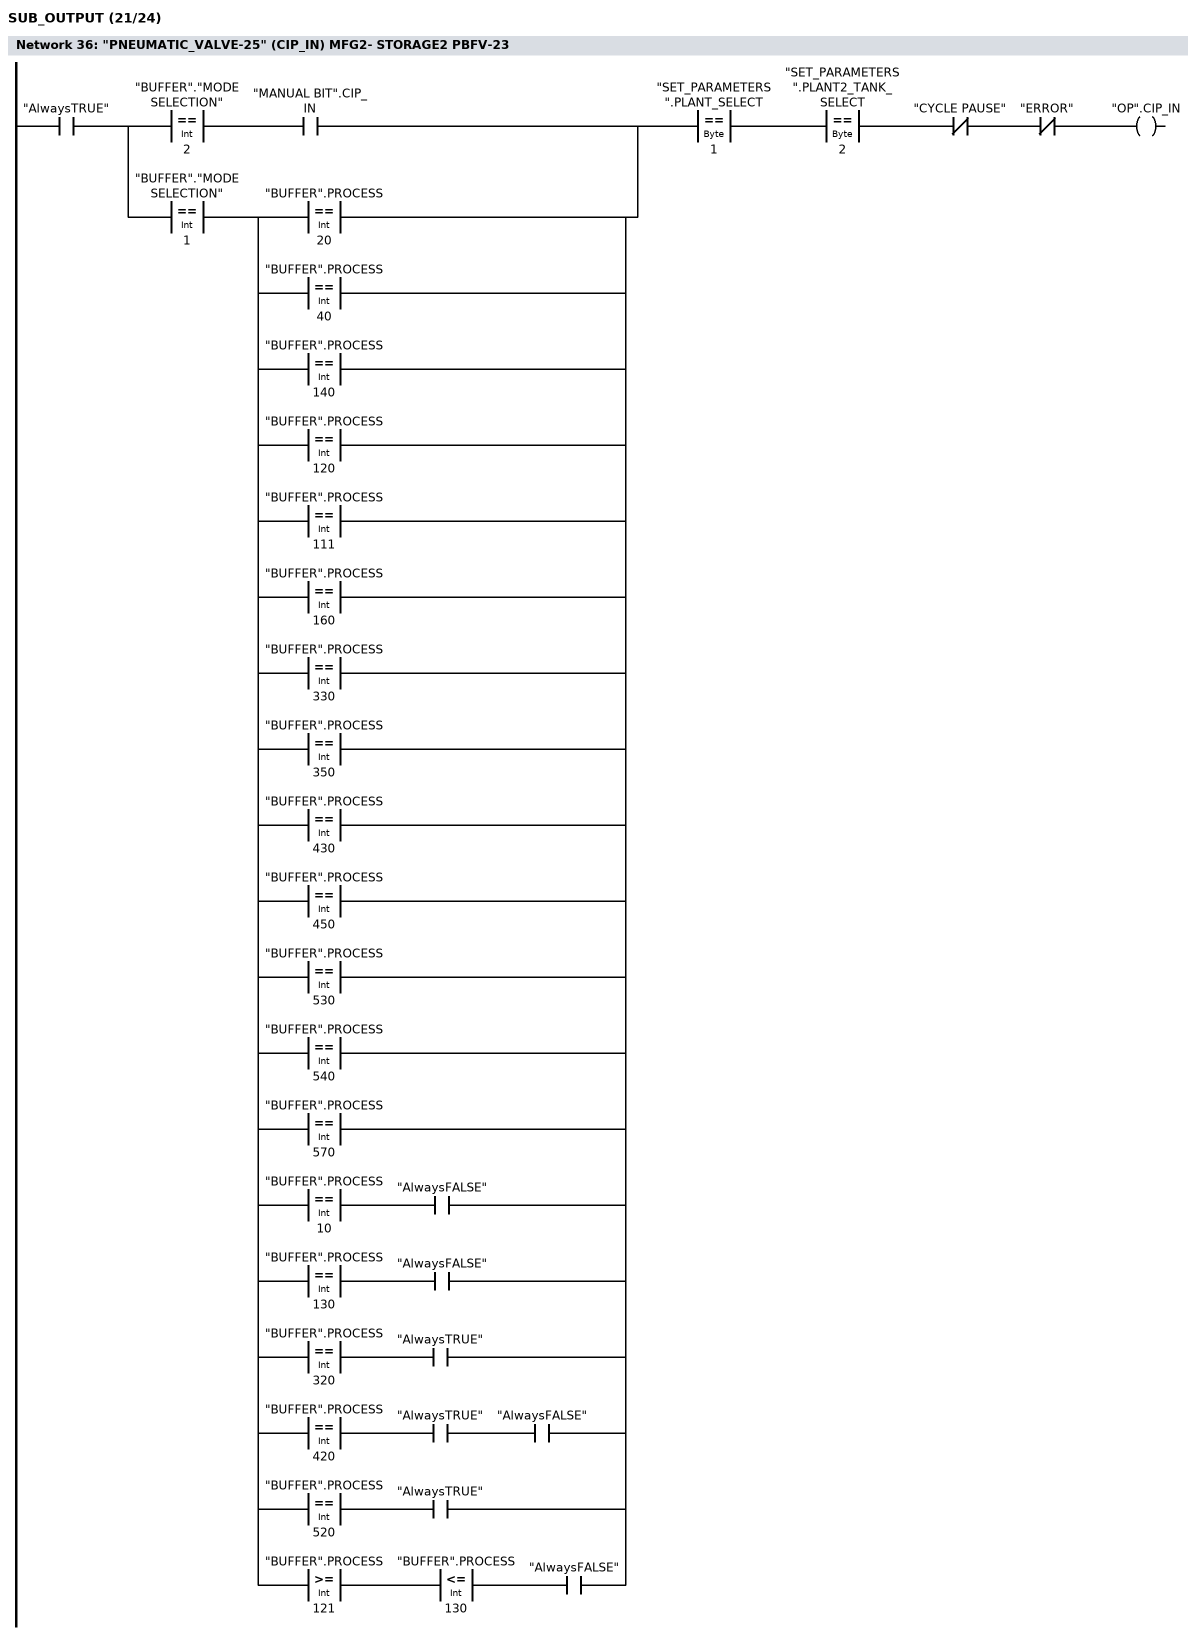
   RUNG wire#powerrail
      Contact( "AlwaysTRUE" )
      wire#w1
      { S7_Templates := "SrcType := Int" } EQ_Contact(in1 := "BUFFER"."MODE SELECTION", in2 := 2)
      Contact( "MANUAL BIT".CIP_IN )
      wire#w2
      { S7_Templates := "SrcType := Byte" } EQ_Contact(in1 := "SET_PARAMETERS".PLANT_SELECT, in2 := 1)
      { S7_Templates := "SrcType := Byte" } EQ_Contact(in1 := "SET_PARAMETERS".PLANT2_TANK_SELECT, in2 := 2)
      I_Contact( "CYCLE PAUSE" )
      I_Contact( "ERROR" )
      Coil( "OP".CIP_IN )
   END_RUNG
   RUNG wire#w1
      { S7_Templates := "SrcType := Int" } EQ_Contact(in1 := "BUFFER"."MODE SELECTION", in2 := 1)
      wire#w3
      { S7_Templates := "SrcType := Int" } EQ_Contact(in1 := "BUFFER".PROCESS, in2 := 20)
   END_RUNG wire#w2
   RUNG wire#w3
      { S7_Templates := "SrcType := Int" } EQ_Contact(in1 := "BUFFER".PROCESS, in2 := 40)
   END_RUNG wire#w2
   RUNG wire#w3
      { S7_Templates := "SrcType := Int" } EQ_Contact(in1 := "BUFFER".PROCESS, in2 := 140)
   END_RUNG wire#w2
   RUNG wire#w3
      { S7_Templates := "SrcType := Int" } EQ_Contact(in1 := "BUFFER".PROCESS, in2 := 120)
   END_RUNG wire#w2
   RUNG wire#w3
      { S7_Templates := "SrcType := Int" } EQ_Contact(in1 := "BUFFER".PROCESS, in2 := 111)
   END_RUNG wire#w2
   RUNG wire#w3
      { S7_Templates := "SrcType := Int" } EQ_Contact(in1 := "BUFFER".PROCESS, in2 := 160)
   END_RUNG wire#w2
   RUNG wire#w3
      { S7_Templates := "SrcType := Int" } EQ_Contact(in1 := "BUFFER".PROCESS, in2 := 330)
   END_RUNG wire#w2
   RUNG wire#w3
      { S7_Templates := "SrcType := Int" } EQ_Contact(in1 := "BUFFER".PROCESS, in2 := 350)
   END_RUNG wire#w2
   RUNG wire#w3
      { S7_Templates := "SrcType := Int" } EQ_Contact(in1 := "BUFFER".PROCESS, in2 := 430)
   END_RUNG wire#w2
   RUNG wire#w3
      { S7_Templates := "SrcType := Int" } EQ_Contact(in1 := "BUFFER".PROCESS, in2 := 450)
   END_RUNG wire#w2
   RUNG wire#w3
      { S7_Templates := "SrcType := Int" } EQ_Contact(in1 := "BUFFER".PROCESS, in2 := 530)
   END_RUNG wire#w2
   RUNG wire#w3
      { S7_Templates := "SrcType := Int" } EQ_Contact(in1 := "BUFFER".PROCESS, in2 := 540)
   END_RUNG wire#w2
   RUNG wire#w3
      { S7_Templates := "SrcType := Int" } EQ_Contact(in1 := "BUFFER".PROCESS, in2 := 570)
   END_RUNG wire#w2
   RUNG wire#w3
      { S7_Templates := "SrcType := Int" } EQ_Contact(in1 := "BUFFER".PROCESS, in2 := 10)
      Contact( "AlwaysFALSE" )
   END_RUNG wire#w2
   RUNG wire#w3
      { S7_Templates := "SrcType := Int" } EQ_Contact(in1 := "BUFFER".PROCESS, in2 := 130)
      Contact( "AlwaysFALSE" )
   END_RUNG wire#w2
   RUNG wire#w3
      { S7_Templates := "SrcType := Int" } EQ_Contact(in1 := "BUFFER".PROCESS, in2 := 320)
      Contact( "AlwaysTRUE" )
   END_RUNG wire#w2
   RUNG wire#w3
      { S7_Templates := "SrcType := Int" } EQ_Contact(in1 := "BUFFER".PROCESS, in2 := 420)
      Contact( "AlwaysTRUE" )
      Contact( "AlwaysFALSE" )
   END_RUNG wire#w2
   RUNG wire#w3
      { S7_Templates := "SrcType := Int" } EQ_Contact(in1 := "BUFFER".PROCESS, in2 := 520)
      Contact( "AlwaysTRUE" )
   END_RUNG wire#w2
   RUNG wire#w3
      { S7_Templates := "SrcType := Int" } GE_Contact(in1 := "BUFFER".PROCESS, in2 := 121)
      { S7_Templates := "SrcType := Int" } LE_Contact(in1 := "BUFFER".PROCESS, in2 := 130)
      Contact( "AlwaysFALSE" )
   END_RUNG wire#w2
   // the same network as SCL:
   "OP".CIP_IN := "AlwaysTRUE" AND ((("BUFFER"."MODE SELECTION" = 2) AND "MANUAL BIT".CIP_IN) OR (("BUFFER"."MODE SELECTION" = 1) AND (("BUFFER".PROCESS = 20) OR ("BUFFER".PROCESS = 40) OR ("BUFFER".PROCESS = 140) OR ("BUFFER".PROCESS = 120) OR ("BUFFER".PROCESS = 111) OR ("BUFFER".PROCESS = 160) OR ("BUFFER".PROCESS = 330) OR ("BUFFER".PROCESS = 350) OR ("BUFFER".PROCESS = 430) OR ("BUFFER".PROCESS = 450) OR ("BUFFER".PROCESS = 530) OR ("BUFFER".PROCESS = 540) OR ("BUFFER".PROCESS = 570) OR (("BUFFER".PROCESS = 10) AND "AlwaysFALSE") OR (("BUFFER".PROCESS = 130) AND "AlwaysFALSE") OR (("BUFFER".PROCESS = 320) AND "AlwaysTRUE") OR (("BUFFER".PROCESS = 420) AND "AlwaysTRUE" AND "AlwaysFALSE") OR (("BUFFER".PROCESS = 520) AND "AlwaysTRUE") OR (("BUFFER".PROCESS >= 121) AND ("BUFFER".PROCESS <= 130) AND "AlwaysFALSE")))) AND ("SET_PARAMETERS".PLANT_SELECT = 1) AND ("SET_PARAMETERS".PLANT2_TANK_SELECT = 2) AND NOT "CYCLE PAUSE" AND NOT "ERROR";
END_REGION

REGION Network 37: "PNEUMATIC_VALVE-26" (CIP_OUT) MFG2- MIXING PBFV-24
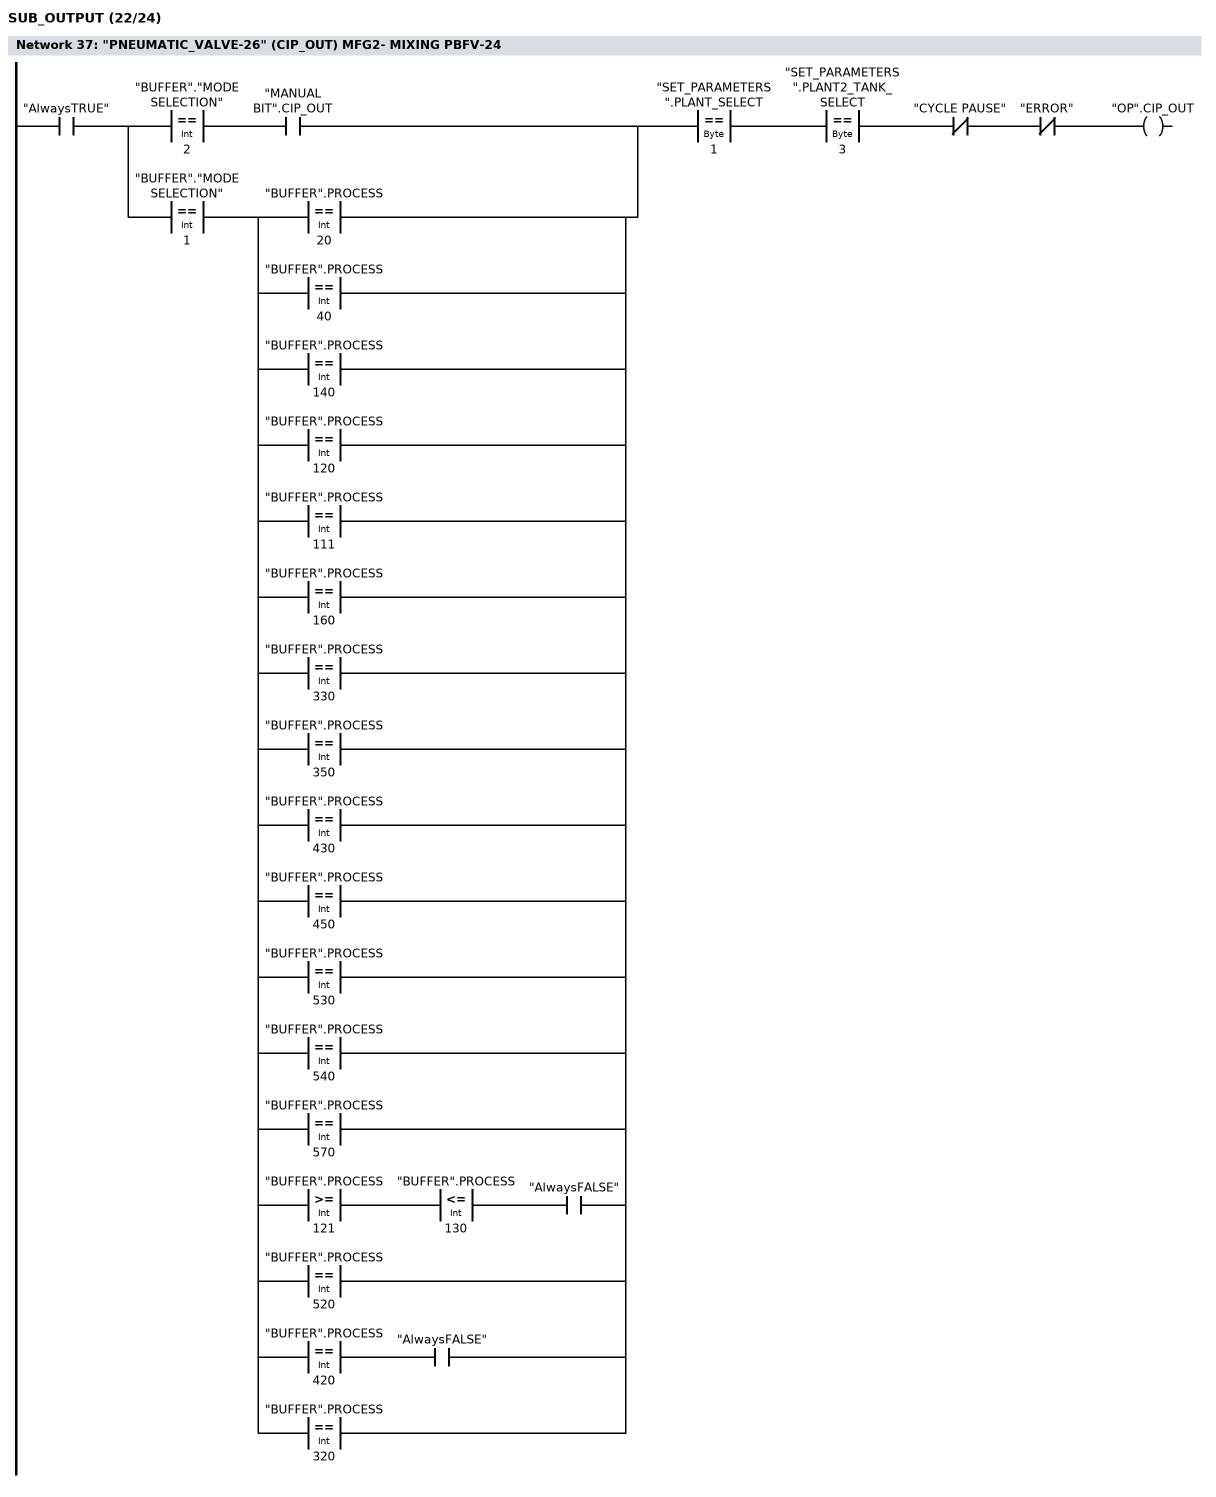
   RUNG wire#powerrail
      Contact( "AlwaysTRUE" )
      wire#w1
      { S7_Templates := "SrcType := Int" } EQ_Contact(in1 := "BUFFER"."MODE SELECTION", in2 := 2)
      Contact( "MANUAL BIT".CIP_OUT )
      wire#w2
      { S7_Templates := "SrcType := Byte" } EQ_Contact(in1 := "SET_PARAMETERS".PLANT_SELECT, in2 := 1)
      { S7_Templates := "SrcType := Byte" } EQ_Contact(in1 := "SET_PARAMETERS".PLANT2_TANK_SELECT, in2 := 3)
      I_Contact( "CYCLE PAUSE" )
      I_Contact( "ERROR" )
      Coil( "OP".CIP_OUT )
   END_RUNG
   RUNG wire#w1
      { S7_Templates := "SrcType := Int" } EQ_Contact(in1 := "BUFFER"."MODE SELECTION", in2 := 1)
      wire#w3
      { S7_Templates := "SrcType := Int" } EQ_Contact(in1 := "BUFFER".PROCESS, in2 := 20)
   END_RUNG wire#w2
   RUNG wire#w3
      { S7_Templates := "SrcType := Int" } EQ_Contact(in1 := "BUFFER".PROCESS, in2 := 40)
   END_RUNG wire#w2
   RUNG wire#w3
      { S7_Templates := "SrcType := Int" } EQ_Contact(in1 := "BUFFER".PROCESS, in2 := 140)
   END_RUNG wire#w2
   RUNG wire#w3
      { S7_Templates := "SrcType := Int" } EQ_Contact(in1 := "BUFFER".PROCESS, in2 := 120)
   END_RUNG wire#w2
   RUNG wire#w3
      { S7_Templates := "SrcType := Int" } EQ_Contact(in1 := "BUFFER".PROCESS, in2 := 111)
   END_RUNG wire#w2
   RUNG wire#w3
      { S7_Templates := "SrcType := Int" } EQ_Contact(in1 := "BUFFER".PROCESS, in2 := 160)
   END_RUNG wire#w2
   RUNG wire#w3
      { S7_Templates := "SrcType := Int" } EQ_Contact(in1 := "BUFFER".PROCESS, in2 := 330)
   END_RUNG wire#w2
   RUNG wire#w3
      { S7_Templates := "SrcType := Int" } EQ_Contact(in1 := "BUFFER".PROCESS, in2 := 350)
   END_RUNG wire#w2
   RUNG wire#w3
      { S7_Templates := "SrcType := Int" } EQ_Contact(in1 := "BUFFER".PROCESS, in2 := 430)
   END_RUNG wire#w2
   RUNG wire#w3
      { S7_Templates := "SrcType := Int" } EQ_Contact(in1 := "BUFFER".PROCESS, in2 := 450)
   END_RUNG wire#w2
   RUNG wire#w3
      { S7_Templates := "SrcType := Int" } EQ_Contact(in1 := "BUFFER".PROCESS, in2 := 530)
   END_RUNG wire#w2
   RUNG wire#w3
      { S7_Templates := "SrcType := Int" } EQ_Contact(in1 := "BUFFER".PROCESS, in2 := 540)
   END_RUNG wire#w2
   RUNG wire#w3
      { S7_Templates := "SrcType := Int" } EQ_Contact(in1 := "BUFFER".PROCESS, in2 := 570)
   END_RUNG wire#w2
   RUNG wire#w3
      { S7_Templates := "SrcType := Int" } GE_Contact(in1 := "BUFFER".PROCESS, in2 := 121)
      { S7_Templates := "SrcType := Int" } LE_Contact(in1 := "BUFFER".PROCESS, in2 := 130)
      Contact( "AlwaysFALSE" )
   END_RUNG wire#w2
   RUNG wire#w3
      { S7_Templates := "SrcType := Int" } EQ_Contact(in1 := "BUFFER".PROCESS, in2 := 520)
   END_RUNG wire#w2
   RUNG wire#w3
      { S7_Templates := "SrcType := Int" } EQ_Contact(in1 := "BUFFER".PROCESS, in2 := 420)
      Contact( "AlwaysFALSE" )
   END_RUNG wire#w2
   RUNG wire#w3
      { S7_Templates := "SrcType := Int" } EQ_Contact(in1 := "BUFFER".PROCESS, in2 := 320)
   END_RUNG wire#w2
   // the same network as SCL:
   "OP".CIP_OUT := "AlwaysTRUE" AND ((("BUFFER"."MODE SELECTION" = 2) AND "MANUAL BIT".CIP_OUT) OR (("BUFFER"."MODE SELECTION" = 1) AND (("BUFFER".PROCESS = 20) OR ("BUFFER".PROCESS = 40) OR ("BUFFER".PROCESS = 140) OR ("BUFFER".PROCESS = 120) OR ("BUFFER".PROCESS = 111) OR ("BUFFER".PROCESS = 160) OR ("BUFFER".PROCESS = 330) OR ("BUFFER".PROCESS = 350) OR ("BUFFER".PROCESS = 430) OR ("BUFFER".PROCESS = 450) OR ("BUFFER".PROCESS = 530) OR ("BUFFER".PROCESS = 540) OR ("BUFFER".PROCESS = 570) OR (("BUFFER".PROCESS >= 121) AND ("BUFFER".PROCESS <= 130) AND "AlwaysFALSE") OR ("BUFFER".PROCESS = 520) OR (("BUFFER".PROCESS = 420) AND "AlwaysFALSE") OR ("BUFFER".PROCESS = 320)))) AND ("SET_PARAMETERS".PLANT_SELECT = 1) AND ("SET_PARAMETERS".PLANT2_TANK_SELECT = 3) AND NOT "CYCLE PAUSE" AND NOT "ERROR";
END_REGION

REGION Network 39: reset 18 and 25
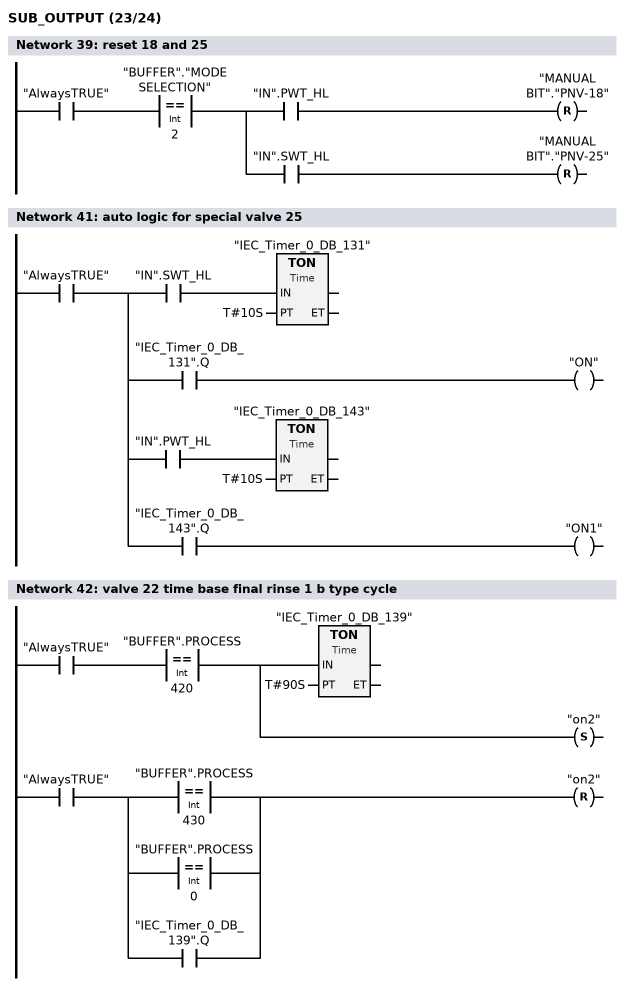
   RUNG wire#powerrail
      Contact( "AlwaysTRUE" )
      { S7_Templates := "SrcType := Int" } EQ_Contact(in1 := "BUFFER"."MODE SELECTION", in2 := 2)
      wire#w1
      Contact( "IN".PWT_HL )
      R_Coil( "MANUAL BIT"."PNV-18" )
   END_RUNG
   RUNG wire#w1
      Contact( "IN".SWT_HL )
      R_Coil( "MANUAL BIT"."PNV-25" )
   END_RUNG
   // the same network as SCL:
   #_w1 := "AlwaysTRUE" AND ("BUFFER"."MODE SELECTION" = 2);
   IF #_w1 AND "IN".PWT_HL THEN "MANUAL BIT"."PNV-18" := FALSE; END_IF;
   IF #_w1 AND "IN".SWT_HL THEN "MANUAL BIT"."PNV-25" := FALSE; END_IF;
END_REGION

REGION Network 41: auto logic for special valve 25
   RUNG wire#powerrail
      Contact( "AlwaysTRUE" )
      wire#w1
      Contact( "IN".SWT_HL )
      { S7_Templates := "time_type := Time" } "IEC_Timer_0_DB_131".TON(pt := T#10S, et =>)
   END_RUNG
   RUNG wire#w1
      Contact( "IEC_Timer_0_DB_131".Q )
      Coil( "ON" )
   END_RUNG
   RUNG wire#w1
      Contact( "IN".PWT_HL )
      { S7_Templates := "time_type := Time" } "IEC_Timer_0_DB_143".TON(pt := T#10S, et =>)
   END_RUNG
   RUNG wire#w1
      Contact( "IEC_Timer_0_DB_143".Q )
      Coil( "ON1" )
   END_RUNG
   // the same network as SCL:
   "IEC_Timer_0_DB_131".TON(IN := "AlwaysTRUE" AND "IN".SWT_HL, PT := T#10S);
   "ON" := "AlwaysTRUE" AND "IEC_Timer_0_DB_131".Q;
   "IEC_Timer_0_DB_143".TON(IN := "AlwaysTRUE" AND "IN".PWT_HL, PT := T#10S);
   "ON1" := "AlwaysTRUE" AND "IEC_Timer_0_DB_143".Q;
END_REGION

REGION Network 42: valve 22 time base final rinse 1 b type cycle
   RUNG wire#powerrail
      Contact( "AlwaysTRUE" )
      { S7_Templates := "SrcType := Int" } EQ_Contact(in1 := "BUFFER".PROCESS, in2 := 420)
      wire#w1
      { S7_Templates := "time_type := Time" } "IEC_Timer_0_DB_139".TON(pt := T#90S, et =>)
   END_RUNG
   RUNG wire#w1
      S_Coil( "on2" )
   END_RUNG
   RUNG wire#powerrail
      Contact( "AlwaysTRUE" )
      wire#w2
      { S7_Templates := "SrcType := Int" } EQ_Contact(in1 := "BUFFER".PROCESS, in2 := 430)
      wire#w3
      R_Coil( "on2" )
   END_RUNG
   RUNG wire#w2
      { S7_Templates := "SrcType := Int" } EQ_Contact(in1 := "BUFFER".PROCESS, in2 := 0)
   END_RUNG wire#w3
   RUNG wire#w2
      Contact( "IEC_Timer_0_DB_139".Q )
   END_RUNG wire#w3
   // the same network as SCL:
   #_w1 := "AlwaysTRUE" AND ("BUFFER".PROCESS = 420);
   "IEC_Timer_0_DB_139".TON(IN := #_w1, PT := T#90S);
   IF #_w1 THEN "on2" := TRUE; END_IF;
   IF "AlwaysTRUE" AND (("BUFFER".PROCESS = 430) OR ("BUFFER".PROCESS = 0) OR "IEC_Timer_0_DB_139".Q) THEN
       "on2" := FALSE;
   END_IF;
END_REGION

REGION Network 43: for air purpose will be on 5sec valve11
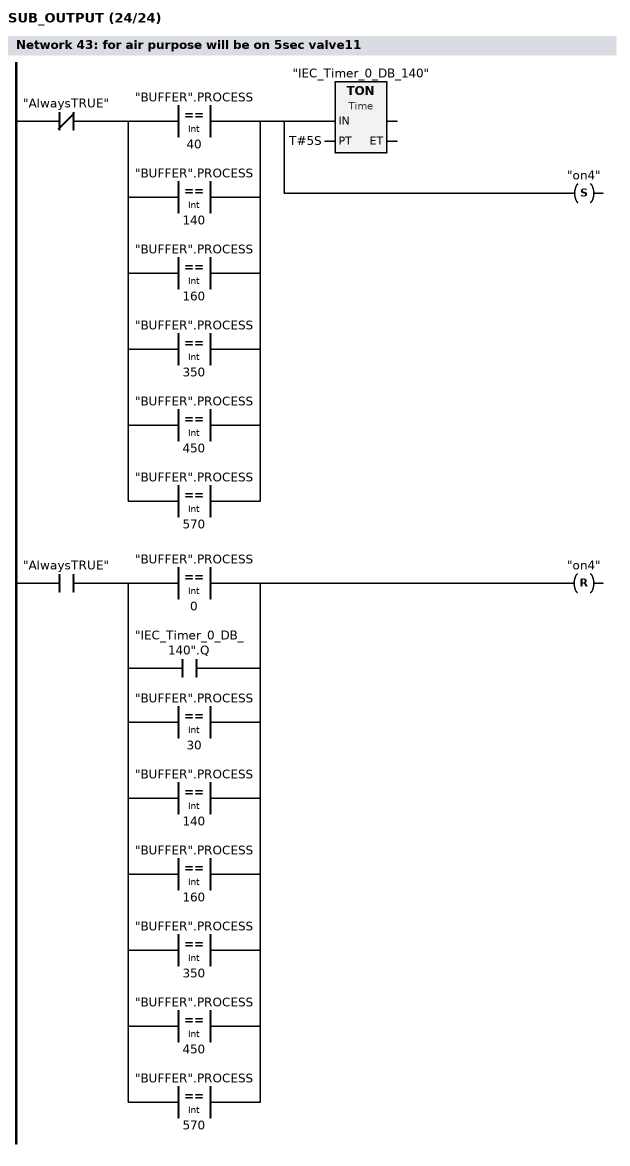
   RUNG wire#powerrail
      I_Contact( "AlwaysTRUE" )
      wire#w1
      { S7_Templates := "SrcType := Int" } EQ_Contact(in1 := "BUFFER".PROCESS, in2 := 40)
      wire#w2
      { S7_Templates := "time_type := Time" } "IEC_Timer_0_DB_140".TON(pt := T#5S, et =>)
   END_RUNG
   RUNG wire#w1
      { S7_Templates := "SrcType := Int" } EQ_Contact(in1 := "BUFFER".PROCESS, in2 := 140)
   END_RUNG wire#w2
   RUNG wire#w1
      { S7_Templates := "SrcType := Int" } EQ_Contact(in1 := "BUFFER".PROCESS, in2 := 160)
   END_RUNG wire#w2
   RUNG wire#w1
      { S7_Templates := "SrcType := Int" } EQ_Contact(in1 := "BUFFER".PROCESS, in2 := 350)
   END_RUNG wire#w2
   RUNG wire#w1
      { S7_Templates := "SrcType := Int" } EQ_Contact(in1 := "BUFFER".PROCESS, in2 := 450)
   END_RUNG wire#w2
   RUNG wire#w1
      { S7_Templates := "SrcType := Int" } EQ_Contact(in1 := "BUFFER".PROCESS, in2 := 570)
   END_RUNG wire#w2
   RUNG wire#w2
      S_Coil( "on4" )
   END_RUNG
   RUNG wire#powerrail
      Contact( "AlwaysTRUE" )
      wire#w3
      { S7_Templates := "SrcType := Int" } EQ_Contact(in1 := "BUFFER".PROCESS, in2 := 0)
      wire#w4
      R_Coil( "on4" )
   END_RUNG
   RUNG wire#w3
      Contact( "IEC_Timer_0_DB_140".Q )
   END_RUNG wire#w4
   RUNG wire#w3
      { S7_Templates := "SrcType := Int" } EQ_Contact(in1 := "BUFFER".PROCESS, in2 := 30)
   END_RUNG wire#w4
   RUNG wire#w3
      { S7_Templates := "SrcType := Int" } EQ_Contact(in1 := "BUFFER".PROCESS, in2 := 140)
   END_RUNG wire#w4
   RUNG wire#w3
      { S7_Templates := "SrcType := Int" } EQ_Contact(in1 := "BUFFER".PROCESS, in2 := 160)
   END_RUNG wire#w4
   RUNG wire#w3
      { S7_Templates := "SrcType := Int" } EQ_Contact(in1 := "BUFFER".PROCESS, in2 := 350)
   END_RUNG wire#w4
   RUNG wire#w3
      { S7_Templates := "SrcType := Int" } EQ_Contact(in1 := "BUFFER".PROCESS, in2 := 450)
   END_RUNG wire#w4
   RUNG wire#w3
      { S7_Templates := "SrcType := Int" } EQ_Contact(in1 := "BUFFER".PROCESS, in2 := 570)
   END_RUNG wire#w4
   // the same network as SCL:
   #_w1 := NOT "AlwaysTRUE" AND (("BUFFER".PROCESS = 40) OR ("BUFFER".PROCESS = 140) OR ("BUFFER".PROCESS = 160) OR ("BUFFER".PROCESS = 350) OR ("BUFFER".PROCESS = 450) OR ("BUFFER".PROCESS = 570));
   "IEC_Timer_0_DB_140".TON(IN := #_w1, PT := T#5S);
   IF #_w1 THEN "on4" := TRUE; END_IF;
   IF "AlwaysTRUE" AND (("BUFFER".PROCESS = 0) OR "IEC_Timer_0_DB_140".Q OR ("BUFFER".PROCESS = 30) OR ("BUFFER".PROCESS = 140) OR ("BUFFER".PROCESS = 160) OR ("BUFFER".PROCESS = 350) OR ("BUFFER".PROCESS = 450) OR ("BUFFER".PROCESS = 570)) THEN
       "on4" := FALSE;
   END_IF;
END_REGION
END_FUNCTION
